REGION Network 2: HOPPER 1 UNIT 01
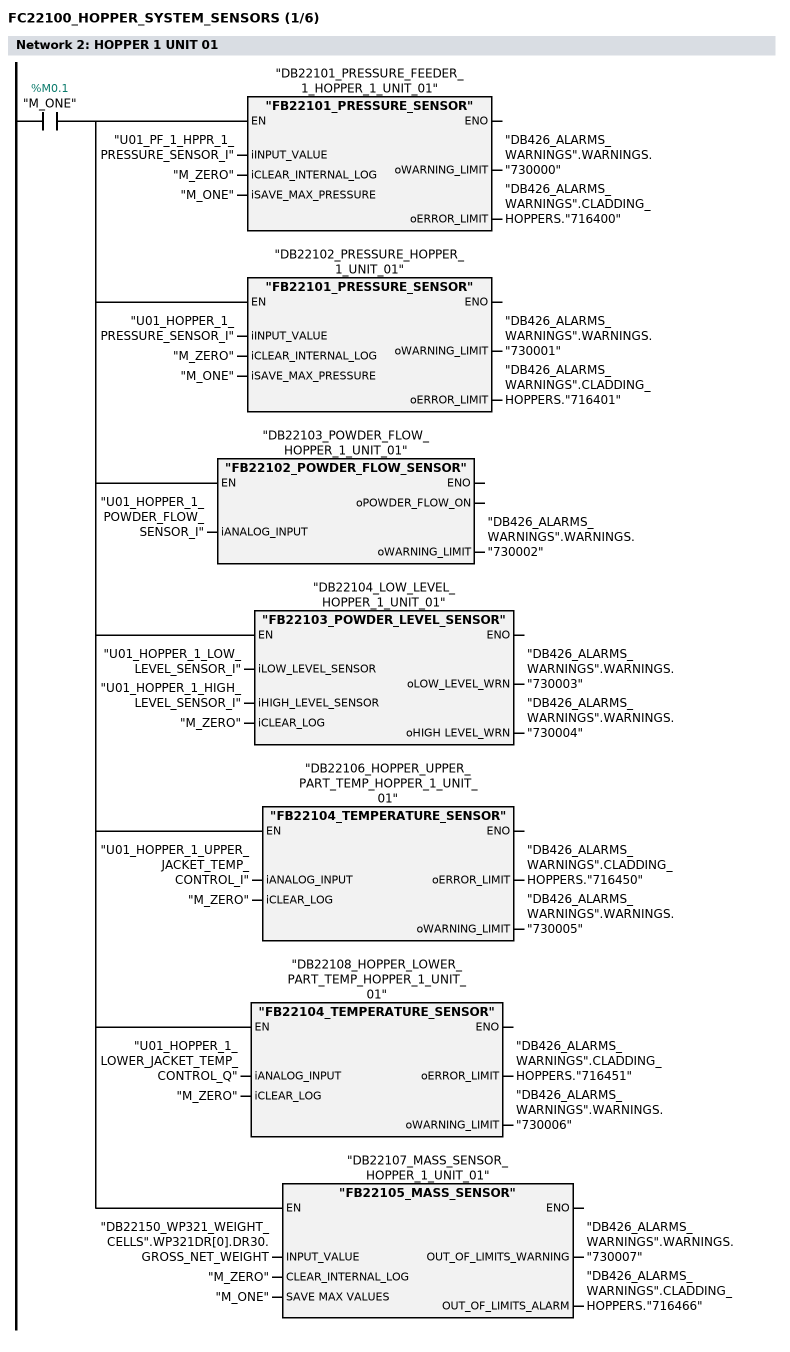
   RUNG wire#powerrail
      Contact( "M_ONE" )
      wire#w1
      "DB22101_PRESSURE_FEEDER_1_HOPPER_1_UNIT_01"(iINPUT_VALUE := "U01_PF_1_HPPR_1_PRESSURE_SENSOR_I", iCLEAR_INTERNAL_LOG := "M_ZERO", iSAVE_MAX_PRESSURE := "M_ONE", oWARNING_LIMIT => "DB426_ALARMS_WARNINGS".WARNINGS."730000", oERROR_LIMIT => "DB426_ALARMS_WARNINGS".CLADDING_HOPPERS."716400")
   END_RUNG
   RUNG wire#w1
      "DB22102_PRESSURE_HOPPER_1_UNIT_01"(iINPUT_VALUE := "U01_HOPPER_1_PRESSURE_SENSOR_I", iCLEAR_INTERNAL_LOG := "M_ZERO", iSAVE_MAX_PRESSURE := "M_ONE", oWARNING_LIMIT => "DB426_ALARMS_WARNINGS".WARNINGS."730001", oERROR_LIMIT => "DB426_ALARMS_WARNINGS".CLADDING_HOPPERS."716401")
   END_RUNG
   RUNG wire#w1
      "DB22103_POWDER_FLOW_HOPPER_1_UNIT_01"(iANALOG_INPUT := "U01_HOPPER_1_POWDER_FLOW_SENSOR_I", oPOWDER_FLOW_ON =>, oWARNING_LIMIT => "DB426_ALARMS_WARNINGS".WARNINGS."730002")
   END_RUNG
   RUNG wire#w1
      "DB22104_LOW_LEVEL_HOPPER_1_UNIT_01"(iLOW_LEVEL_SENSOR := "U01_HOPPER_1_LOW_LEVEL_SENSOR_I", iHIGH_LEVEL_SENSOR := "U01_HOPPER_1_HIGH_LEVEL_SENSOR_I", iCLEAR_LOG := "M_ZERO", oLOW_LEVEL_WRN => "DB426_ALARMS_WARNINGS".WARNINGS."730003", "oHIGH LEVEL_WRN" => "DB426_ALARMS_WARNINGS".WARNINGS."730004")
   END_RUNG
   RUNG wire#w1
      "DB22106_HOPPER_UPPER_PART_TEMP_HOPPER_1_UNIT_01"(iANALOG_INPUT := "U01_HOPPER_1_UPPER_JACKET_TEMP_CONTROL_I", iCLEAR_LOG := "M_ZERO", oERROR_LIMIT => "DB426_ALARMS_WARNINGS".CLADDING_HOPPERS."716450", oWARNING_LIMIT => "DB426_ALARMS_WARNINGS".WARNINGS."730005")
   END_RUNG
   RUNG wire#w1
      "DB22108_HOPPER_LOWER_PART_TEMP_HOPPER_1_UNIT_01"(iANALOG_INPUT := "U01_HOPPER_1_LOWER_JACKET_TEMP_CONTROL_Q", iCLEAR_LOG := "M_ZERO", oERROR_LIMIT => "DB426_ALARMS_WARNINGS".CLADDING_HOPPERS."716451", oWARNING_LIMIT => "DB426_ALARMS_WARNINGS".WARNINGS."730006")
   END_RUNG
   RUNG wire#w1
      "DB22107_MASS_SENSOR_HOPPER_1_UNIT_01"(INPUT_VALUE := "DB22150_WP321_WEIGHT_CELLS".WP321DR[0].DR30.GROSS_NET_WEIGHT, CLEAR_INTERNAL_LOG := "M_ZERO", "SAVE MAX VALUES" := "M_ONE", OUT_OF_LIMITS_WARNING => "DB426_ALARMS_WARNINGS".WARNINGS."730007", OUT_OF_LIMITS_ALARM => "DB426_ALARMS_WARNINGS".CLADDING_HOPPERS."716466")
   END_RUNG
   // the same network as SCL:
   #_w1 := "M_ONE";
   IF #_w1 THEN
       "DB22101_PRESSURE_FEEDER_1_HOPPER_1_UNIT_01"(iINPUT_VALUE := "U01_PF_1_HPPR_1_PRESSURE_SENSOR_I",   // "FB22101_PRESSURE_SENSOR"
                               iCLEAR_INTERNAL_LOG := "M_ZERO",
                               iSAVE_MAX_PRESSURE := "M_ONE",
                               oWARNING_LIMIT => "DB426_ALARMS_WARNINGS".WARNINGS."730000",
                               oERROR_LIMIT => "DB426_ALARMS_WARNINGS".CLADDING_HOPPERS."716400");
       "DB22102_PRESSURE_HOPPER_1_UNIT_01"(iINPUT_VALUE := "U01_HOPPER_1_PRESSURE_SENSOR_I",   // "FB22101_PRESSURE_SENSOR"
                               iCLEAR_INTERNAL_LOG := "M_ZERO",
                               iSAVE_MAX_PRESSURE := "M_ONE",
                               oWARNING_LIMIT => "DB426_ALARMS_WARNINGS".WARNINGS."730001",
                               oERROR_LIMIT => "DB426_ALARMS_WARNINGS".CLADDING_HOPPERS."716401");
       "DB22103_POWDER_FLOW_HOPPER_1_UNIT_01"(iANALOG_INPUT := "U01_HOPPER_1_POWDER_FLOW_SENSOR_I",   // "FB22102_POWDER_FLOW_SENSOR"
                               oWARNING_LIMIT => "DB426_ALARMS_WARNINGS".WARNINGS."730002");
       "DB22104_LOW_LEVEL_HOPPER_1_UNIT_01"(iLOW_LEVEL_SENSOR := "U01_HOPPER_1_LOW_LEVEL_SENSOR_I",   // "FB22103_POWDER_LEVEL_SENSOR"
                               iHIGH_LEVEL_SENSOR := "U01_HOPPER_1_HIGH_LEVEL_SENSOR_I",
                               iCLEAR_LOG := "M_ZERO",
                               oLOW_LEVEL_WRN => "DB426_ALARMS_WARNINGS".WARNINGS."730003",
                               "oHIGH LEVEL_WRN" => "DB426_ALARMS_WARNINGS".WARNINGS."730004");
       "DB22106_HOPPER_UPPER_PART_TEMP_HOPPER_1_UNIT_01"(iANALOG_INPUT := "U01_HOPPER_1_UPPER_JACKET_TEMP_CONTROL_I",   // "FB22104_TEMPERATURE_SENSOR"
                               iCLEAR_LOG := "M_ZERO",
                               oERROR_LIMIT => "DB426_ALARMS_WARNINGS".CLADDING_HOPPERS."716450",
                               oWARNING_LIMIT => "DB426_ALARMS_WARNINGS".WARNINGS."730005");
       "DB22108_HOPPER_LOWER_PART_TEMP_HOPPER_1_UNIT_01"(iANALOG_INPUT := "U01_HOPPER_1_LOWER_JACKET_TEMP_CONTROL_Q",   // "FB22104_TEMPERATURE_SENSOR"
                               iCLEAR_LOG := "M_ZERO",
                               oERROR_LIMIT => "DB426_ALARMS_WARNINGS".CLADDING_HOPPERS."716451",
                               oWARNING_LIMIT => "DB426_ALARMS_WARNINGS".WARNINGS."730006");
       "DB22107_MASS_SENSOR_HOPPER_1_UNIT_01"(INPUT_VALUE := "DB22150_WP321_WEIGHT_CELLS".WP321DR[0].DR30.GROSS_NET_WEIGHT,   // "FB22105_MASS_SENSOR"
                               CLEAR_INTERNAL_LOG := "M_ZERO",
                               "SAVE MAX VALUES" := "M_ONE",
                               OUT_OF_LIMITS_WARNING => "DB426_ALARMS_WARNINGS".WARNINGS."730007",
                               OUT_OF_LIMITS_ALARM => "DB426_ALARMS_WARNINGS".CLADDING_HOPPERS."716466");
   END_IF;
END_REGION

REGION Network 3: HOPPER 2 UNIT 01
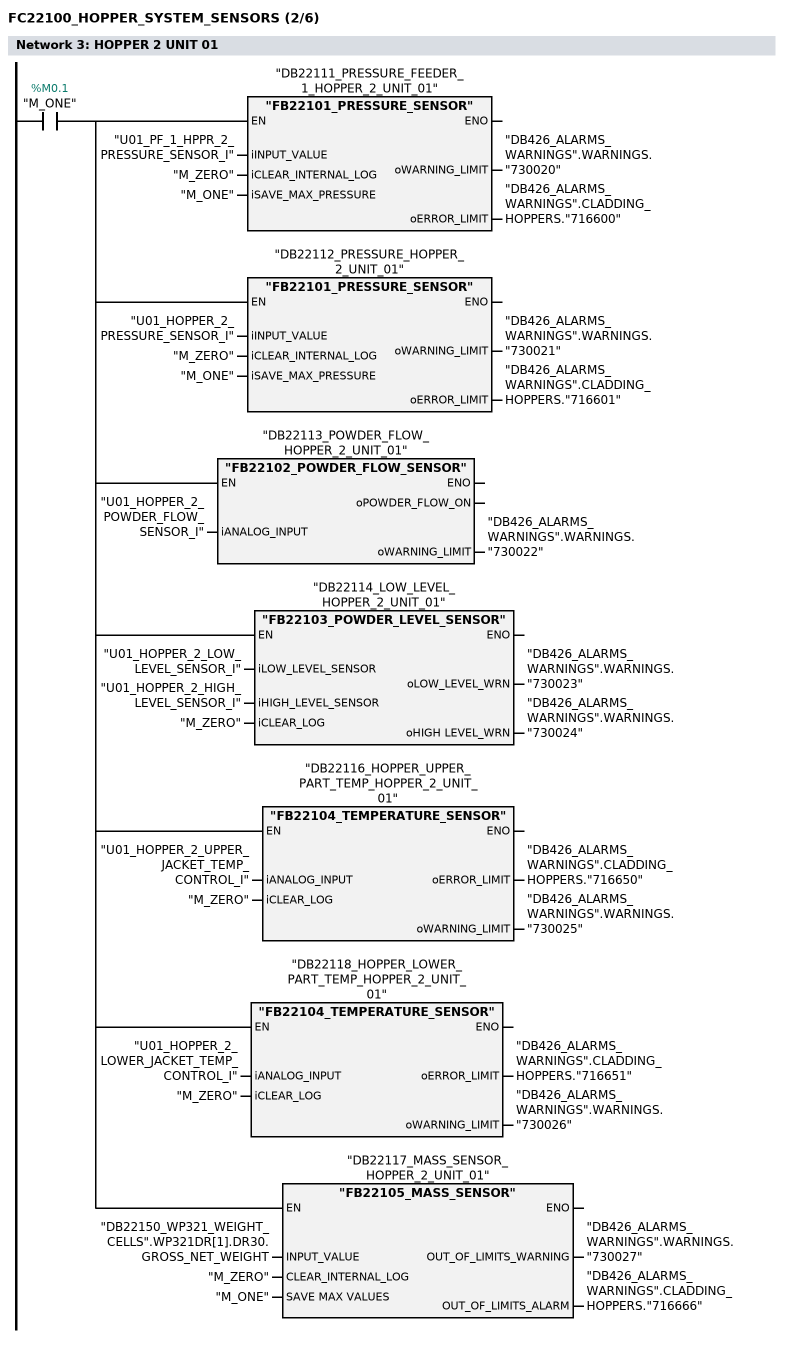
   RUNG wire#powerrail
      Contact( "M_ONE" )
      wire#w1
      "DB22111_PRESSURE_FEEDER_1_HOPPER_2_UNIT_01"(iINPUT_VALUE := "U01_PF_1_HPPR_2_PRESSURE_SENSOR_I", iCLEAR_INTERNAL_LOG := "M_ZERO", iSAVE_MAX_PRESSURE := "M_ONE", oWARNING_LIMIT => "DB426_ALARMS_WARNINGS".WARNINGS."730020", oERROR_LIMIT => "DB426_ALARMS_WARNINGS".CLADDING_HOPPERS."716600")
   END_RUNG
   RUNG wire#w1
      "DB22112_PRESSURE_HOPPER_2_UNIT_01"(iINPUT_VALUE := "U01_HOPPER_2_PRESSURE_SENSOR_I", iCLEAR_INTERNAL_LOG := "M_ZERO", iSAVE_MAX_PRESSURE := "M_ONE", oWARNING_LIMIT => "DB426_ALARMS_WARNINGS".WARNINGS."730021", oERROR_LIMIT => "DB426_ALARMS_WARNINGS".CLADDING_HOPPERS."716601")
   END_RUNG
   RUNG wire#w1
      "DB22113_POWDER_FLOW_HOPPER_2_UNIT_01"(iANALOG_INPUT := "U01_HOPPER_2_POWDER_FLOW_SENSOR_I", oPOWDER_FLOW_ON =>, oWARNING_LIMIT => "DB426_ALARMS_WARNINGS".WARNINGS."730022")
   END_RUNG
   RUNG wire#w1
      "DB22114_LOW_LEVEL_HOPPER_2_UNIT_01"(iLOW_LEVEL_SENSOR := "U01_HOPPER_2_LOW_LEVEL_SENSOR_I", iHIGH_LEVEL_SENSOR := "U01_HOPPER_2_HIGH_LEVEL_SENSOR_I", iCLEAR_LOG := "M_ZERO", oLOW_LEVEL_WRN => "DB426_ALARMS_WARNINGS".WARNINGS."730023", "oHIGH LEVEL_WRN" => "DB426_ALARMS_WARNINGS".WARNINGS."730024")
   END_RUNG
   RUNG wire#w1
      "DB22116_HOPPER_UPPER_PART_TEMP_HOPPER_2_UNIT_01"(iANALOG_INPUT := "U01_HOPPER_2_UPPER_JACKET_TEMP_CONTROL_I", iCLEAR_LOG := "M_ZERO", oERROR_LIMIT => "DB426_ALARMS_WARNINGS".CLADDING_HOPPERS."716650", oWARNING_LIMIT => "DB426_ALARMS_WARNINGS".WARNINGS."730025")
   END_RUNG
   RUNG wire#w1
      "DB22118_HOPPER_LOWER_PART_TEMP_HOPPER_2_UNIT_01"(iANALOG_INPUT := "U01_HOPPER_2_LOWER_JACKET_TEMP_CONTROL_I", iCLEAR_LOG := "M_ZERO", oERROR_LIMIT => "DB426_ALARMS_WARNINGS".CLADDING_HOPPERS."716651", oWARNING_LIMIT => "DB426_ALARMS_WARNINGS".WARNINGS."730026")
   END_RUNG
   RUNG wire#w1
      "DB22117_MASS_SENSOR_HOPPER_2_UNIT_01"(INPUT_VALUE := "DB22150_WP321_WEIGHT_CELLS".WP321DR[1].DR30.GROSS_NET_WEIGHT, CLEAR_INTERNAL_LOG := "M_ZERO", "SAVE MAX VALUES" := "M_ONE", OUT_OF_LIMITS_WARNING => "DB426_ALARMS_WARNINGS".WARNINGS."730027", OUT_OF_LIMITS_ALARM => "DB426_ALARMS_WARNINGS".CLADDING_HOPPERS."716666")
   END_RUNG
   // the same network as SCL:
   #_w1 := "M_ONE";
   IF #_w1 THEN
       "DB22111_PRESSURE_FEEDER_1_HOPPER_2_UNIT_01"(iINPUT_VALUE := "U01_PF_1_HPPR_2_PRESSURE_SENSOR_I",   // "FB22101_PRESSURE_SENSOR"
                               iCLEAR_INTERNAL_LOG := "M_ZERO",
                               iSAVE_MAX_PRESSURE := "M_ONE",
                               oWARNING_LIMIT => "DB426_ALARMS_WARNINGS".WARNINGS."730020",
                               oERROR_LIMIT => "DB426_ALARMS_WARNINGS".CLADDING_HOPPERS."716600");
       "DB22112_PRESSURE_HOPPER_2_UNIT_01"(iINPUT_VALUE := "U01_HOPPER_2_PRESSURE_SENSOR_I",   // "FB22101_PRESSURE_SENSOR"
                               iCLEAR_INTERNAL_LOG := "M_ZERO",
                               iSAVE_MAX_PRESSURE := "M_ONE",
                               oWARNING_LIMIT => "DB426_ALARMS_WARNINGS".WARNINGS."730021",
                               oERROR_LIMIT => "DB426_ALARMS_WARNINGS".CLADDING_HOPPERS."716601");
       "DB22113_POWDER_FLOW_HOPPER_2_UNIT_01"(iANALOG_INPUT := "U01_HOPPER_2_POWDER_FLOW_SENSOR_I",   // "FB22102_POWDER_FLOW_SENSOR"
                               oWARNING_LIMIT => "DB426_ALARMS_WARNINGS".WARNINGS."730022");
       "DB22114_LOW_LEVEL_HOPPER_2_UNIT_01"(iLOW_LEVEL_SENSOR := "U01_HOPPER_2_LOW_LEVEL_SENSOR_I",   // "FB22103_POWDER_LEVEL_SENSOR"
                               iHIGH_LEVEL_SENSOR := "U01_HOPPER_2_HIGH_LEVEL_SENSOR_I",
                               iCLEAR_LOG := "M_ZERO",
                               oLOW_LEVEL_WRN => "DB426_ALARMS_WARNINGS".WARNINGS."730023",
                               "oHIGH LEVEL_WRN" => "DB426_ALARMS_WARNINGS".WARNINGS."730024");
       "DB22116_HOPPER_UPPER_PART_TEMP_HOPPER_2_UNIT_01"(iANALOG_INPUT := "U01_HOPPER_2_UPPER_JACKET_TEMP_CONTROL_I",   // "FB22104_TEMPERATURE_SENSOR"
                               iCLEAR_LOG := "M_ZERO",
                               oERROR_LIMIT => "DB426_ALARMS_WARNINGS".CLADDING_HOPPERS."716650",
                               oWARNING_LIMIT => "DB426_ALARMS_WARNINGS".WARNINGS."730025");
       "DB22118_HOPPER_LOWER_PART_TEMP_HOPPER_2_UNIT_01"(iANALOG_INPUT := "U01_HOPPER_2_LOWER_JACKET_TEMP_CONTROL_I",   // "FB22104_TEMPERATURE_SENSOR"
                               iCLEAR_LOG := "M_ZERO",
                               oERROR_LIMIT => "DB426_ALARMS_WARNINGS".CLADDING_HOPPERS."716651",
                               oWARNING_LIMIT => "DB426_ALARMS_WARNINGS".WARNINGS."730026");
       "DB22117_MASS_SENSOR_HOPPER_2_UNIT_01"(INPUT_VALUE := "DB22150_WP321_WEIGHT_CELLS".WP321DR[1].DR30.GROSS_NET_WEIGHT,   // "FB22105_MASS_SENSOR"
                               CLEAR_INTERNAL_LOG := "M_ZERO",
                               "SAVE MAX VALUES" := "M_ONE",
                               OUT_OF_LIMITS_WARNING => "DB426_ALARMS_WARNINGS".WARNINGS."730027",
                               OUT_OF_LIMITS_ALARM => "DB426_ALARMS_WARNINGS".CLADDING_HOPPERS."716666");
   END_IF;
END_REGION

REGION Network 4: /////_UNIT_02_SENSORS_/////
END_REGION

REGION Network 5: HOPPER 1 UNIT 02
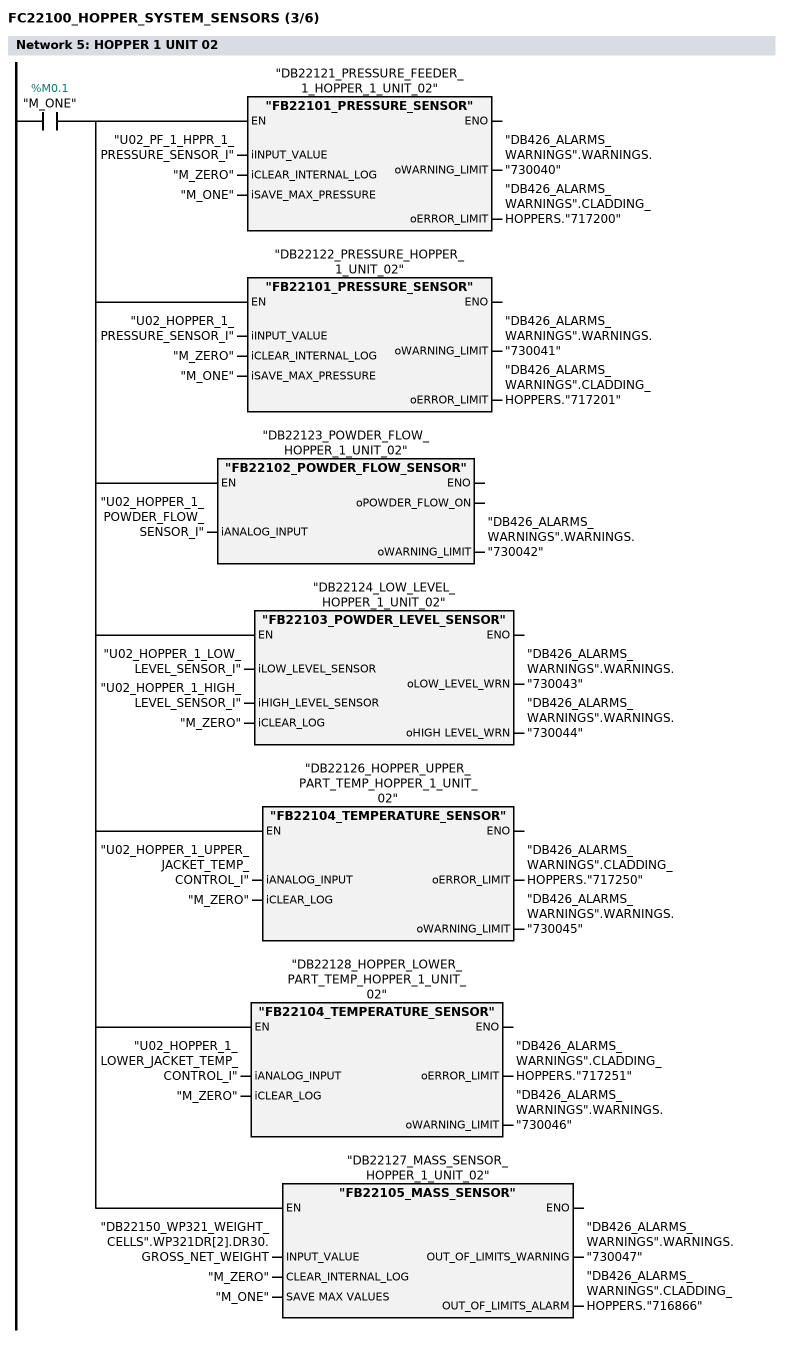
   RUNG wire#powerrail
      Contact( "M_ONE" )
      wire#w1
      "DB22121_PRESSURE_FEEDER_1_HOPPER_1_UNIT_02"(iINPUT_VALUE := "U02_PF_1_HPPR_1_PRESSURE_SENSOR_I", iCLEAR_INTERNAL_LOG := "M_ZERO", iSAVE_MAX_PRESSURE := "M_ONE", oWARNING_LIMIT => "DB426_ALARMS_WARNINGS".WARNINGS."730040", oERROR_LIMIT => "DB426_ALARMS_WARNINGS".CLADDING_HOPPERS."717200")
   END_RUNG
   RUNG wire#w1
      "DB22122_PRESSURE_HOPPER_1_UNIT_02"(iINPUT_VALUE := "U02_HOPPER_1_PRESSURE_SENSOR_I", iCLEAR_INTERNAL_LOG := "M_ZERO", iSAVE_MAX_PRESSURE := "M_ONE", oWARNING_LIMIT => "DB426_ALARMS_WARNINGS".WARNINGS."730041", oERROR_LIMIT => "DB426_ALARMS_WARNINGS".CLADDING_HOPPERS."717201")
   END_RUNG
   RUNG wire#w1
      "DB22123_POWDER_FLOW_HOPPER_1_UNIT_02"(iANALOG_INPUT := "U02_HOPPER_1_POWDER_FLOW_SENSOR_I", oPOWDER_FLOW_ON =>, oWARNING_LIMIT => "DB426_ALARMS_WARNINGS".WARNINGS."730042")
   END_RUNG
   RUNG wire#w1
      "DB22124_LOW_LEVEL_HOPPER_1_UNIT_02"(iLOW_LEVEL_SENSOR := "U02_HOPPER_1_LOW_LEVEL_SENSOR_I", iHIGH_LEVEL_SENSOR := "U02_HOPPER_1_HIGH_LEVEL_SENSOR_I", iCLEAR_LOG := "M_ZERO", oLOW_LEVEL_WRN => "DB426_ALARMS_WARNINGS".WARNINGS."730043", "oHIGH LEVEL_WRN" => "DB426_ALARMS_WARNINGS".WARNINGS."730044")
   END_RUNG
   RUNG wire#w1
      "DB22126_HOPPER_UPPER_PART_TEMP_HOPPER_1_UNIT_02"(iANALOG_INPUT := "U02_HOPPER_1_UPPER_JACKET_TEMP_CONTROL_I", iCLEAR_LOG := "M_ZERO", oERROR_LIMIT => "DB426_ALARMS_WARNINGS".CLADDING_HOPPERS."717250", oWARNING_LIMIT => "DB426_ALARMS_WARNINGS".WARNINGS."730045")
   END_RUNG
   RUNG wire#w1
      "DB22128_HOPPER_LOWER_PART_TEMP_HOPPER_1_UNIT_02"(iANALOG_INPUT := "U02_HOPPER_1_LOWER_JACKET_TEMP_CONTROL_I", iCLEAR_LOG := "M_ZERO", oERROR_LIMIT => "DB426_ALARMS_WARNINGS".CLADDING_HOPPERS."717251", oWARNING_LIMIT => "DB426_ALARMS_WARNINGS".WARNINGS."730046")
   END_RUNG
   RUNG wire#w1
      "DB22127_MASS_SENSOR_HOPPER_1_UNIT_02"(INPUT_VALUE := "DB22150_WP321_WEIGHT_CELLS".WP321DR[2].DR30.GROSS_NET_WEIGHT, CLEAR_INTERNAL_LOG := "M_ZERO", "SAVE MAX VALUES" := "M_ONE", OUT_OF_LIMITS_WARNING => "DB426_ALARMS_WARNINGS".WARNINGS."730047", OUT_OF_LIMITS_ALARM => "DB426_ALARMS_WARNINGS".CLADDING_HOPPERS."716866")
   END_RUNG
   // the same network as SCL:
   #_w1 := "M_ONE";
   IF #_w1 THEN
       "DB22121_PRESSURE_FEEDER_1_HOPPER_1_UNIT_02"(iINPUT_VALUE := "U02_PF_1_HPPR_1_PRESSURE_SENSOR_I",   // "FB22101_PRESSURE_SENSOR"
                               iCLEAR_INTERNAL_LOG := "M_ZERO",
                               iSAVE_MAX_PRESSURE := "M_ONE",
                               oWARNING_LIMIT => "DB426_ALARMS_WARNINGS".WARNINGS."730040",
                               oERROR_LIMIT => "DB426_ALARMS_WARNINGS".CLADDING_HOPPERS."717200");
       "DB22122_PRESSURE_HOPPER_1_UNIT_02"(iINPUT_VALUE := "U02_HOPPER_1_PRESSURE_SENSOR_I",   // "FB22101_PRESSURE_SENSOR"
                               iCLEAR_INTERNAL_LOG := "M_ZERO",
                               iSAVE_MAX_PRESSURE := "M_ONE",
                               oWARNING_LIMIT => "DB426_ALARMS_WARNINGS".WARNINGS."730041",
                               oERROR_LIMIT => "DB426_ALARMS_WARNINGS".CLADDING_HOPPERS."717201");
       "DB22123_POWDER_FLOW_HOPPER_1_UNIT_02"(iANALOG_INPUT := "U02_HOPPER_1_POWDER_FLOW_SENSOR_I",   // "FB22102_POWDER_FLOW_SENSOR"
                               oWARNING_LIMIT => "DB426_ALARMS_WARNINGS".WARNINGS."730042");
       "DB22124_LOW_LEVEL_HOPPER_1_UNIT_02"(iLOW_LEVEL_SENSOR := "U02_HOPPER_1_LOW_LEVEL_SENSOR_I",   // "FB22103_POWDER_LEVEL_SENSOR"
                               iHIGH_LEVEL_SENSOR := "U02_HOPPER_1_HIGH_LEVEL_SENSOR_I",
                               iCLEAR_LOG := "M_ZERO",
                               oLOW_LEVEL_WRN => "DB426_ALARMS_WARNINGS".WARNINGS."730043",
                               "oHIGH LEVEL_WRN" => "DB426_ALARMS_WARNINGS".WARNINGS."730044");
       "DB22126_HOPPER_UPPER_PART_TEMP_HOPPER_1_UNIT_02"(iANALOG_INPUT := "U02_HOPPER_1_UPPER_JACKET_TEMP_CONTROL_I",   // "FB22104_TEMPERATURE_SENSOR"
                               iCLEAR_LOG := "M_ZERO",
                               oERROR_LIMIT => "DB426_ALARMS_WARNINGS".CLADDING_HOPPERS."717250",
                               oWARNING_LIMIT => "DB426_ALARMS_WARNINGS".WARNINGS."730045");
       "DB22128_HOPPER_LOWER_PART_TEMP_HOPPER_1_UNIT_02"(iANALOG_INPUT := "U02_HOPPER_1_LOWER_JACKET_TEMP_CONTROL_I",   // "FB22104_TEMPERATURE_SENSOR"
                               iCLEAR_LOG := "M_ZERO",
                               oERROR_LIMIT => "DB426_ALARMS_WARNINGS".CLADDING_HOPPERS."717251",
                               oWARNING_LIMIT => "DB426_ALARMS_WARNINGS".WARNINGS."730046");
       "DB22127_MASS_SENSOR_HOPPER_1_UNIT_02"(INPUT_VALUE := "DB22150_WP321_WEIGHT_CELLS".WP321DR[2].DR30.GROSS_NET_WEIGHT,   // "FB22105_MASS_SENSOR"
                               CLEAR_INTERNAL_LOG := "M_ZERO",
                               "SAVE MAX VALUES" := "M_ONE",
                               OUT_OF_LIMITS_WARNING => "DB426_ALARMS_WARNINGS".WARNINGS."730047",
                               OUT_OF_LIMITS_ALARM => "DB426_ALARMS_WARNINGS".CLADDING_HOPPERS."716866");
   END_IF;
END_REGION

REGION Network 6: HOPPER 2 UNIT 02
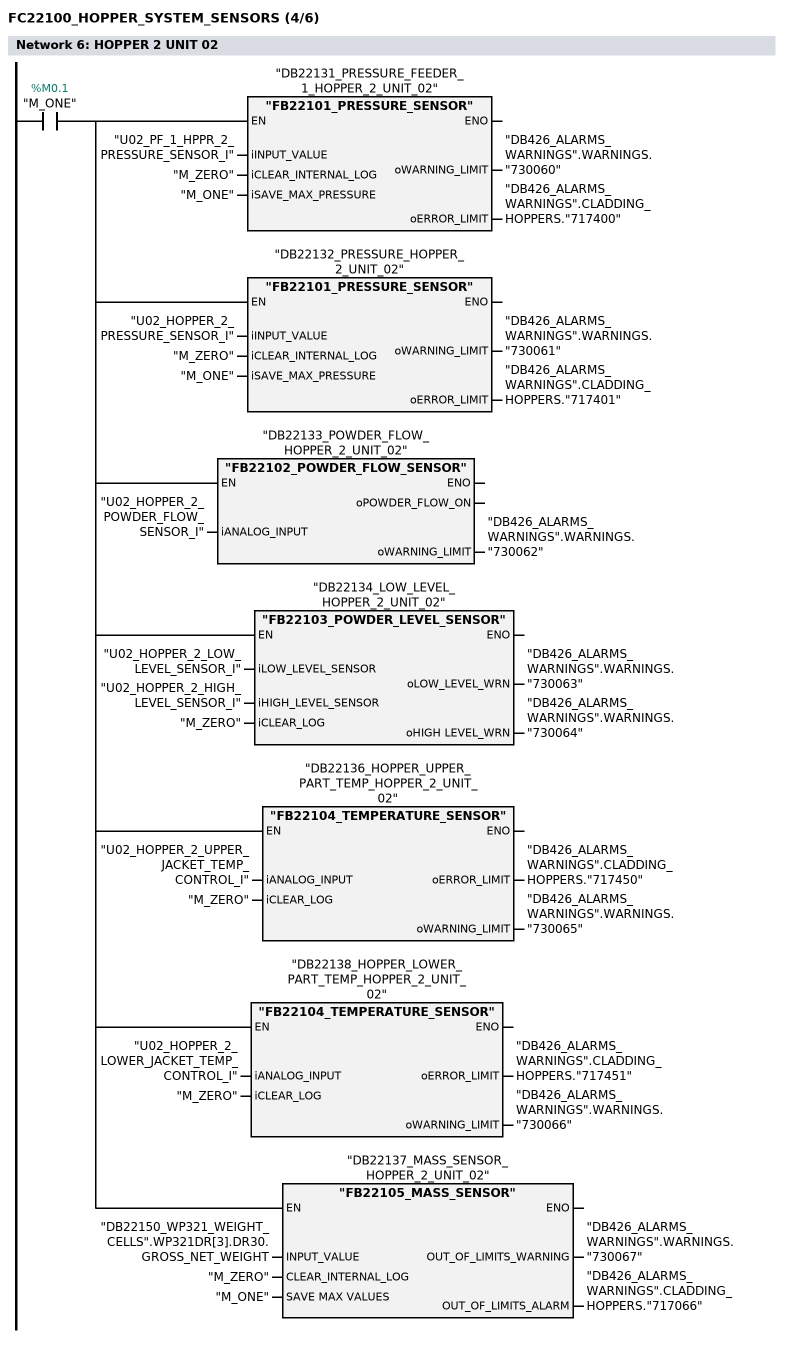
   RUNG wire#powerrail
      Contact( "M_ONE" )
      wire#w1
      "DB22131_PRESSURE_FEEDER_1_HOPPER_2_UNIT_02"(iINPUT_VALUE := "U02_PF_1_HPPR_2_PRESSURE_SENSOR_I", iCLEAR_INTERNAL_LOG := "M_ZERO", iSAVE_MAX_PRESSURE := "M_ONE", oWARNING_LIMIT => "DB426_ALARMS_WARNINGS".WARNINGS."730060", oERROR_LIMIT => "DB426_ALARMS_WARNINGS".CLADDING_HOPPERS."717400")
   END_RUNG
   RUNG wire#w1
      "DB22132_PRESSURE_HOPPER_2_UNIT_02"(iINPUT_VALUE := "U02_HOPPER_2_PRESSURE_SENSOR_I", iCLEAR_INTERNAL_LOG := "M_ZERO", iSAVE_MAX_PRESSURE := "M_ONE", oWARNING_LIMIT => "DB426_ALARMS_WARNINGS".WARNINGS."730061", oERROR_LIMIT => "DB426_ALARMS_WARNINGS".CLADDING_HOPPERS."717401")
   END_RUNG
   RUNG wire#w1
      "DB22133_POWDER_FLOW_HOPPER_2_UNIT_02"(iANALOG_INPUT := "U02_HOPPER_2_POWDER_FLOW_SENSOR_I", oPOWDER_FLOW_ON =>, oWARNING_LIMIT => "DB426_ALARMS_WARNINGS".WARNINGS."730062")
   END_RUNG
   RUNG wire#w1
      "DB22134_LOW_LEVEL_HOPPER_2_UNIT_02"(iLOW_LEVEL_SENSOR := "U02_HOPPER_2_LOW_LEVEL_SENSOR_I", iHIGH_LEVEL_SENSOR := "U02_HOPPER_2_HIGH_LEVEL_SENSOR_I", iCLEAR_LOG := "M_ZERO", oLOW_LEVEL_WRN => "DB426_ALARMS_WARNINGS".WARNINGS."730063", "oHIGH LEVEL_WRN" => "DB426_ALARMS_WARNINGS".WARNINGS."730064")
   END_RUNG
   RUNG wire#w1
      "DB22136_HOPPER_UPPER_PART_TEMP_HOPPER_2_UNIT_02"(iANALOG_INPUT := "U02_HOPPER_2_UPPER_JACKET_TEMP_CONTROL_I", iCLEAR_LOG := "M_ZERO", oERROR_LIMIT => "DB426_ALARMS_WARNINGS".CLADDING_HOPPERS."717450", oWARNING_LIMIT => "DB426_ALARMS_WARNINGS".WARNINGS."730065")
   END_RUNG
   RUNG wire#w1
      "DB22138_HOPPER_LOWER_PART_TEMP_HOPPER_2_UNIT_02"(iANALOG_INPUT := "U02_HOPPER_2_LOWER_JACKET_TEMP_CONTROL_I", iCLEAR_LOG := "M_ZERO", oERROR_LIMIT => "DB426_ALARMS_WARNINGS".CLADDING_HOPPERS."717451", oWARNING_LIMIT => "DB426_ALARMS_WARNINGS".WARNINGS."730066")
   END_RUNG
   RUNG wire#w1
      "DB22137_MASS_SENSOR_HOPPER_2_UNIT_02"(INPUT_VALUE := "DB22150_WP321_WEIGHT_CELLS".WP321DR[3].DR30.GROSS_NET_WEIGHT, CLEAR_INTERNAL_LOG := "M_ZERO", "SAVE MAX VALUES" := "M_ONE", OUT_OF_LIMITS_WARNING => "DB426_ALARMS_WARNINGS".WARNINGS."730067", OUT_OF_LIMITS_ALARM => "DB426_ALARMS_WARNINGS".CLADDING_HOPPERS."717066")
   END_RUNG
   // the same network as SCL:
   #_w1 := "M_ONE";
   IF #_w1 THEN
       "DB22131_PRESSURE_FEEDER_1_HOPPER_2_UNIT_02"(iINPUT_VALUE := "U02_PF_1_HPPR_2_PRESSURE_SENSOR_I",   // "FB22101_PRESSURE_SENSOR"
                               iCLEAR_INTERNAL_LOG := "M_ZERO",
                               iSAVE_MAX_PRESSURE := "M_ONE",
                               oWARNING_LIMIT => "DB426_ALARMS_WARNINGS".WARNINGS."730060",
                               oERROR_LIMIT => "DB426_ALARMS_WARNINGS".CLADDING_HOPPERS."717400");
       "DB22132_PRESSURE_HOPPER_2_UNIT_02"(iINPUT_VALUE := "U02_HOPPER_2_PRESSURE_SENSOR_I",   // "FB22101_PRESSURE_SENSOR"
                               iCLEAR_INTERNAL_LOG := "M_ZERO",
                               iSAVE_MAX_PRESSURE := "M_ONE",
                               oWARNING_LIMIT => "DB426_ALARMS_WARNINGS".WARNINGS."730061",
                               oERROR_LIMIT => "DB426_ALARMS_WARNINGS".CLADDING_HOPPERS."717401");
       "DB22133_POWDER_FLOW_HOPPER_2_UNIT_02"(iANALOG_INPUT := "U02_HOPPER_2_POWDER_FLOW_SENSOR_I",   // "FB22102_POWDER_FLOW_SENSOR"
                               oWARNING_LIMIT => "DB426_ALARMS_WARNINGS".WARNINGS."730062");
       "DB22134_LOW_LEVEL_HOPPER_2_UNIT_02"(iLOW_LEVEL_SENSOR := "U02_HOPPER_2_LOW_LEVEL_SENSOR_I",   // "FB22103_POWDER_LEVEL_SENSOR"
                               iHIGH_LEVEL_SENSOR := "U02_HOPPER_2_HIGH_LEVEL_SENSOR_I",
                               iCLEAR_LOG := "M_ZERO",
                               oLOW_LEVEL_WRN => "DB426_ALARMS_WARNINGS".WARNINGS."730063",
                               "oHIGH LEVEL_WRN" => "DB426_ALARMS_WARNINGS".WARNINGS."730064");
       "DB22136_HOPPER_UPPER_PART_TEMP_HOPPER_2_UNIT_02"(iANALOG_INPUT := "U02_HOPPER_2_UPPER_JACKET_TEMP_CONTROL_I",   // "FB22104_TEMPERATURE_SENSOR"
                               iCLEAR_LOG := "M_ZERO",
                               oERROR_LIMIT => "DB426_ALARMS_WARNINGS".CLADDING_HOPPERS."717450",
                               oWARNING_LIMIT => "DB426_ALARMS_WARNINGS".WARNINGS."730065");
       "DB22138_HOPPER_LOWER_PART_TEMP_HOPPER_2_UNIT_02"(iANALOG_INPUT := "U02_HOPPER_2_LOWER_JACKET_TEMP_CONTROL_I",   // "FB22104_TEMPERATURE_SENSOR"
                               iCLEAR_LOG := "M_ZERO",
                               oERROR_LIMIT => "DB426_ALARMS_WARNINGS".CLADDING_HOPPERS."717451",
                               oWARNING_LIMIT => "DB426_ALARMS_WARNINGS".WARNINGS."730066");
       "DB22137_MASS_SENSOR_HOPPER_2_UNIT_02"(INPUT_VALUE := "DB22150_WP321_WEIGHT_CELLS".WP321DR[3].DR30.GROSS_NET_WEIGHT,   // "FB22105_MASS_SENSOR"
                               CLEAR_INTERNAL_LOG := "M_ZERO",
                               "SAVE MAX VALUES" := "M_ONE",
                               OUT_OF_LIMITS_WARNING => "DB426_ALARMS_WARNINGS".WARNINGS."730067",
                               OUT_OF_LIMITS_ALARM => "DB426_ALARMS_WARNINGS".CLADDING_HOPPERS."717066");
   END_IF;
END_REGION

REGION Network 7: HOPPER 3 UNIT 02
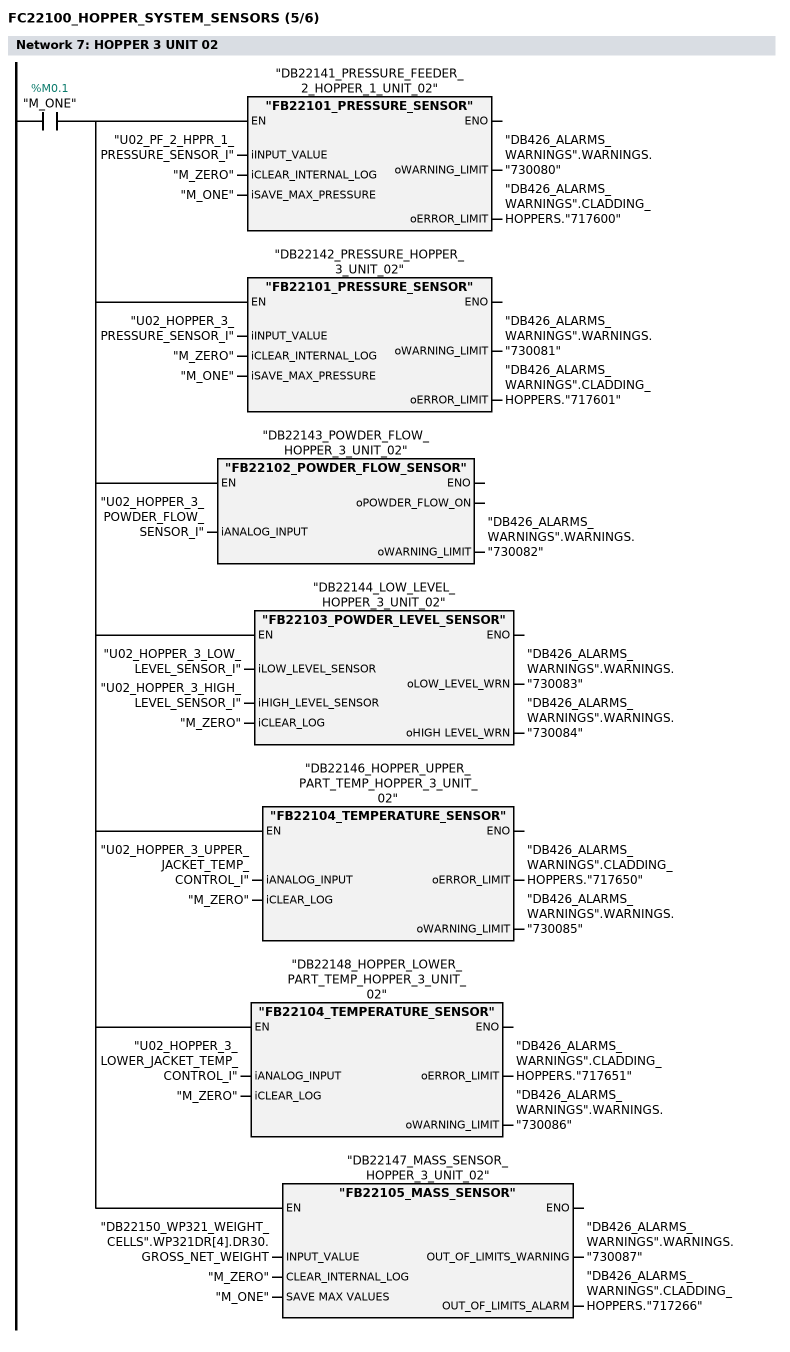
   RUNG wire#powerrail
      Contact( "M_ONE" )
      wire#w1
      "DB22141_PRESSURE_FEEDER_2_HOPPER_1_UNIT_02"(iINPUT_VALUE := "U02_PF_2_HPPR_1_PRESSURE_SENSOR_I", iCLEAR_INTERNAL_LOG := "M_ZERO", iSAVE_MAX_PRESSURE := "M_ONE", oWARNING_LIMIT => "DB426_ALARMS_WARNINGS".WARNINGS."730080", oERROR_LIMIT => "DB426_ALARMS_WARNINGS".CLADDING_HOPPERS."717600")
   END_RUNG
   RUNG wire#w1
      "DB22142_PRESSURE_HOPPER_3_UNIT_02"(iINPUT_VALUE := "U02_HOPPER_3_PRESSURE_SENSOR_I", iCLEAR_INTERNAL_LOG := "M_ZERO", iSAVE_MAX_PRESSURE := "M_ONE", oWARNING_LIMIT => "DB426_ALARMS_WARNINGS".WARNINGS."730081", oERROR_LIMIT => "DB426_ALARMS_WARNINGS".CLADDING_HOPPERS."717601")
   END_RUNG
   RUNG wire#w1
      "DB22143_POWDER_FLOW_HOPPER_3_UNIT_02"(iANALOG_INPUT := "U02_HOPPER_3_POWDER_FLOW_SENSOR_I", oPOWDER_FLOW_ON =>, oWARNING_LIMIT => "DB426_ALARMS_WARNINGS".WARNINGS."730082")
   END_RUNG
   RUNG wire#w1
      "DB22144_LOW_LEVEL_HOPPER_3_UNIT_02"(iLOW_LEVEL_SENSOR := "U02_HOPPER_3_LOW_LEVEL_SENSOR_I", iHIGH_LEVEL_SENSOR := "U02_HOPPER_3_HIGH_LEVEL_SENSOR_I", iCLEAR_LOG := "M_ZERO", oLOW_LEVEL_WRN => "DB426_ALARMS_WARNINGS".WARNINGS."730083", "oHIGH LEVEL_WRN" => "DB426_ALARMS_WARNINGS".WARNINGS."730084")
   END_RUNG
   RUNG wire#w1
      "DB22146_HOPPER_UPPER_PART_TEMP_HOPPER_3_UNIT_02"(iANALOG_INPUT := "U02_HOPPER_3_UPPER_JACKET_TEMP_CONTROL_I", iCLEAR_LOG := "M_ZERO", oERROR_LIMIT => "DB426_ALARMS_WARNINGS".CLADDING_HOPPERS."717650", oWARNING_LIMIT => "DB426_ALARMS_WARNINGS".WARNINGS."730085")
   END_RUNG
   RUNG wire#w1
      "DB22148_HOPPER_LOWER_PART_TEMP_HOPPER_3_UNIT_02"(iANALOG_INPUT := "U02_HOPPER_3_LOWER_JACKET_TEMP_CONTROL_I", iCLEAR_LOG := "M_ZERO", oERROR_LIMIT => "DB426_ALARMS_WARNINGS".CLADDING_HOPPERS."717651", oWARNING_LIMIT => "DB426_ALARMS_WARNINGS".WARNINGS."730086")
   END_RUNG
   RUNG wire#w1
      "DB22147_MASS_SENSOR_HOPPER_3_UNIT_02"(INPUT_VALUE := "DB22150_WP321_WEIGHT_CELLS".WP321DR[4].DR30.GROSS_NET_WEIGHT, CLEAR_INTERNAL_LOG := "M_ZERO", "SAVE MAX VALUES" := "M_ONE", OUT_OF_LIMITS_WARNING => "DB426_ALARMS_WARNINGS".WARNINGS."730087", OUT_OF_LIMITS_ALARM => "DB426_ALARMS_WARNINGS".CLADDING_HOPPERS."717266")
   END_RUNG
   // the same network as SCL:
   #_w1 := "M_ONE";
   IF #_w1 THEN
       "DB22141_PRESSURE_FEEDER_2_HOPPER_1_UNIT_02"(iINPUT_VALUE := "U02_PF_2_HPPR_1_PRESSURE_SENSOR_I",   // "FB22101_PRESSURE_SENSOR"
                               iCLEAR_INTERNAL_LOG := "M_ZERO",
                               iSAVE_MAX_PRESSURE := "M_ONE",
                               oWARNING_LIMIT => "DB426_ALARMS_WARNINGS".WARNINGS."730080",
                               oERROR_LIMIT => "DB426_ALARMS_WARNINGS".CLADDING_HOPPERS."717600");
       "DB22142_PRESSURE_HOPPER_3_UNIT_02"(iINPUT_VALUE := "U02_HOPPER_3_PRESSURE_SENSOR_I",   // "FB22101_PRESSURE_SENSOR"
                               iCLEAR_INTERNAL_LOG := "M_ZERO",
                               iSAVE_MAX_PRESSURE := "M_ONE",
                               oWARNING_LIMIT => "DB426_ALARMS_WARNINGS".WARNINGS."730081",
                               oERROR_LIMIT => "DB426_ALARMS_WARNINGS".CLADDING_HOPPERS."717601");
       "DB22143_POWDER_FLOW_HOPPER_3_UNIT_02"(iANALOG_INPUT := "U02_HOPPER_3_POWDER_FLOW_SENSOR_I",   // "FB22102_POWDER_FLOW_SENSOR"
                               oWARNING_LIMIT => "DB426_ALARMS_WARNINGS".WARNINGS."730082");
       "DB22144_LOW_LEVEL_HOPPER_3_UNIT_02"(iLOW_LEVEL_SENSOR := "U02_HOPPER_3_LOW_LEVEL_SENSOR_I",   // "FB22103_POWDER_LEVEL_SENSOR"
                               iHIGH_LEVEL_SENSOR := "U02_HOPPER_3_HIGH_LEVEL_SENSOR_I",
                               iCLEAR_LOG := "M_ZERO",
                               oLOW_LEVEL_WRN => "DB426_ALARMS_WARNINGS".WARNINGS."730083",
                               "oHIGH LEVEL_WRN" => "DB426_ALARMS_WARNINGS".WARNINGS."730084");
       "DB22146_HOPPER_UPPER_PART_TEMP_HOPPER_3_UNIT_02"(iANALOG_INPUT := "U02_HOPPER_3_UPPER_JACKET_TEMP_CONTROL_I",   // "FB22104_TEMPERATURE_SENSOR"
                               iCLEAR_LOG := "M_ZERO",
                               oERROR_LIMIT => "DB426_ALARMS_WARNINGS".CLADDING_HOPPERS."717650",
                               oWARNING_LIMIT => "DB426_ALARMS_WARNINGS".WARNINGS."730085");
       "DB22148_HOPPER_LOWER_PART_TEMP_HOPPER_3_UNIT_02"(iANALOG_INPUT := "U02_HOPPER_3_LOWER_JACKET_TEMP_CONTROL_I",   // "FB22104_TEMPERATURE_SENSOR"
                               iCLEAR_LOG := "M_ZERO",
                               oERROR_LIMIT => "DB426_ALARMS_WARNINGS".CLADDING_HOPPERS."717651",
                               oWARNING_LIMIT => "DB426_ALARMS_WARNINGS".WARNINGS."730086");
       "DB22147_MASS_SENSOR_HOPPER_3_UNIT_02"(INPUT_VALUE := "DB22150_WP321_WEIGHT_CELLS".WP321DR[4].DR30.GROSS_NET_WEIGHT,   // "FB22105_MASS_SENSOR"
                               CLEAR_INTERNAL_LOG := "M_ZERO",
                               "SAVE MAX VALUES" := "M_ONE",
                               OUT_OF_LIMITS_WARNING => "DB426_ALARMS_WARNINGS".WARNINGS."730087",
                               OUT_OF_LIMITS_ALARM => "DB426_ALARMS_WARNINGS".CLADDING_HOPPERS."717266");
   END_IF;
END_REGION

REGION Network 8: CALL FB22108 WP321_MUL_CALL
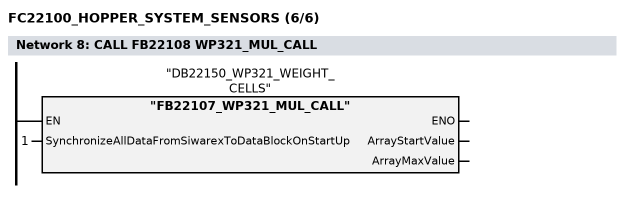
   RUNG wire#powerrail
      "DB22150_WP321_WEIGHT_CELLS"(SynchronizeAllDataFromSiwarexToDataBlockOnStartUp := 1, ArrayStartValue =>, ArrayMaxValue =>)
   END_RUNG
   // the same network as SCL:
   "DB22150_WP321_WEIGHT_CELLS"(SynchronizeAllDataFromSiwarexToDataBlockOnStartUp := 1);   // "FB22107_WP321_MUL_CALL"
END_REGION
END_FUNCTION

FUNCTION "FC22300_HOPPER_SYSTEM_ACTUATORS" : Void   // FC22300, LAD
TITLE = FC22300 HOPPER SYSTEM ACTUATORS
{ S7_Optimized_Access := 'TRUE' }
VERSION : 0.1
// stored: AutoNumber false, IsIECCheckEnabled false, SetENOAutomatically false, UDAEnableTagReadback false
BEGIN

REGION Network 1: //////////ACTUATORS HOPPERS UNIT 01//////////
END_REGION

REGION Network 2: CALL FB22301 TRANSFER POWDER VALVE HOPPER 1 UNIT 01
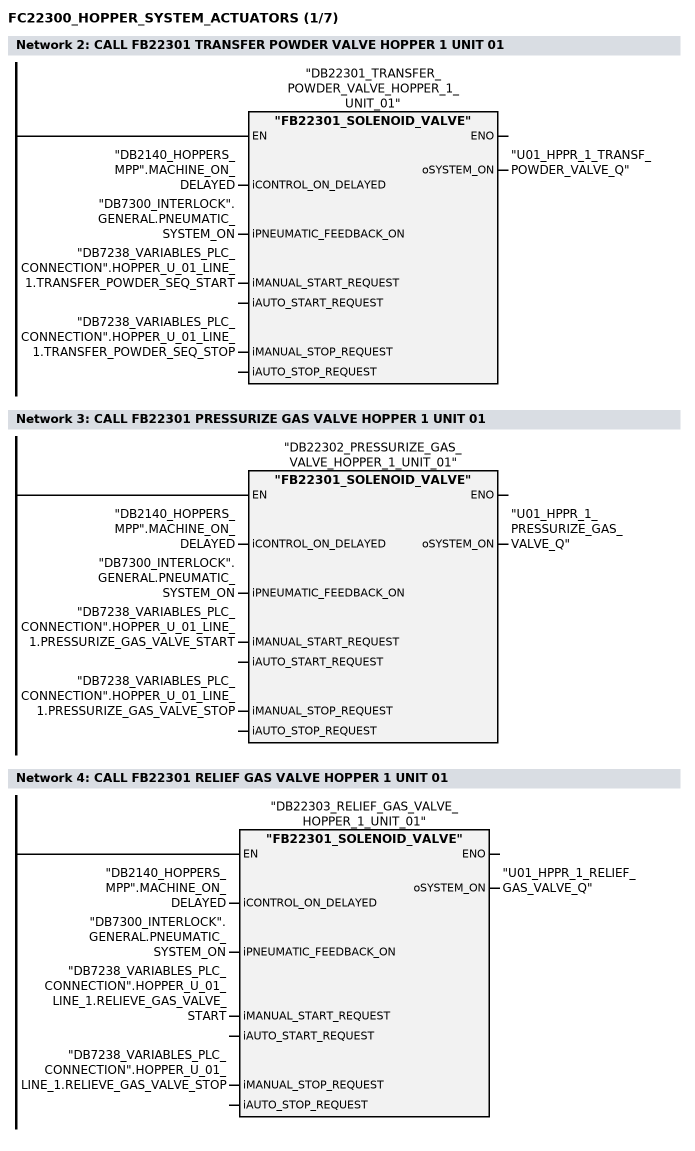
   RUNG wire#powerrail
      "DB22301_TRANSFER_POWDER_VALVE_HOPPER_1_UNIT_01"(iCONTROL_ON_DELAYED := "DB2140_HOPPERS_MPP".MACHINE_ON_DELAYED, iPNEUMATIC_FEEDBACK_ON := "DB7300_INTERLOCK".GENERAL.PNEUMATIC_SYSTEM_ON, iMANUAL_START_REQUEST := "DB7238_VARIABLES_PLC_CONNECTION".HOPPER_U_01_LINE_1.TRANSFER_POWDER_SEQ_START, iAUTO_START_REQUEST :=, iMANUAL_STOP_REQUEST := "DB7238_VARIABLES_PLC_CONNECTION".HOPPER_U_01_LINE_1.TRANSFER_POWDER_SEQ_STOP, iAUTO_STOP_REQUEST :=, oSYSTEM_ON => "U01_HPPR_1_TRANSF_POWDER_VALVE_Q")
   END_RUNG
   // the same network as SCL:
   "DB22301_TRANSFER_POWDER_VALVE_HOPPER_1_UNIT_01"(iCONTROL_ON_DELAYED := "DB2140_HOPPERS_MPP".MACHINE_ON_DELAYED,   // "FB22301_SOLENOID_VALVE"
                           iPNEUMATIC_FEEDBACK_ON := "DB7300_INTERLOCK".GENERAL.PNEUMATIC_SYSTEM_ON,
                           iMANUAL_START_REQUEST := "DB7238_VARIABLES_PLC_CONNECTION".HOPPER_U_01_LINE_1.TRANSFER_POWDER_SEQ_START,
                           iMANUAL_STOP_REQUEST := "DB7238_VARIABLES_PLC_CONNECTION".HOPPER_U_01_LINE_1.TRANSFER_POWDER_SEQ_STOP,
                           oSYSTEM_ON => "U01_HPPR_1_TRANSF_POWDER_VALVE_Q");
END_REGION

REGION Network 3: CALL FB22301 PRESSURIZE GAS VALVE HOPPER 1 UNIT 01
   RUNG wire#powerrail
      "DB22302_PRESSURIZE_GAS_VALVE_HOPPER_1_UNIT_01"(iCONTROL_ON_DELAYED := "DB2140_HOPPERS_MPP".MACHINE_ON_DELAYED, iPNEUMATIC_FEEDBACK_ON := "DB7300_INTERLOCK".GENERAL.PNEUMATIC_SYSTEM_ON, iMANUAL_START_REQUEST := "DB7238_VARIABLES_PLC_CONNECTION".HOPPER_U_01_LINE_1.PRESSURIZE_GAS_VALVE_START, iAUTO_START_REQUEST :=, iMANUAL_STOP_REQUEST := "DB7238_VARIABLES_PLC_CONNECTION".HOPPER_U_01_LINE_1.PRESSURIZE_GAS_VALVE_STOP, iAUTO_STOP_REQUEST :=, oSYSTEM_ON => "U01_HPPR_1_PRESSURIZE_GAS_VALVE_Q")
   END_RUNG
   // the same network as SCL:
   "DB22302_PRESSURIZE_GAS_VALVE_HOPPER_1_UNIT_01"(iCONTROL_ON_DELAYED := "DB2140_HOPPERS_MPP".MACHINE_ON_DELAYED,   // "FB22301_SOLENOID_VALVE"
                           iPNEUMATIC_FEEDBACK_ON := "DB7300_INTERLOCK".GENERAL.PNEUMATIC_SYSTEM_ON,
                           iMANUAL_START_REQUEST := "DB7238_VARIABLES_PLC_CONNECTION".HOPPER_U_01_LINE_1.PRESSURIZE_GAS_VALVE_START,
                           iMANUAL_STOP_REQUEST := "DB7238_VARIABLES_PLC_CONNECTION".HOPPER_U_01_LINE_1.PRESSURIZE_GAS_VALVE_STOP,
                           oSYSTEM_ON => "U01_HPPR_1_PRESSURIZE_GAS_VALVE_Q");
END_REGION

REGION Network 4: CALL FB22301 RELIEF GAS VALVE HOPPER 1 UNIT 01
   RUNG wire#powerrail
      "DB22303_RELIEF_GAS_VALVE_HOPPER_1_UNIT_01"(iCONTROL_ON_DELAYED := "DB2140_HOPPERS_MPP".MACHINE_ON_DELAYED, iPNEUMATIC_FEEDBACK_ON := "DB7300_INTERLOCK".GENERAL.PNEUMATIC_SYSTEM_ON, iMANUAL_START_REQUEST := "DB7238_VARIABLES_PLC_CONNECTION".HOPPER_U_01_LINE_1.RELIEVE_GAS_VALVE_START, iAUTO_START_REQUEST :=, iMANUAL_STOP_REQUEST := "DB7238_VARIABLES_PLC_CONNECTION".HOPPER_U_01_LINE_1.RELIEVE_GAS_VALVE_STOP, iAUTO_STOP_REQUEST :=, oSYSTEM_ON => "U01_HPPR_1_RELIEF_GAS_VALVE_Q")
   END_RUNG
   // the same network as SCL:
   "DB22303_RELIEF_GAS_VALVE_HOPPER_1_UNIT_01"(iCONTROL_ON_DELAYED := "DB2140_HOPPERS_MPP".MACHINE_ON_DELAYED,   // "FB22301_SOLENOID_VALVE"
                           iPNEUMATIC_FEEDBACK_ON := "DB7300_INTERLOCK".GENERAL.PNEUMATIC_SYSTEM_ON,
                           iMANUAL_START_REQUEST := "DB7238_VARIABLES_PLC_CONNECTION".HOPPER_U_01_LINE_1.RELIEVE_GAS_VALVE_START,
                           iMANUAL_STOP_REQUEST := "DB7238_VARIABLES_PLC_CONNECTION".HOPPER_U_01_LINE_1.RELIEVE_GAS_VALVE_STOP,
                           oSYSTEM_ON => "U01_HPPR_1_RELIEF_GAS_VALVE_Q");
END_REGION

REGION Network 5: CALL FB22301 CLEANING AIR VALVE HOPPER 1 UNIT 01
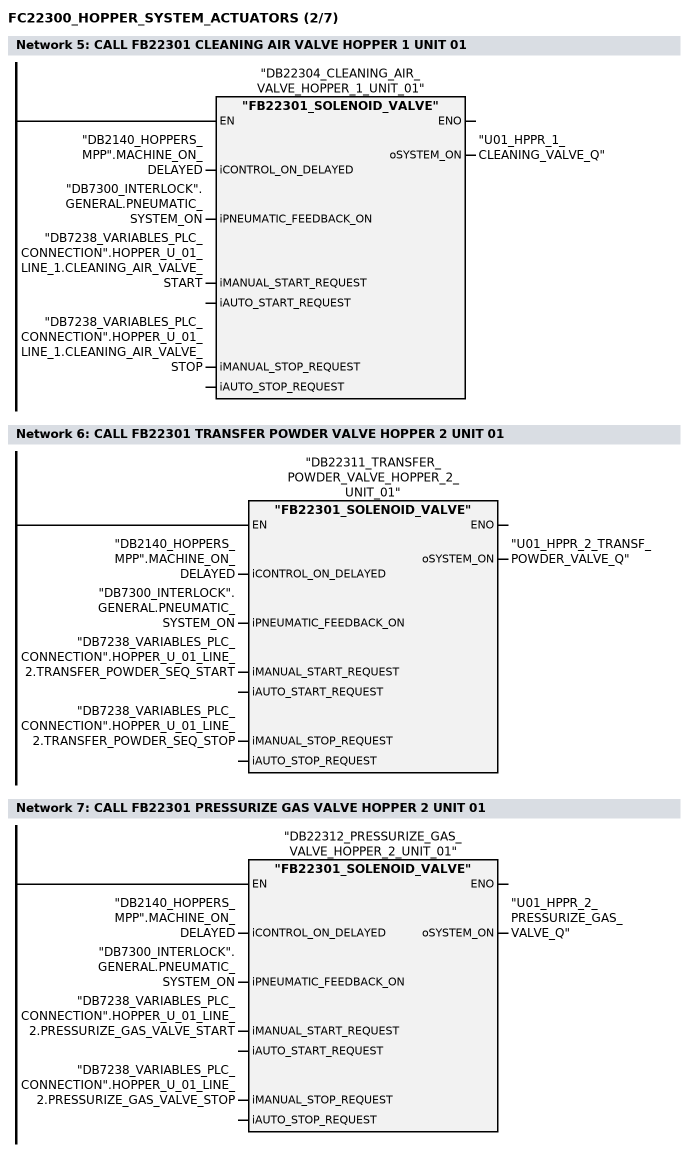
   RUNG wire#powerrail
      "DB22304_CLEANING_AIR_VALVE_HOPPER_1_UNIT_01"(iCONTROL_ON_DELAYED := "DB2140_HOPPERS_MPP".MACHINE_ON_DELAYED, iPNEUMATIC_FEEDBACK_ON := "DB7300_INTERLOCK".GENERAL.PNEUMATIC_SYSTEM_ON, iMANUAL_START_REQUEST := "DB7238_VARIABLES_PLC_CONNECTION".HOPPER_U_01_LINE_1.CLEANING_AIR_VALVE_START, iAUTO_START_REQUEST :=, iMANUAL_STOP_REQUEST := "DB7238_VARIABLES_PLC_CONNECTION".HOPPER_U_01_LINE_1.CLEANING_AIR_VALVE_STOP, iAUTO_STOP_REQUEST :=, oSYSTEM_ON => "U01_HPPR_1_CLEANING_VALVE_Q")
   END_RUNG
   // the same network as SCL:
   "DB22304_CLEANING_AIR_VALVE_HOPPER_1_UNIT_01"(iCONTROL_ON_DELAYED := "DB2140_HOPPERS_MPP".MACHINE_ON_DELAYED,   // "FB22301_SOLENOID_VALVE"
                           iPNEUMATIC_FEEDBACK_ON := "DB7300_INTERLOCK".GENERAL.PNEUMATIC_SYSTEM_ON,
                           iMANUAL_START_REQUEST := "DB7238_VARIABLES_PLC_CONNECTION".HOPPER_U_01_LINE_1.CLEANING_AIR_VALVE_START,
                           iMANUAL_STOP_REQUEST := "DB7238_VARIABLES_PLC_CONNECTION".HOPPER_U_01_LINE_1.CLEANING_AIR_VALVE_STOP,
                           oSYSTEM_ON => "U01_HPPR_1_CLEANING_VALVE_Q");
END_REGION

REGION Network 6: CALL FB22301 TRANSFER POWDER VALVE HOPPER 2 UNIT 01
   RUNG wire#powerrail
      "DB22311_TRANSFER_POWDER_VALVE_HOPPER_2_UNIT_01"(iCONTROL_ON_DELAYED := "DB2140_HOPPERS_MPP".MACHINE_ON_DELAYED, iPNEUMATIC_FEEDBACK_ON := "DB7300_INTERLOCK".GENERAL.PNEUMATIC_SYSTEM_ON, iMANUAL_START_REQUEST := "DB7238_VARIABLES_PLC_CONNECTION".HOPPER_U_01_LINE_2.TRANSFER_POWDER_SEQ_START, iAUTO_START_REQUEST :=, iMANUAL_STOP_REQUEST := "DB7238_VARIABLES_PLC_CONNECTION".HOPPER_U_01_LINE_2.TRANSFER_POWDER_SEQ_STOP, iAUTO_STOP_REQUEST :=, oSYSTEM_ON => "U01_HPPR_2_TRANSF_POWDER_VALVE_Q")
   END_RUNG
   // the same network as SCL:
   "DB22311_TRANSFER_POWDER_VALVE_HOPPER_2_UNIT_01"(iCONTROL_ON_DELAYED := "DB2140_HOPPERS_MPP".MACHINE_ON_DELAYED,   // "FB22301_SOLENOID_VALVE"
                           iPNEUMATIC_FEEDBACK_ON := "DB7300_INTERLOCK".GENERAL.PNEUMATIC_SYSTEM_ON,
                           iMANUAL_START_REQUEST := "DB7238_VARIABLES_PLC_CONNECTION".HOPPER_U_01_LINE_2.TRANSFER_POWDER_SEQ_START,
                           iMANUAL_STOP_REQUEST := "DB7238_VARIABLES_PLC_CONNECTION".HOPPER_U_01_LINE_2.TRANSFER_POWDER_SEQ_STOP,
                           oSYSTEM_ON => "U01_HPPR_2_TRANSF_POWDER_VALVE_Q");
END_REGION

REGION Network 7: CALL FB22301 PRESSURIZE GAS VALVE HOPPER 2 UNIT 01
   RUNG wire#powerrail
      "DB22312_PRESSURIZE_GAS_VALVE_HOPPER_2_UNIT_01"(iCONTROL_ON_DELAYED := "DB2140_HOPPERS_MPP".MACHINE_ON_DELAYED, iPNEUMATIC_FEEDBACK_ON := "DB7300_INTERLOCK".GENERAL.PNEUMATIC_SYSTEM_ON, iMANUAL_START_REQUEST := "DB7238_VARIABLES_PLC_CONNECTION".HOPPER_U_01_LINE_2.PRESSURIZE_GAS_VALVE_START, iAUTO_START_REQUEST :=, iMANUAL_STOP_REQUEST := "DB7238_VARIABLES_PLC_CONNECTION".HOPPER_U_01_LINE_2.PRESSURIZE_GAS_VALVE_STOP, iAUTO_STOP_REQUEST :=, oSYSTEM_ON => "U01_HPPR_2_PRESSURIZE_GAS_VALVE_Q")
   END_RUNG
   // the same network as SCL:
   "DB22312_PRESSURIZE_GAS_VALVE_HOPPER_2_UNIT_01"(iCONTROL_ON_DELAYED := "DB2140_HOPPERS_MPP".MACHINE_ON_DELAYED,   // "FB22301_SOLENOID_VALVE"
                           iPNEUMATIC_FEEDBACK_ON := "DB7300_INTERLOCK".GENERAL.PNEUMATIC_SYSTEM_ON,
                           iMANUAL_START_REQUEST := "DB7238_VARIABLES_PLC_CONNECTION".HOPPER_U_01_LINE_2.PRESSURIZE_GAS_VALVE_START,
                           iMANUAL_STOP_REQUEST := "DB7238_VARIABLES_PLC_CONNECTION".HOPPER_U_01_LINE_2.PRESSURIZE_GAS_VALVE_STOP,
                           oSYSTEM_ON => "U01_HPPR_2_PRESSURIZE_GAS_VALVE_Q");
END_REGION

REGION Network 8: CALL FB22301 RELIEF GAS VALVE HOPPER 2 UNIT 01
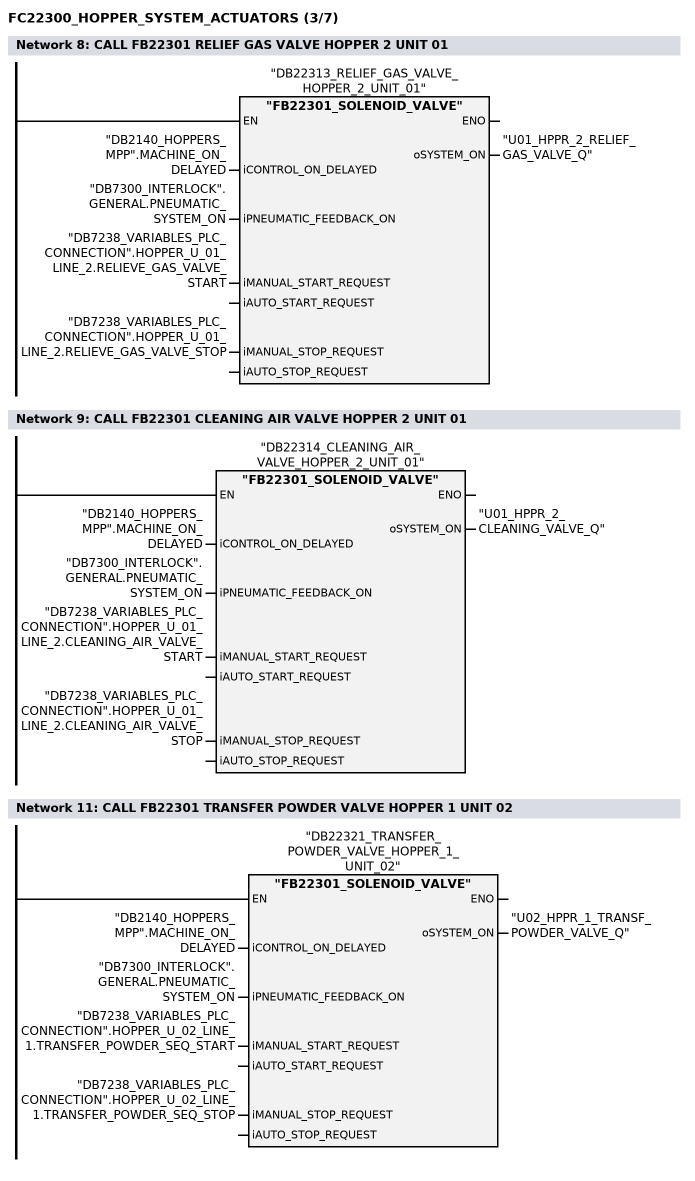
   RUNG wire#powerrail
      "DB22313_RELIEF_GAS_VALVE_HOPPER_2_UNIT_01"(iCONTROL_ON_DELAYED := "DB2140_HOPPERS_MPP".MACHINE_ON_DELAYED, iPNEUMATIC_FEEDBACK_ON := "DB7300_INTERLOCK".GENERAL.PNEUMATIC_SYSTEM_ON, iMANUAL_START_REQUEST := "DB7238_VARIABLES_PLC_CONNECTION".HOPPER_U_01_LINE_2.RELIEVE_GAS_VALVE_START, iAUTO_START_REQUEST :=, iMANUAL_STOP_REQUEST := "DB7238_VARIABLES_PLC_CONNECTION".HOPPER_U_01_LINE_2.RELIEVE_GAS_VALVE_STOP, iAUTO_STOP_REQUEST :=, oSYSTEM_ON => "U01_HPPR_2_RELIEF_GAS_VALVE_Q")
   END_RUNG
   // the same network as SCL:
   "DB22313_RELIEF_GAS_VALVE_HOPPER_2_UNIT_01"(iCONTROL_ON_DELAYED := "DB2140_HOPPERS_MPP".MACHINE_ON_DELAYED,   // "FB22301_SOLENOID_VALVE"
                           iPNEUMATIC_FEEDBACK_ON := "DB7300_INTERLOCK".GENERAL.PNEUMATIC_SYSTEM_ON,
                           iMANUAL_START_REQUEST := "DB7238_VARIABLES_PLC_CONNECTION".HOPPER_U_01_LINE_2.RELIEVE_GAS_VALVE_START,
                           iMANUAL_STOP_REQUEST := "DB7238_VARIABLES_PLC_CONNECTION".HOPPER_U_01_LINE_2.RELIEVE_GAS_VALVE_STOP,
                           oSYSTEM_ON => "U01_HPPR_2_RELIEF_GAS_VALVE_Q");
END_REGION

REGION Network 9: CALL FB22301 CLEANING AIR VALVE HOPPER 2 UNIT 01
   RUNG wire#powerrail
      "DB22314_CLEANING_AIR_VALVE_HOPPER_2_UNIT_01"(iCONTROL_ON_DELAYED := "DB2140_HOPPERS_MPP".MACHINE_ON_DELAYED, iPNEUMATIC_FEEDBACK_ON := "DB7300_INTERLOCK".GENERAL.PNEUMATIC_SYSTEM_ON, iMANUAL_START_REQUEST := "DB7238_VARIABLES_PLC_CONNECTION".HOPPER_U_01_LINE_2.CLEANING_AIR_VALVE_START, iAUTO_START_REQUEST :=, iMANUAL_STOP_REQUEST := "DB7238_VARIABLES_PLC_CONNECTION".HOPPER_U_01_LINE_2.CLEANING_AIR_VALVE_STOP, iAUTO_STOP_REQUEST :=, oSYSTEM_ON => "U01_HPPR_2_CLEANING_VALVE_Q")
   END_RUNG
   // the same network as SCL:
   "DB22314_CLEANING_AIR_VALVE_HOPPER_2_UNIT_01"(iCONTROL_ON_DELAYED := "DB2140_HOPPERS_MPP".MACHINE_ON_DELAYED,   // "FB22301_SOLENOID_VALVE"
                           iPNEUMATIC_FEEDBACK_ON := "DB7300_INTERLOCK".GENERAL.PNEUMATIC_SYSTEM_ON,
                           iMANUAL_START_REQUEST := "DB7238_VARIABLES_PLC_CONNECTION".HOPPER_U_01_LINE_2.CLEANING_AIR_VALVE_START,
                           iMANUAL_STOP_REQUEST := "DB7238_VARIABLES_PLC_CONNECTION".HOPPER_U_01_LINE_2.CLEANING_AIR_VALVE_STOP,
                           oSYSTEM_ON => "U01_HPPR_2_CLEANING_VALVE_Q");
END_REGION

REGION Network 10: //////////ACTUATORS HOPPERS UNIT 02//////////
END_REGION

REGION Network 11: CALL FB22301 TRANSFER POWDER VALVE HOPPER 1 UNIT 02
   RUNG wire#powerrail
      "DB22321_TRANSFER_POWDER_VALVE_HOPPER_1_UNIT_02"(iCONTROL_ON_DELAYED := "DB2140_HOPPERS_MPP".MACHINE_ON_DELAYED, iPNEUMATIC_FEEDBACK_ON := "DB7300_INTERLOCK".GENERAL.PNEUMATIC_SYSTEM_ON, iMANUAL_START_REQUEST := "DB7238_VARIABLES_PLC_CONNECTION".HOPPER_U_02_LINE_1.TRANSFER_POWDER_SEQ_START, iAUTO_START_REQUEST :=, iMANUAL_STOP_REQUEST := "DB7238_VARIABLES_PLC_CONNECTION".HOPPER_U_02_LINE_1.TRANSFER_POWDER_SEQ_STOP, iAUTO_STOP_REQUEST :=, oSYSTEM_ON => "U02_HPPR_1_TRANSF_POWDER_VALVE_Q")
   END_RUNG
   // the same network as SCL:
   "DB22321_TRANSFER_POWDER_VALVE_HOPPER_1_UNIT_02"(iCONTROL_ON_DELAYED := "DB2140_HOPPERS_MPP".MACHINE_ON_DELAYED,   // "FB22301_SOLENOID_VALVE"
                           iPNEUMATIC_FEEDBACK_ON := "DB7300_INTERLOCK".GENERAL.PNEUMATIC_SYSTEM_ON,
                           iMANUAL_START_REQUEST := "DB7238_VARIABLES_PLC_CONNECTION".HOPPER_U_02_LINE_1.TRANSFER_POWDER_SEQ_START,
                           iMANUAL_STOP_REQUEST := "DB7238_VARIABLES_PLC_CONNECTION".HOPPER_U_02_LINE_1.TRANSFER_POWDER_SEQ_STOP,
                           oSYSTEM_ON => "U02_HPPR_1_TRANSF_POWDER_VALVE_Q");
END_REGION

REGION Network 12: CALL FB22301 PRESSURIZE GAS VALVE HOPPER 1 UNIT 02
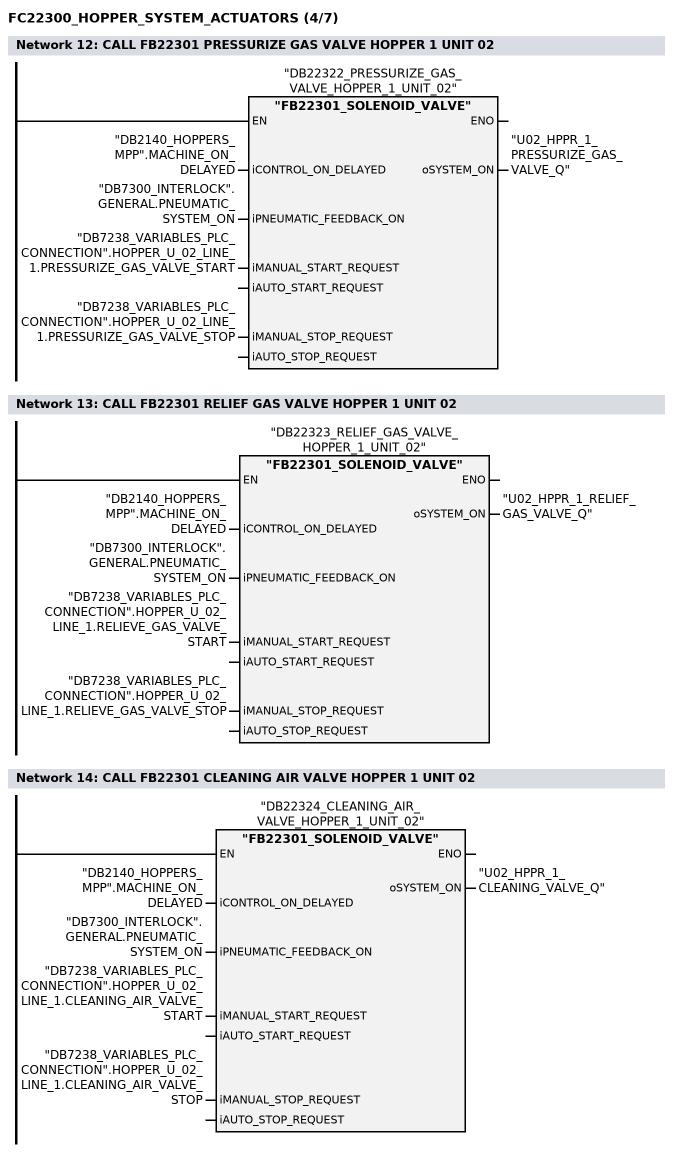
   RUNG wire#powerrail
      "DB22322_PRESSURIZE_GAS_VALVE_HOPPER_1_UNIT_02"(iCONTROL_ON_DELAYED := "DB2140_HOPPERS_MPP".MACHINE_ON_DELAYED, iPNEUMATIC_FEEDBACK_ON := "DB7300_INTERLOCK".GENERAL.PNEUMATIC_SYSTEM_ON, iMANUAL_START_REQUEST := "DB7238_VARIABLES_PLC_CONNECTION".HOPPER_U_02_LINE_1.PRESSURIZE_GAS_VALVE_START, iAUTO_START_REQUEST :=, iMANUAL_STOP_REQUEST := "DB7238_VARIABLES_PLC_CONNECTION".HOPPER_U_02_LINE_1.PRESSURIZE_GAS_VALVE_STOP, iAUTO_STOP_REQUEST :=, oSYSTEM_ON => "U02_HPPR_1_PRESSURIZE_GAS_VALVE_Q")
   END_RUNG
   // the same network as SCL:
   "DB22322_PRESSURIZE_GAS_VALVE_HOPPER_1_UNIT_02"(iCONTROL_ON_DELAYED := "DB2140_HOPPERS_MPP".MACHINE_ON_DELAYED,   // "FB22301_SOLENOID_VALVE"
                           iPNEUMATIC_FEEDBACK_ON := "DB7300_INTERLOCK".GENERAL.PNEUMATIC_SYSTEM_ON,
                           iMANUAL_START_REQUEST := "DB7238_VARIABLES_PLC_CONNECTION".HOPPER_U_02_LINE_1.PRESSURIZE_GAS_VALVE_START,
                           iMANUAL_STOP_REQUEST := "DB7238_VARIABLES_PLC_CONNECTION".HOPPER_U_02_LINE_1.PRESSURIZE_GAS_VALVE_STOP,
                           oSYSTEM_ON => "U02_HPPR_1_PRESSURIZE_GAS_VALVE_Q");
END_REGION

REGION Network 13: CALL FB22301 RELIEF GAS VALVE HOPPER 1 UNIT 02
   RUNG wire#powerrail
      "DB22323_RELIEF_GAS_VALVE_HOPPER_1_UNIT_02"(iCONTROL_ON_DELAYED := "DB2140_HOPPERS_MPP".MACHINE_ON_DELAYED, iPNEUMATIC_FEEDBACK_ON := "DB7300_INTERLOCK".GENERAL.PNEUMATIC_SYSTEM_ON, iMANUAL_START_REQUEST := "DB7238_VARIABLES_PLC_CONNECTION".HOPPER_U_02_LINE_1.RELIEVE_GAS_VALVE_START, iAUTO_START_REQUEST :=, iMANUAL_STOP_REQUEST := "DB7238_VARIABLES_PLC_CONNECTION".HOPPER_U_02_LINE_1.RELIEVE_GAS_VALVE_STOP, iAUTO_STOP_REQUEST :=, oSYSTEM_ON => "U02_HPPR_1_RELIEF_GAS_VALVE_Q")
   END_RUNG
   // the same network as SCL:
   "DB22323_RELIEF_GAS_VALVE_HOPPER_1_UNIT_02"(iCONTROL_ON_DELAYED := "DB2140_HOPPERS_MPP".MACHINE_ON_DELAYED,   // "FB22301_SOLENOID_VALVE"
                           iPNEUMATIC_FEEDBACK_ON := "DB7300_INTERLOCK".GENERAL.PNEUMATIC_SYSTEM_ON,
                           iMANUAL_START_REQUEST := "DB7238_VARIABLES_PLC_CONNECTION".HOPPER_U_02_LINE_1.RELIEVE_GAS_VALVE_START,
                           iMANUAL_STOP_REQUEST := "DB7238_VARIABLES_PLC_CONNECTION".HOPPER_U_02_LINE_1.RELIEVE_GAS_VALVE_STOP,
                           oSYSTEM_ON => "U02_HPPR_1_RELIEF_GAS_VALVE_Q");
END_REGION

REGION Network 14: CALL FB22301 CLEANING AIR VALVE HOPPER 1 UNIT 02
   RUNG wire#powerrail
      "DB22324_CLEANING_AIR_VALVE_HOPPER_1_UNIT_02"(iCONTROL_ON_DELAYED := "DB2140_HOPPERS_MPP".MACHINE_ON_DELAYED, iPNEUMATIC_FEEDBACK_ON := "DB7300_INTERLOCK".GENERAL.PNEUMATIC_SYSTEM_ON, iMANUAL_START_REQUEST := "DB7238_VARIABLES_PLC_CONNECTION".HOPPER_U_02_LINE_1.CLEANING_AIR_VALVE_START, iAUTO_START_REQUEST :=, iMANUAL_STOP_REQUEST := "DB7238_VARIABLES_PLC_CONNECTION".HOPPER_U_02_LINE_1.CLEANING_AIR_VALVE_STOP, iAUTO_STOP_REQUEST :=, oSYSTEM_ON => "U02_HPPR_1_CLEANING_VALVE_Q")
   END_RUNG
   // the same network as SCL:
   "DB22324_CLEANING_AIR_VALVE_HOPPER_1_UNIT_02"(iCONTROL_ON_DELAYED := "DB2140_HOPPERS_MPP".MACHINE_ON_DELAYED,   // "FB22301_SOLENOID_VALVE"
                           iPNEUMATIC_FEEDBACK_ON := "DB7300_INTERLOCK".GENERAL.PNEUMATIC_SYSTEM_ON,
                           iMANUAL_START_REQUEST := "DB7238_VARIABLES_PLC_CONNECTION".HOPPER_U_02_LINE_1.CLEANING_AIR_VALVE_START,
                           iMANUAL_STOP_REQUEST := "DB7238_VARIABLES_PLC_CONNECTION".HOPPER_U_02_LINE_1.CLEANING_AIR_VALVE_STOP,
                           oSYSTEM_ON => "U02_HPPR_1_CLEANING_VALVE_Q");
END_REGION

REGION Network 15: CALL FB22301 TRANSFER POWDER VALVE HOPPER 2 UNIT 02
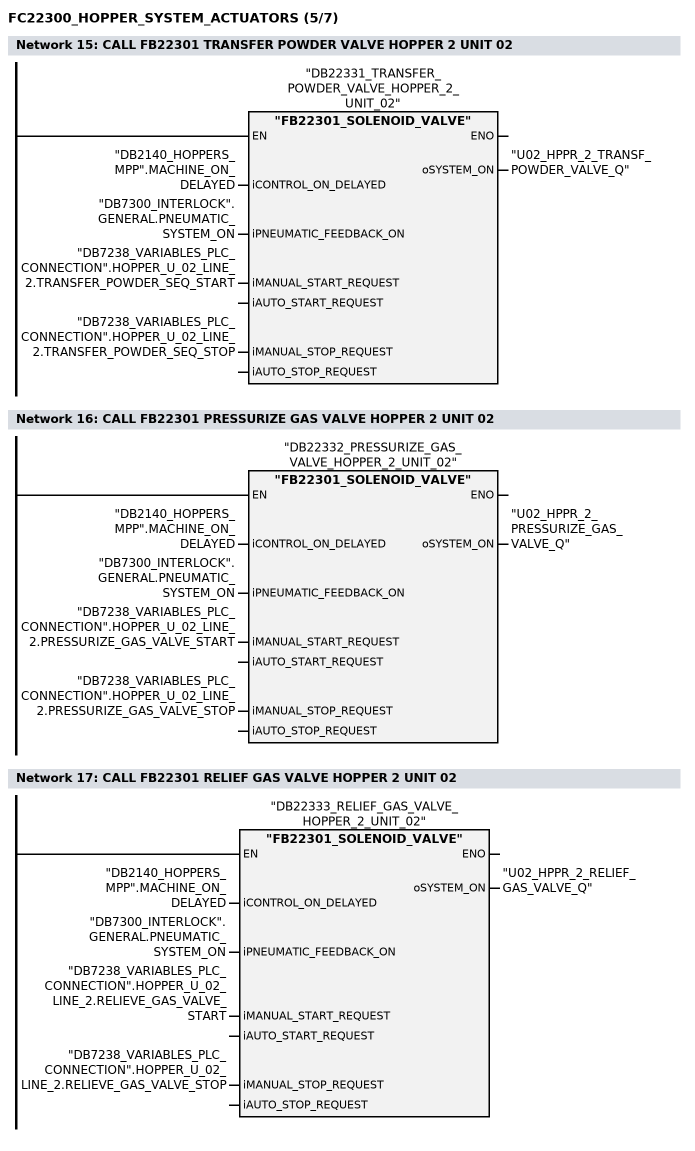
   RUNG wire#powerrail
      "DB22331_TRANSFER_POWDER_VALVE_HOPPER_2_UNIT_02"(iCONTROL_ON_DELAYED := "DB2140_HOPPERS_MPP".MACHINE_ON_DELAYED, iPNEUMATIC_FEEDBACK_ON := "DB7300_INTERLOCK".GENERAL.PNEUMATIC_SYSTEM_ON, iMANUAL_START_REQUEST := "DB7238_VARIABLES_PLC_CONNECTION".HOPPER_U_02_LINE_2.TRANSFER_POWDER_SEQ_START, iAUTO_START_REQUEST :=, iMANUAL_STOP_REQUEST := "DB7238_VARIABLES_PLC_CONNECTION".HOPPER_U_02_LINE_2.TRANSFER_POWDER_SEQ_STOP, iAUTO_STOP_REQUEST :=, oSYSTEM_ON => "U02_HPPR_2_TRANSF_POWDER_VALVE_Q")
   END_RUNG
   // the same network as SCL:
   "DB22331_TRANSFER_POWDER_VALVE_HOPPER_2_UNIT_02"(iCONTROL_ON_DELAYED := "DB2140_HOPPERS_MPP".MACHINE_ON_DELAYED,   // "FB22301_SOLENOID_VALVE"
                           iPNEUMATIC_FEEDBACK_ON := "DB7300_INTERLOCK".GENERAL.PNEUMATIC_SYSTEM_ON,
                           iMANUAL_START_REQUEST := "DB7238_VARIABLES_PLC_CONNECTION".HOPPER_U_02_LINE_2.TRANSFER_POWDER_SEQ_START,
                           iMANUAL_STOP_REQUEST := "DB7238_VARIABLES_PLC_CONNECTION".HOPPER_U_02_LINE_2.TRANSFER_POWDER_SEQ_STOP,
                           oSYSTEM_ON => "U02_HPPR_2_TRANSF_POWDER_VALVE_Q");
END_REGION

REGION Network 16: CALL FB22301 PRESSURIZE GAS VALVE HOPPER 2 UNIT 02
   RUNG wire#powerrail
      "DB22332_PRESSURIZE_GAS_VALVE_HOPPER_2_UNIT_02"(iCONTROL_ON_DELAYED := "DB2140_HOPPERS_MPP".MACHINE_ON_DELAYED, iPNEUMATIC_FEEDBACK_ON := "DB7300_INTERLOCK".GENERAL.PNEUMATIC_SYSTEM_ON, iMANUAL_START_REQUEST := "DB7238_VARIABLES_PLC_CONNECTION".HOPPER_U_02_LINE_2.PRESSURIZE_GAS_VALVE_START, iAUTO_START_REQUEST :=, iMANUAL_STOP_REQUEST := "DB7238_VARIABLES_PLC_CONNECTION".HOPPER_U_02_LINE_2.PRESSURIZE_GAS_VALVE_STOP, iAUTO_STOP_REQUEST :=, oSYSTEM_ON => "U02_HPPR_2_PRESSURIZE_GAS_VALVE_Q")
   END_RUNG
   // the same network as SCL:
   "DB22332_PRESSURIZE_GAS_VALVE_HOPPER_2_UNIT_02"(iCONTROL_ON_DELAYED := "DB2140_HOPPERS_MPP".MACHINE_ON_DELAYED,   // "FB22301_SOLENOID_VALVE"
                           iPNEUMATIC_FEEDBACK_ON := "DB7300_INTERLOCK".GENERAL.PNEUMATIC_SYSTEM_ON,
                           iMANUAL_START_REQUEST := "DB7238_VARIABLES_PLC_CONNECTION".HOPPER_U_02_LINE_2.PRESSURIZE_GAS_VALVE_START,
                           iMANUAL_STOP_REQUEST := "DB7238_VARIABLES_PLC_CONNECTION".HOPPER_U_02_LINE_2.PRESSURIZE_GAS_VALVE_STOP,
                           oSYSTEM_ON => "U02_HPPR_2_PRESSURIZE_GAS_VALVE_Q");
END_REGION

REGION Network 17: CALL FB22301 RELIEF GAS VALVE HOPPER 2 UNIT 02
   RUNG wire#powerrail
      "DB22333_RELIEF_GAS_VALVE_HOPPER_2_UNIT_02"(iCONTROL_ON_DELAYED := "DB2140_HOPPERS_MPP".MACHINE_ON_DELAYED, iPNEUMATIC_FEEDBACK_ON := "DB7300_INTERLOCK".GENERAL.PNEUMATIC_SYSTEM_ON, iMANUAL_START_REQUEST := "DB7238_VARIABLES_PLC_CONNECTION".HOPPER_U_02_LINE_2.RELIEVE_GAS_VALVE_START, iAUTO_START_REQUEST :=, iMANUAL_STOP_REQUEST := "DB7238_VARIABLES_PLC_CONNECTION".HOPPER_U_02_LINE_2.RELIEVE_GAS_VALVE_STOP, iAUTO_STOP_REQUEST :=, oSYSTEM_ON => "U02_HPPR_2_RELIEF_GAS_VALVE_Q")
   END_RUNG
   // the same network as SCL:
   "DB22333_RELIEF_GAS_VALVE_HOPPER_2_UNIT_02"(iCONTROL_ON_DELAYED := "DB2140_HOPPERS_MPP".MACHINE_ON_DELAYED,   // "FB22301_SOLENOID_VALVE"
                           iPNEUMATIC_FEEDBACK_ON := "DB7300_INTERLOCK".GENERAL.PNEUMATIC_SYSTEM_ON,
                           iMANUAL_START_REQUEST := "DB7238_VARIABLES_PLC_CONNECTION".HOPPER_U_02_LINE_2.RELIEVE_GAS_VALVE_START,
                           iMANUAL_STOP_REQUEST := "DB7238_VARIABLES_PLC_CONNECTION".HOPPER_U_02_LINE_2.RELIEVE_GAS_VALVE_STOP,
                           oSYSTEM_ON => "U02_HPPR_2_RELIEF_GAS_VALVE_Q");
END_REGION

REGION Network 18: CALL FB22301 CLEANING AIR VALVE HOPPER 2 UNIT 02
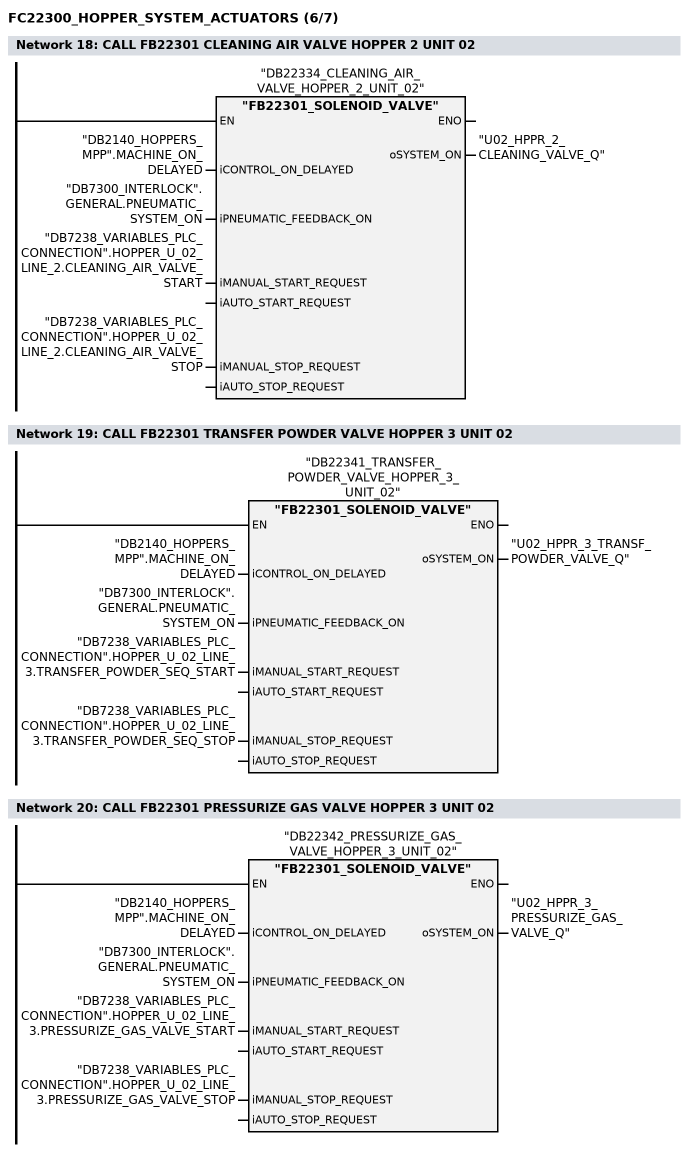
   RUNG wire#powerrail
      "DB22334_CLEANING_AIR_VALVE_HOPPER_2_UNIT_02"(iCONTROL_ON_DELAYED := "DB2140_HOPPERS_MPP".MACHINE_ON_DELAYED, iPNEUMATIC_FEEDBACK_ON := "DB7300_INTERLOCK".GENERAL.PNEUMATIC_SYSTEM_ON, iMANUAL_START_REQUEST := "DB7238_VARIABLES_PLC_CONNECTION".HOPPER_U_02_LINE_2.CLEANING_AIR_VALVE_START, iAUTO_START_REQUEST :=, iMANUAL_STOP_REQUEST := "DB7238_VARIABLES_PLC_CONNECTION".HOPPER_U_02_LINE_2.CLEANING_AIR_VALVE_STOP, iAUTO_STOP_REQUEST :=, oSYSTEM_ON => "U02_HPPR_2_CLEANING_VALVE_Q")
   END_RUNG
   // the same network as SCL:
   "DB22334_CLEANING_AIR_VALVE_HOPPER_2_UNIT_02"(iCONTROL_ON_DELAYED := "DB2140_HOPPERS_MPP".MACHINE_ON_DELAYED,   // "FB22301_SOLENOID_VALVE"
                           iPNEUMATIC_FEEDBACK_ON := "DB7300_INTERLOCK".GENERAL.PNEUMATIC_SYSTEM_ON,
                           iMANUAL_START_REQUEST := "DB7238_VARIABLES_PLC_CONNECTION".HOPPER_U_02_LINE_2.CLEANING_AIR_VALVE_START,
                           iMANUAL_STOP_REQUEST := "DB7238_VARIABLES_PLC_CONNECTION".HOPPER_U_02_LINE_2.CLEANING_AIR_VALVE_STOP,
                           oSYSTEM_ON => "U02_HPPR_2_CLEANING_VALVE_Q");
END_REGION

REGION Network 19: CALL FB22301 TRANSFER POWDER VALVE HOPPER 3 UNIT 02
   RUNG wire#powerrail
      "DB22341_TRANSFER_POWDER_VALVE_HOPPER_3_UNIT_02"(iCONTROL_ON_DELAYED := "DB2140_HOPPERS_MPP".MACHINE_ON_DELAYED, iPNEUMATIC_FEEDBACK_ON := "DB7300_INTERLOCK".GENERAL.PNEUMATIC_SYSTEM_ON, iMANUAL_START_REQUEST := "DB7238_VARIABLES_PLC_CONNECTION".HOPPER_U_02_LINE_3.TRANSFER_POWDER_SEQ_START, iAUTO_START_REQUEST :=, iMANUAL_STOP_REQUEST := "DB7238_VARIABLES_PLC_CONNECTION".HOPPER_U_02_LINE_3.TRANSFER_POWDER_SEQ_STOP, iAUTO_STOP_REQUEST :=, oSYSTEM_ON => "U02_HPPR_3_TRANSF_POWDER_VALVE_Q")
   END_RUNG
   // the same network as SCL:
   "DB22341_TRANSFER_POWDER_VALVE_HOPPER_3_UNIT_02"(iCONTROL_ON_DELAYED := "DB2140_HOPPERS_MPP".MACHINE_ON_DELAYED,   // "FB22301_SOLENOID_VALVE"
                           iPNEUMATIC_FEEDBACK_ON := "DB7300_INTERLOCK".GENERAL.PNEUMATIC_SYSTEM_ON,
                           iMANUAL_START_REQUEST := "DB7238_VARIABLES_PLC_CONNECTION".HOPPER_U_02_LINE_3.TRANSFER_POWDER_SEQ_START,
                           iMANUAL_STOP_REQUEST := "DB7238_VARIABLES_PLC_CONNECTION".HOPPER_U_02_LINE_3.TRANSFER_POWDER_SEQ_STOP,
                           oSYSTEM_ON => "U02_HPPR_3_TRANSF_POWDER_VALVE_Q");
END_REGION

REGION Network 20: CALL FB22301 PRESSURIZE GAS VALVE HOPPER 3 UNIT 02
   RUNG wire#powerrail
      "DB22342_PRESSURIZE_GAS_VALVE_HOPPER_3_UNIT_02"(iCONTROL_ON_DELAYED := "DB2140_HOPPERS_MPP".MACHINE_ON_DELAYED, iPNEUMATIC_FEEDBACK_ON := "DB7300_INTERLOCK".GENERAL.PNEUMATIC_SYSTEM_ON, iMANUAL_START_REQUEST := "DB7238_VARIABLES_PLC_CONNECTION".HOPPER_U_02_LINE_3.PRESSURIZE_GAS_VALVE_START, iAUTO_START_REQUEST :=, iMANUAL_STOP_REQUEST := "DB7238_VARIABLES_PLC_CONNECTION".HOPPER_U_02_LINE_3.PRESSURIZE_GAS_VALVE_STOP, iAUTO_STOP_REQUEST :=, oSYSTEM_ON => "U02_HPPR_3_PRESSURIZE_GAS_VALVE_Q")
   END_RUNG
   // the same network as SCL:
   "DB22342_PRESSURIZE_GAS_VALVE_HOPPER_3_UNIT_02"(iCONTROL_ON_DELAYED := "DB2140_HOPPERS_MPP".MACHINE_ON_DELAYED,   // "FB22301_SOLENOID_VALVE"
                           iPNEUMATIC_FEEDBACK_ON := "DB7300_INTERLOCK".GENERAL.PNEUMATIC_SYSTEM_ON,
                           iMANUAL_START_REQUEST := "DB7238_VARIABLES_PLC_CONNECTION".HOPPER_U_02_LINE_3.PRESSURIZE_GAS_VALVE_START,
                           iMANUAL_STOP_REQUEST := "DB7238_VARIABLES_PLC_CONNECTION".HOPPER_U_02_LINE_3.PRESSURIZE_GAS_VALVE_STOP,
                           oSYSTEM_ON => "U02_HPPR_3_PRESSURIZE_GAS_VALVE_Q");
END_REGION

REGION Network 21: CALL FB22301 RELIEF GAS VALVE HOPPER 3 UNIT 02
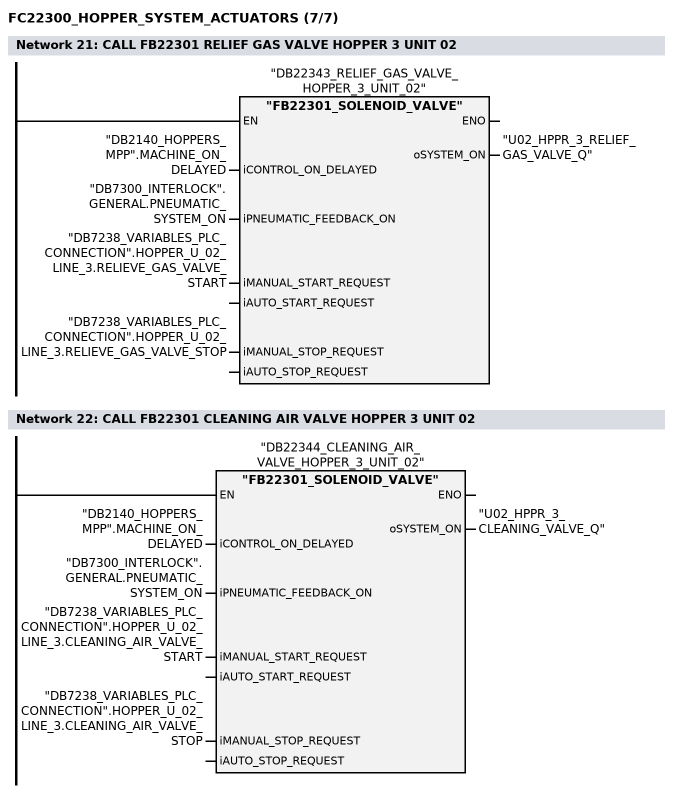
   RUNG wire#powerrail
      "DB22343_RELIEF_GAS_VALVE_HOPPER_3_UNIT_02"(iCONTROL_ON_DELAYED := "DB2140_HOPPERS_MPP".MACHINE_ON_DELAYED, iPNEUMATIC_FEEDBACK_ON := "DB7300_INTERLOCK".GENERAL.PNEUMATIC_SYSTEM_ON, iMANUAL_START_REQUEST := "DB7238_VARIABLES_PLC_CONNECTION".HOPPER_U_02_LINE_3.RELIEVE_GAS_VALVE_START, iAUTO_START_REQUEST :=, iMANUAL_STOP_REQUEST := "DB7238_VARIABLES_PLC_CONNECTION".HOPPER_U_02_LINE_3.RELIEVE_GAS_VALVE_STOP, iAUTO_STOP_REQUEST :=, oSYSTEM_ON => "U02_HPPR_3_RELIEF_GAS_VALVE_Q")
   END_RUNG
   // the same network as SCL:
   "DB22343_RELIEF_GAS_VALVE_HOPPER_3_UNIT_02"(iCONTROL_ON_DELAYED := "DB2140_HOPPERS_MPP".MACHINE_ON_DELAYED,   // "FB22301_SOLENOID_VALVE"
                           iPNEUMATIC_FEEDBACK_ON := "DB7300_INTERLOCK".GENERAL.PNEUMATIC_SYSTEM_ON,
                           iMANUAL_START_REQUEST := "DB7238_VARIABLES_PLC_CONNECTION".HOPPER_U_02_LINE_3.RELIEVE_GAS_VALVE_START,
                           iMANUAL_STOP_REQUEST := "DB7238_VARIABLES_PLC_CONNECTION".HOPPER_U_02_LINE_3.RELIEVE_GAS_VALVE_STOP,
                           oSYSTEM_ON => "U02_HPPR_3_RELIEF_GAS_VALVE_Q");
END_REGION

REGION Network 22: CALL FB22301 CLEANING AIR VALVE HOPPER 3 UNIT 02
   RUNG wire#powerrail
      "DB22344_CLEANING_AIR_VALVE_HOPPER_3_UNIT_02"(iCONTROL_ON_DELAYED := "DB2140_HOPPERS_MPP".MACHINE_ON_DELAYED, iPNEUMATIC_FEEDBACK_ON := "DB7300_INTERLOCK".GENERAL.PNEUMATIC_SYSTEM_ON, iMANUAL_START_REQUEST := "DB7238_VARIABLES_PLC_CONNECTION".HOPPER_U_02_LINE_3.CLEANING_AIR_VALVE_START, iAUTO_START_REQUEST :=, iMANUAL_STOP_REQUEST := "DB7238_VARIABLES_PLC_CONNECTION".HOPPER_U_02_LINE_3.CLEANING_AIR_VALVE_STOP, iAUTO_STOP_REQUEST :=, oSYSTEM_ON => "U02_HPPR_3_CLEANING_VALVE_Q")
   END_RUNG
   // the same network as SCL:
   "DB22344_CLEANING_AIR_VALVE_HOPPER_3_UNIT_02"(iCONTROL_ON_DELAYED := "DB2140_HOPPERS_MPP".MACHINE_ON_DELAYED,   // "FB22301_SOLENOID_VALVE"
                           iPNEUMATIC_FEEDBACK_ON := "DB7300_INTERLOCK".GENERAL.PNEUMATIC_SYSTEM_ON,
                           iMANUAL_START_REQUEST := "DB7238_VARIABLES_PLC_CONNECTION".HOPPER_U_02_LINE_3.CLEANING_AIR_VALVE_START,
                           iMANUAL_STOP_REQUEST := "DB7238_VARIABLES_PLC_CONNECTION".HOPPER_U_02_LINE_3.CLEANING_AIR_VALVE_STOP,
                           oSYSTEM_ON => "U02_HPPR_3_CLEANING_VALVE_Q");
END_REGION
END_FUNCTION

FUNCTION "FC22500_HOPPER_SYSTEM_CONTROLS" : Void   // FC22500, LAD
TITLE = FC22500 HOPPER SYSTEM CONTROLS
{ S7_Optimized_Access := 'TRUE' }
VERSION : 0.1
// stored: AutoNumber false, IsIECCheckEnabled false, SetENOAutomatically false, UDAEnableTagReadback false
   VAR_TEMP
      RPM_INT_AUX : Word;
      RPM_REAL_AUX : Real;
   END_VAR
BEGIN

REGION Network 1: //////////UNIT 01 HOPERS CONTROLS//////////
END_REGION

REGION Network 2: CALL FB22501 TEMPERATURE JKT CONTROL UPPER HOPPER 1 UNIT 01
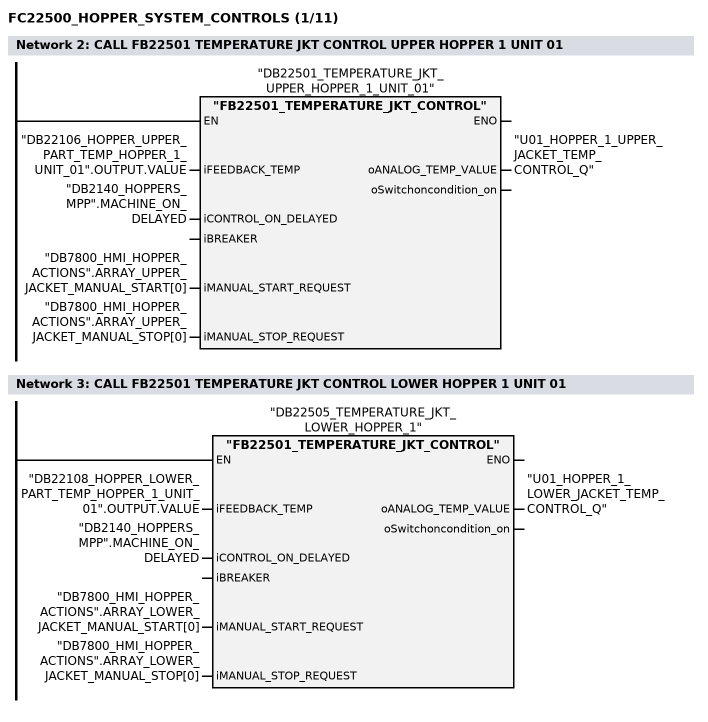
   RUNG wire#powerrail
      "DB22501_TEMPERATURE_JKT_UPPER_HOPPER_1_UNIT_01"(iFEEDBACK_TEMP := "DB22106_HOPPER_UPPER_PART_TEMP_HOPPER_1_UNIT_01".OUTPUT.VALUE, iCONTROL_ON_DELAYED := "DB2140_HOPPERS_MPP".MACHINE_ON_DELAYED, iBREAKER :=, iMANUAL_START_REQUEST := "DB7800_HMI_HOPPER_ACTIONS".ARRAY_UPPER_JACKET_MANUAL_START[0], iMANUAL_STOP_REQUEST := "DB7800_HMI_HOPPER_ACTIONS".ARRAY_UPPER_JACKET_MANUAL_STOP[0], oANALOG_TEMP_VALUE => "U01_HOPPER_1_UPPER_JACKET_TEMP_CONTROL_Q", oSwitchoncondition_on =>)
   END_RUNG
   // the same network as SCL:
   "DB22501_TEMPERATURE_JKT_UPPER_HOPPER_1_UNIT_01"(iFEEDBACK_TEMP := "DB22106_HOPPER_UPPER_PART_TEMP_HOPPER_1_UNIT_01".OUTPUT.VALUE,   // "FB22501_TEMPERATURE_JKT_CONTROL"
                           iCONTROL_ON_DELAYED := "DB2140_HOPPERS_MPP".MACHINE_ON_DELAYED,
                           iMANUAL_START_REQUEST := "DB7800_HMI_HOPPER_ACTIONS".ARRAY_UPPER_JACKET_MANUAL_START[0],
                           iMANUAL_STOP_REQUEST := "DB7800_HMI_HOPPER_ACTIONS".ARRAY_UPPER_JACKET_MANUAL_STOP[0],
                           oANALOG_TEMP_VALUE => "U01_HOPPER_1_UPPER_JACKET_TEMP_CONTROL_Q");
END_REGION

REGION Network 3: CALL FB22501 TEMPERATURE JKT CONTROL LOWER HOPPER 1 UNIT 01
   RUNG wire#powerrail
      "DB22505_TEMPERATURE_JKT_LOWER_HOPPER_1"(iFEEDBACK_TEMP := "DB22108_HOPPER_LOWER_PART_TEMP_HOPPER_1_UNIT_01".OUTPUT.VALUE, iCONTROL_ON_DELAYED := "DB2140_HOPPERS_MPP".MACHINE_ON_DELAYED, iBREAKER :=, iMANUAL_START_REQUEST := "DB7800_HMI_HOPPER_ACTIONS".ARRAY_LOWER_JACKET_MANUAL_START[0], iMANUAL_STOP_REQUEST := "DB7800_HMI_HOPPER_ACTIONS".ARRAY_LOWER_JACKET_MANUAL_STOP[0], oANALOG_TEMP_VALUE => "U01_HOPPER_1_LOWER_JACKET_TEMP_CONTROL_Q", oSwitchoncondition_on =>)
   END_RUNG
   // the same network as SCL:
   "DB22505_TEMPERATURE_JKT_LOWER_HOPPER_1"(iFEEDBACK_TEMP := "DB22108_HOPPER_LOWER_PART_TEMP_HOPPER_1_UNIT_01".OUTPUT.VALUE,   // "FB22501_TEMPERATURE_JKT_CONTROL"
                           iCONTROL_ON_DELAYED := "DB2140_HOPPERS_MPP".MACHINE_ON_DELAYED,
                           iMANUAL_START_REQUEST := "DB7800_HMI_HOPPER_ACTIONS".ARRAY_LOWER_JACKET_MANUAL_START[0],
                           iMANUAL_STOP_REQUEST := "DB7800_HMI_HOPPER_ACTIONS".ARRAY_LOWER_JACKET_MANUAL_STOP[0],
                           oANALOG_TEMP_VALUE => "U01_HOPPER_1_LOWER_JACKET_TEMP_CONTROL_Q");
END_REGION

REGION Network 4: CALL FB22502 MOTOR STIRRER CONTROL HOPPER 1 UNIT 01
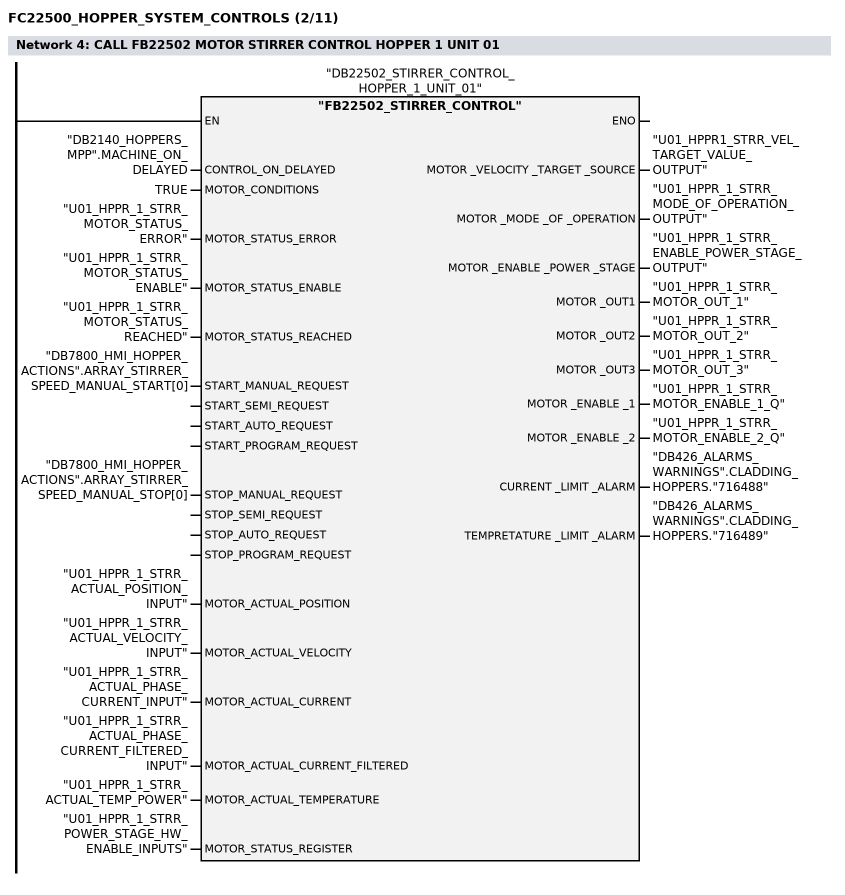
   RUNG wire#powerrail
      "DB22502_STIRRER_CONTROL_HOPPER_1_UNIT_01"(CONTROL_ON_DELAYED := "DB2140_HOPPERS_MPP".MACHINE_ON_DELAYED, MOTOR_CONDITIONS := TRUE, MOTOR_STATUS_ERROR := "U01_HPPR_1_STRR_MOTOR_STATUS_ERROR", MOTOR_STATUS_ENABLE := "U01_HPPR_1_STRR_MOTOR_STATUS_ENABLE", MOTOR_STATUS_REACHED := "U01_HPPR_1_STRR_MOTOR_STATUS_REACHED", START_MANUAL_REQUEST := "DB7800_HMI_HOPPER_ACTIONS".ARRAY_STIRRER_SPEED_MANUAL_START[0], START_SEMI_REQUEST :=, START_AUTO_REQUEST :=, START_PROGRAM_REQUEST :=, STOP_MANUAL_REQUEST := "DB7800_HMI_HOPPER_ACTIONS".ARRAY_STIRRER_SPEED_MANUAL_STOP[0], STOP_SEMI_REQUEST :=, STOP_AUTO_REQUEST :=, STOP_PROGRAM_REQUEST :=, MOTOR_ACTUAL_POSITION := "U01_HPPR_1_STRR_ACTUAL_POSITION_INPUT", MOTOR_ACTUAL_VELOCITY := "U01_HPPR_1_STRR_ACTUAL_VELOCITY_INPUT", MOTOR_ACTUAL_CURRENT := "U01_HPPR_1_STRR_ACTUAL_PHASE_CURRENT_INPUT", MOTOR_ACTUAL_CURRENT_FILTERED := "U01_HPPR_1_STRR_ACTUAL_PHASE_CURRENT_FILTERED_INPUT", MOTOR_ACTUAL_TEMPERATURE := "U01_HPPR_1_STRR_ACTUAL_TEMP_POWER", MOTOR_STATUS_REGISTER := "U01_HPPR_1_STRR_POWER_STAGE_HW_ENABLE_INPUTS", "MOTOR _VELOCITY _TARGET _SOURCE" => "U01_HPPR1_STRR_VEL_TARGET_VALUE_OUTPUT", "MOTOR _MODE _OF _OPERATION" => "U01_HPPR_1_STRR_MODE_OF_OPERATION_OUTPUT", "MOTOR _ENABLE _POWER _STAGE" => "U01_HPPR_1_STRR_ENABLE_POWER_STAGE_OUTPUT", "MOTOR _OUT1" => "U01_HPPR_1_STRR_MOTOR_OUT_1", "MOTOR _OUT2" => "U01_HPPR_1_STRR_MOTOR_OUT_2", "MOTOR _OUT3" => "U01_HPPR_1_STRR_MOTOR_OUT_3", "MOTOR _ENABLE _1" => "U01_HPPR_1_STRR_MOTOR_ENABLE_1_Q", "MOTOR _ENABLE _2" => "U01_HPPR_1_STRR_MOTOR_ENABLE_2_Q", "CURRENT _LIMIT _ALARM" => "DB426_ALARMS_WARNINGS".CLADDING_HOPPERS."716488", "TEMPRETATURE _LIMIT _ALARM" => "DB426_ALARMS_WARNINGS".CLADDING_HOPPERS."716489")
   END_RUNG
   // the same network as SCL:
   "DB22502_STIRRER_CONTROL_HOPPER_1_UNIT_01"(CONTROL_ON_DELAYED := "DB2140_HOPPERS_MPP".MACHINE_ON_DELAYED,   // "FB22502_STIRRER_CONTROL"
                           MOTOR_CONDITIONS := TRUE,
                           MOTOR_STATUS_ERROR := "U01_HPPR_1_STRR_MOTOR_STATUS_ERROR",
                           MOTOR_STATUS_ENABLE := "U01_HPPR_1_STRR_MOTOR_STATUS_ENABLE",
                           MOTOR_STATUS_REACHED := "U01_HPPR_1_STRR_MOTOR_STATUS_REACHED",
                           START_MANUAL_REQUEST := "DB7800_HMI_HOPPER_ACTIONS".ARRAY_STIRRER_SPEED_MANUAL_START[0],
                           STOP_MANUAL_REQUEST := "DB7800_HMI_HOPPER_ACTIONS".ARRAY_STIRRER_SPEED_MANUAL_STOP[0],
                           MOTOR_ACTUAL_POSITION := "U01_HPPR_1_STRR_ACTUAL_POSITION_INPUT",
                           MOTOR_ACTUAL_VELOCITY := "U01_HPPR_1_STRR_ACTUAL_VELOCITY_INPUT",
                           MOTOR_ACTUAL_CURRENT := "U01_HPPR_1_STRR_ACTUAL_PHASE_CURRENT_INPUT",
                           MOTOR_ACTUAL_CURRENT_FILTERED := "U01_HPPR_1_STRR_ACTUAL_PHASE_CURRENT_FILTERED_INPUT",
                           MOTOR_ACTUAL_TEMPERATURE := "U01_HPPR_1_STRR_ACTUAL_TEMP_POWER",
                           MOTOR_STATUS_REGISTER := "U01_HPPR_1_STRR_POWER_STAGE_HW_ENABLE_INPUTS",
                           "MOTOR _VELOCITY _TARGET _SOURCE" => "U01_HPPR1_STRR_VEL_TARGET_VALUE_OUTPUT",
                           "MOTOR _MODE _OF _OPERATION" => "U01_HPPR_1_STRR_MODE_OF_OPERATION_OUTPUT",
                           "MOTOR _ENABLE _POWER _STAGE" => "U01_HPPR_1_STRR_ENABLE_POWER_STAGE_OUTPUT",
                           "MOTOR _OUT1" => "U01_HPPR_1_STRR_MOTOR_OUT_1",
                           "MOTOR _OUT2" => "U01_HPPR_1_STRR_MOTOR_OUT_2",
                           "MOTOR _OUT3" => "U01_HPPR_1_STRR_MOTOR_OUT_3",
                           "MOTOR _ENABLE _1" => "U01_HPPR_1_STRR_MOTOR_ENABLE_1_Q",
                           "MOTOR _ENABLE _2" => "U01_HPPR_1_STRR_MOTOR_ENABLE_2_Q",
                           "CURRENT _LIMIT _ALARM" => "DB426_ALARMS_WARNINGS".CLADDING_HOPPERS."716488",
                           "TEMPRETATURE _LIMIT _ALARM" => "DB426_ALARMS_WARNINGS".CLADDING_HOPPERS."716489");
END_REGION

REGION Network 5: CALL FB22503 HOPPER COVER PRESSURE CONTROL HOPPER 1 UNIT 01
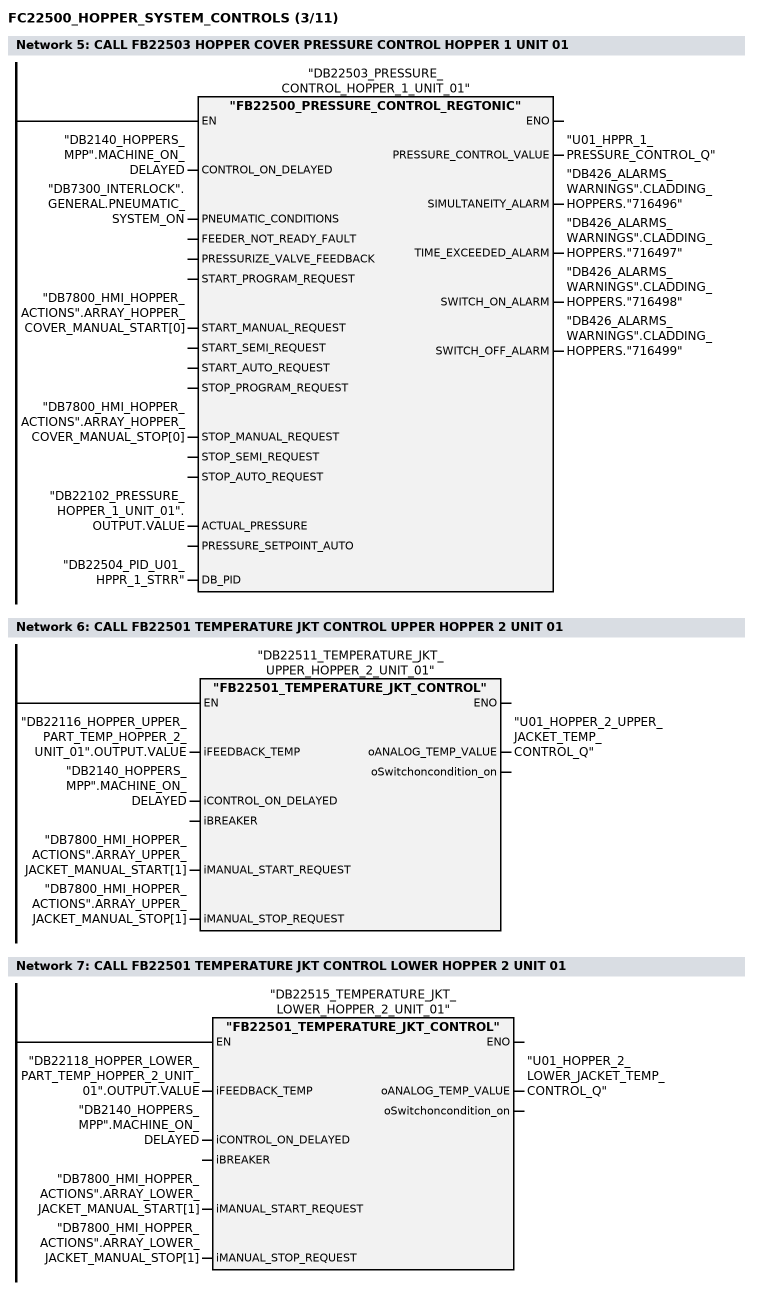
   RUNG wire#powerrail
      "DB22503_PRESSURE_CONTROL_HOPPER_1_UNIT_01"(CONTROL_ON_DELAYED := "DB2140_HOPPERS_MPP".MACHINE_ON_DELAYED, PNEUMATIC_CONDITIONS := "DB7300_INTERLOCK".GENERAL.PNEUMATIC_SYSTEM_ON, FEEDER_NOT_READY_FAULT :=, PRESSURIZE_VALVE_FEEDBACK :=, START_PROGRAM_REQUEST :=, START_MANUAL_REQUEST := "DB7800_HMI_HOPPER_ACTIONS".ARRAY_HOPPER_COVER_MANUAL_START[0], START_SEMI_REQUEST :=, START_AUTO_REQUEST :=, STOP_PROGRAM_REQUEST :=, STOP_MANUAL_REQUEST := "DB7800_HMI_HOPPER_ACTIONS".ARRAY_HOPPER_COVER_MANUAL_STOP[0], STOP_SEMI_REQUEST :=, STOP_AUTO_REQUEST :=, ACTUAL_PRESSURE := "DB22102_PRESSURE_HOPPER_1_UNIT_01".OUTPUT.VALUE, PRESSURE_SETPOINT_AUTO :=, DB_PID := "DB22504_PID_U01_HPPR_1_STRR", PRESSURE_CONTROL_VALUE => "U01_HPPR_1_PRESSURE_CONTROL_Q", SIMULTANEITY_ALARM => "DB426_ALARMS_WARNINGS".CLADDING_HOPPERS."716496", TIME_EXCEEDED_ALARM => "DB426_ALARMS_WARNINGS".CLADDING_HOPPERS."716497", SWITCH_ON_ALARM => "DB426_ALARMS_WARNINGS".CLADDING_HOPPERS."716498", SWITCH_OFF_ALARM => "DB426_ALARMS_WARNINGS".CLADDING_HOPPERS."716499")
   END_RUNG
   // the same network as SCL:
   "DB22503_PRESSURE_CONTROL_HOPPER_1_UNIT_01"(CONTROL_ON_DELAYED := "DB2140_HOPPERS_MPP".MACHINE_ON_DELAYED,   // "FB22500_PRESSURE_CONTROL_REGTONIC"
                           PNEUMATIC_CONDITIONS := "DB7300_INTERLOCK".GENERAL.PNEUMATIC_SYSTEM_ON,
                           START_MANUAL_REQUEST := "DB7800_HMI_HOPPER_ACTIONS".ARRAY_HOPPER_COVER_MANUAL_START[0],
                           STOP_MANUAL_REQUEST := "DB7800_HMI_HOPPER_ACTIONS".ARRAY_HOPPER_COVER_MANUAL_STOP[0],
                           ACTUAL_PRESSURE := "DB22102_PRESSURE_HOPPER_1_UNIT_01".OUTPUT.VALUE,
                           DB_PID := "DB22504_PID_U01_HPPR_1_STRR",
                           PRESSURE_CONTROL_VALUE => "U01_HPPR_1_PRESSURE_CONTROL_Q",
                           SIMULTANEITY_ALARM => "DB426_ALARMS_WARNINGS".CLADDING_HOPPERS."716496",
                           TIME_EXCEEDED_ALARM => "DB426_ALARMS_WARNINGS".CLADDING_HOPPERS."716497",
                           SWITCH_ON_ALARM => "DB426_ALARMS_WARNINGS".CLADDING_HOPPERS."716498",
                           SWITCH_OFF_ALARM => "DB426_ALARMS_WARNINGS".CLADDING_HOPPERS."716499");
END_REGION

REGION Network 6: CALL FB22501 TEMPERATURE JKT CONTROL UPPER HOPPER 2 UNIT 01
   RUNG wire#powerrail
      "DB22511_TEMPERATURE_JKT_UPPER_HOPPER_2_UNIT_01"(iFEEDBACK_TEMP := "DB22116_HOPPER_UPPER_PART_TEMP_HOPPER_2_UNIT_01".OUTPUT.VALUE, iCONTROL_ON_DELAYED := "DB2140_HOPPERS_MPP".MACHINE_ON_DELAYED, iBREAKER :=, iMANUAL_START_REQUEST := "DB7800_HMI_HOPPER_ACTIONS".ARRAY_UPPER_JACKET_MANUAL_START[1], iMANUAL_STOP_REQUEST := "DB7800_HMI_HOPPER_ACTIONS".ARRAY_UPPER_JACKET_MANUAL_STOP[1], oANALOG_TEMP_VALUE => "U01_HOPPER_2_UPPER_JACKET_TEMP_CONTROL_Q", oSwitchoncondition_on =>)
   END_RUNG
   // the same network as SCL:
   "DB22511_TEMPERATURE_JKT_UPPER_HOPPER_2_UNIT_01"(iFEEDBACK_TEMP := "DB22116_HOPPER_UPPER_PART_TEMP_HOPPER_2_UNIT_01".OUTPUT.VALUE,   // "FB22501_TEMPERATURE_JKT_CONTROL"
                           iCONTROL_ON_DELAYED := "DB2140_HOPPERS_MPP".MACHINE_ON_DELAYED,
                           iMANUAL_START_REQUEST := "DB7800_HMI_HOPPER_ACTIONS".ARRAY_UPPER_JACKET_MANUAL_START[1],
                           iMANUAL_STOP_REQUEST := "DB7800_HMI_HOPPER_ACTIONS".ARRAY_UPPER_JACKET_MANUAL_STOP[1],
                           oANALOG_TEMP_VALUE => "U01_HOPPER_2_UPPER_JACKET_TEMP_CONTROL_Q");
END_REGION

REGION Network 7: CALL FB22501 TEMPERATURE JKT CONTROL LOWER HOPPER 2 UNIT 01
   RUNG wire#powerrail
      "DB22515_TEMPERATURE_JKT_LOWER_HOPPER_2_UNIT_01"(iFEEDBACK_TEMP := "DB22118_HOPPER_LOWER_PART_TEMP_HOPPER_2_UNIT_01".OUTPUT.VALUE, iCONTROL_ON_DELAYED := "DB2140_HOPPERS_MPP".MACHINE_ON_DELAYED, iBREAKER :=, iMANUAL_START_REQUEST := "DB7800_HMI_HOPPER_ACTIONS".ARRAY_LOWER_JACKET_MANUAL_START[1], iMANUAL_STOP_REQUEST := "DB7800_HMI_HOPPER_ACTIONS".ARRAY_LOWER_JACKET_MANUAL_STOP[1], oANALOG_TEMP_VALUE => "U01_HOPPER_2_LOWER_JACKET_TEMP_CONTROL_Q", oSwitchoncondition_on =>)
   END_RUNG
   // the same network as SCL:
   "DB22515_TEMPERATURE_JKT_LOWER_HOPPER_2_UNIT_01"(iFEEDBACK_TEMP := "DB22118_HOPPER_LOWER_PART_TEMP_HOPPER_2_UNIT_01".OUTPUT.VALUE,   // "FB22501_TEMPERATURE_JKT_CONTROL"
                           iCONTROL_ON_DELAYED := "DB2140_HOPPERS_MPP".MACHINE_ON_DELAYED,
                           iMANUAL_START_REQUEST := "DB7800_HMI_HOPPER_ACTIONS".ARRAY_LOWER_JACKET_MANUAL_START[1],
                           iMANUAL_STOP_REQUEST := "DB7800_HMI_HOPPER_ACTIONS".ARRAY_LOWER_JACKET_MANUAL_STOP[1],
                           oANALOG_TEMP_VALUE => "U01_HOPPER_2_LOWER_JACKET_TEMP_CONTROL_Q");
END_REGION

REGION Network 8: CALL FB22502 MOTOR STIRRER CONTROL HOPPER 2 UNIT 01
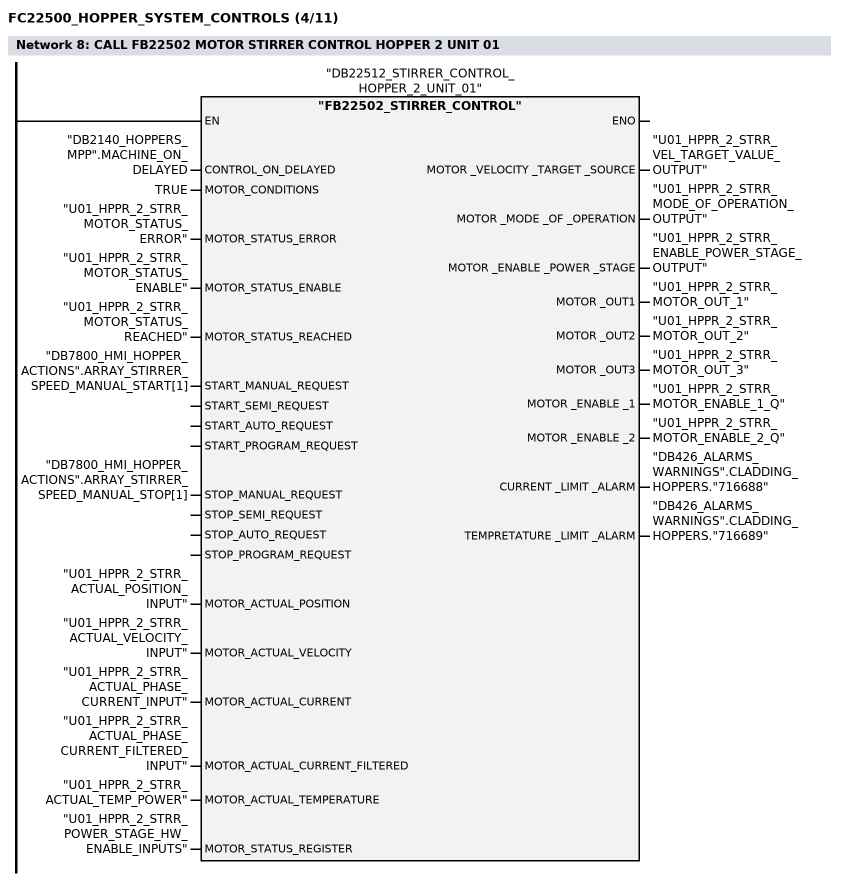
   RUNG wire#powerrail
      "DB22512_STIRRER_CONTROL_HOPPER_2_UNIT_01"(CONTROL_ON_DELAYED := "DB2140_HOPPERS_MPP".MACHINE_ON_DELAYED, MOTOR_CONDITIONS := TRUE, MOTOR_STATUS_ERROR := "U01_HPPR_2_STRR_MOTOR_STATUS_ERROR", MOTOR_STATUS_ENABLE := "U01_HPPR_2_STRR_MOTOR_STATUS_ENABLE", MOTOR_STATUS_REACHED := "U01_HPPR_2_STRR_MOTOR_STATUS_REACHED", START_MANUAL_REQUEST := "DB7800_HMI_HOPPER_ACTIONS".ARRAY_STIRRER_SPEED_MANUAL_START[1], START_SEMI_REQUEST :=, START_AUTO_REQUEST :=, START_PROGRAM_REQUEST :=, STOP_MANUAL_REQUEST := "DB7800_HMI_HOPPER_ACTIONS".ARRAY_STIRRER_SPEED_MANUAL_STOP[1], STOP_SEMI_REQUEST :=, STOP_AUTO_REQUEST :=, STOP_PROGRAM_REQUEST :=, MOTOR_ACTUAL_POSITION := "U01_HPPR_2_STRR_ACTUAL_POSITION_INPUT", MOTOR_ACTUAL_VELOCITY := "U01_HPPR_2_STRR_ACTUAL_VELOCITY_INPUT", MOTOR_ACTUAL_CURRENT := "U01_HPPR_2_STRR_ACTUAL_PHASE_CURRENT_INPUT", MOTOR_ACTUAL_CURRENT_FILTERED := "U01_HPPR_2_STRR_ACTUAL_PHASE_CURRENT_FILTERED_INPUT", MOTOR_ACTUAL_TEMPERATURE := "U01_HPPR_2_STRR_ACTUAL_TEMP_POWER", MOTOR_STATUS_REGISTER := "U01_HPPR_2_STRR_POWER_STAGE_HW_ENABLE_INPUTS", "MOTOR _VELOCITY _TARGET _SOURCE" => "U01_HPPR_2_STRR_VEL_TARGET_VALUE_OUTPUT", "MOTOR _MODE _OF _OPERATION" => "U01_HPPR_2_STRR_MODE_OF_OPERATION_OUTPUT", "MOTOR _ENABLE _POWER _STAGE" => "U01_HPPR_2_STRR_ENABLE_POWER_STAGE_OUTPUT", "MOTOR _OUT1" => "U01_HPPR_2_STRR_MOTOR_OUT_1", "MOTOR _OUT2" => "U01_HPPR_2_STRR_MOTOR_OUT_2", "MOTOR _OUT3" => "U01_HPPR_2_STRR_MOTOR_OUT_3", "MOTOR _ENABLE _1" => "U01_HPPR_2_STRR_MOTOR_ENABLE_1_Q", "MOTOR _ENABLE _2" => "U01_HPPR_2_STRR_MOTOR_ENABLE_2_Q", "CURRENT _LIMIT _ALARM" => "DB426_ALARMS_WARNINGS".CLADDING_HOPPERS."716688", "TEMPRETATURE _LIMIT _ALARM" => "DB426_ALARMS_WARNINGS".CLADDING_HOPPERS."716689")
   END_RUNG
   // the same network as SCL:
   "DB22512_STIRRER_CONTROL_HOPPER_2_UNIT_01"(CONTROL_ON_DELAYED := "DB2140_HOPPERS_MPP".MACHINE_ON_DELAYED,   // "FB22502_STIRRER_CONTROL"
                           MOTOR_CONDITIONS := TRUE,
                           MOTOR_STATUS_ERROR := "U01_HPPR_2_STRR_MOTOR_STATUS_ERROR",
                           MOTOR_STATUS_ENABLE := "U01_HPPR_2_STRR_MOTOR_STATUS_ENABLE",
                           MOTOR_STATUS_REACHED := "U01_HPPR_2_STRR_MOTOR_STATUS_REACHED",
                           START_MANUAL_REQUEST := "DB7800_HMI_HOPPER_ACTIONS".ARRAY_STIRRER_SPEED_MANUAL_START[1],
                           STOP_MANUAL_REQUEST := "DB7800_HMI_HOPPER_ACTIONS".ARRAY_STIRRER_SPEED_MANUAL_STOP[1],
                           MOTOR_ACTUAL_POSITION := "U01_HPPR_2_STRR_ACTUAL_POSITION_INPUT",
                           MOTOR_ACTUAL_VELOCITY := "U01_HPPR_2_STRR_ACTUAL_VELOCITY_INPUT",
                           MOTOR_ACTUAL_CURRENT := "U01_HPPR_2_STRR_ACTUAL_PHASE_CURRENT_INPUT",
                           MOTOR_ACTUAL_CURRENT_FILTERED := "U01_HPPR_2_STRR_ACTUAL_PHASE_CURRENT_FILTERED_INPUT",
                           MOTOR_ACTUAL_TEMPERATURE := "U01_HPPR_2_STRR_ACTUAL_TEMP_POWER",
                           MOTOR_STATUS_REGISTER := "U01_HPPR_2_STRR_POWER_STAGE_HW_ENABLE_INPUTS",
                           "MOTOR _VELOCITY _TARGET _SOURCE" => "U01_HPPR_2_STRR_VEL_TARGET_VALUE_OUTPUT",
                           "MOTOR _MODE _OF _OPERATION" => "U01_HPPR_2_STRR_MODE_OF_OPERATION_OUTPUT",
                           "MOTOR _ENABLE _POWER _STAGE" => "U01_HPPR_2_STRR_ENABLE_POWER_STAGE_OUTPUT",
                           "MOTOR _OUT1" => "U01_HPPR_2_STRR_MOTOR_OUT_1",
                           "MOTOR _OUT2" => "U01_HPPR_2_STRR_MOTOR_OUT_2",
                           "MOTOR _OUT3" => "U01_HPPR_2_STRR_MOTOR_OUT_3",
                           "MOTOR _ENABLE _1" => "U01_HPPR_2_STRR_MOTOR_ENABLE_1_Q",
                           "MOTOR _ENABLE _2" => "U01_HPPR_2_STRR_MOTOR_ENABLE_2_Q",
                           "CURRENT _LIMIT _ALARM" => "DB426_ALARMS_WARNINGS".CLADDING_HOPPERS."716688",
                           "TEMPRETATURE _LIMIT _ALARM" => "DB426_ALARMS_WARNINGS".CLADDING_HOPPERS."716689");
END_REGION

REGION Network 9: CALL FB22503 HOPPER PRESSURE CONTROL HOPPER 2 UNIT 01
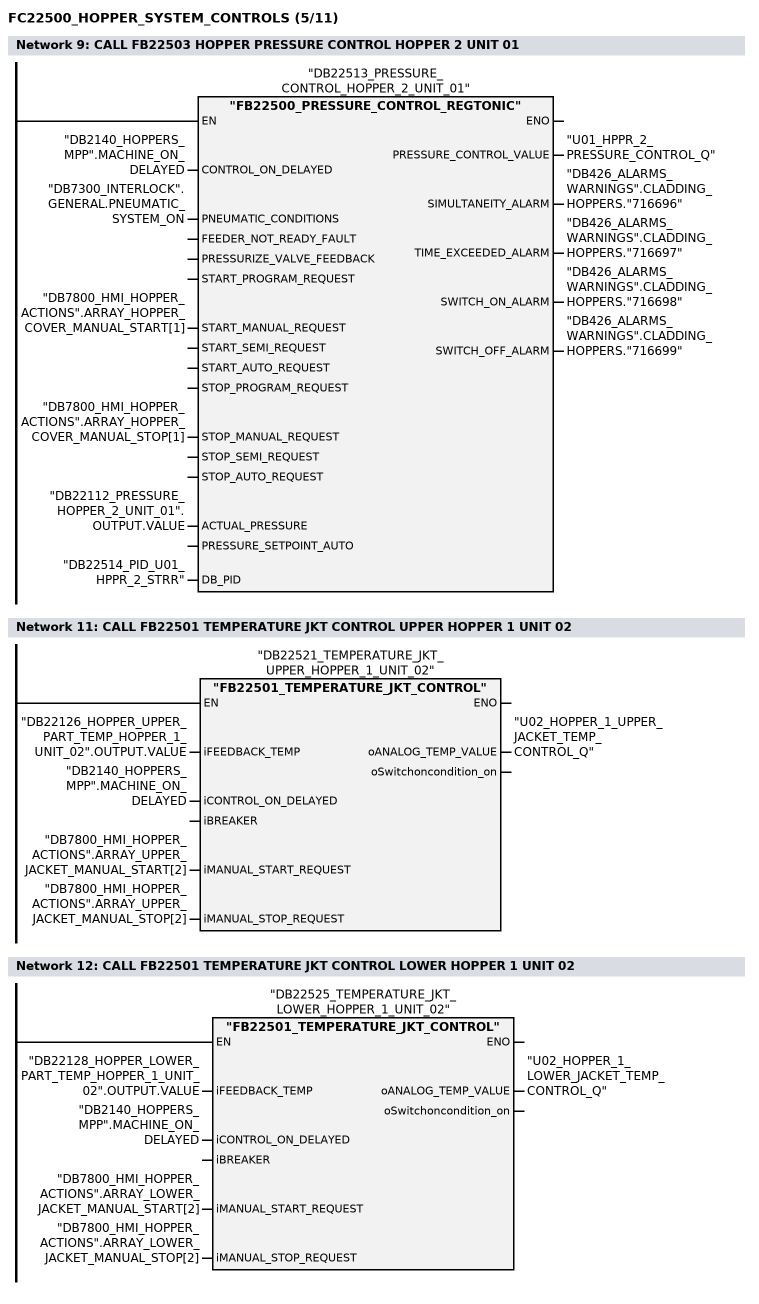
   RUNG wire#powerrail
      "DB22513_PRESSURE_CONTROL_HOPPER_2_UNIT_01"(CONTROL_ON_DELAYED := "DB2140_HOPPERS_MPP".MACHINE_ON_DELAYED, PNEUMATIC_CONDITIONS := "DB7300_INTERLOCK".GENERAL.PNEUMATIC_SYSTEM_ON, FEEDER_NOT_READY_FAULT :=, PRESSURIZE_VALVE_FEEDBACK :=, START_PROGRAM_REQUEST :=, START_MANUAL_REQUEST := "DB7800_HMI_HOPPER_ACTIONS".ARRAY_HOPPER_COVER_MANUAL_START[1], START_SEMI_REQUEST :=, START_AUTO_REQUEST :=, STOP_PROGRAM_REQUEST :=, STOP_MANUAL_REQUEST := "DB7800_HMI_HOPPER_ACTIONS".ARRAY_HOPPER_COVER_MANUAL_STOP[1], STOP_SEMI_REQUEST :=, STOP_AUTO_REQUEST :=, ACTUAL_PRESSURE := "DB22112_PRESSURE_HOPPER_2_UNIT_01".OUTPUT.VALUE, PRESSURE_SETPOINT_AUTO :=, DB_PID := "DB22514_PID_U01_HPPR_2_STRR", PRESSURE_CONTROL_VALUE => "U01_HPPR_2_PRESSURE_CONTROL_Q", SIMULTANEITY_ALARM => "DB426_ALARMS_WARNINGS".CLADDING_HOPPERS."716696", TIME_EXCEEDED_ALARM => "DB426_ALARMS_WARNINGS".CLADDING_HOPPERS."716697", SWITCH_ON_ALARM => "DB426_ALARMS_WARNINGS".CLADDING_HOPPERS."716698", SWITCH_OFF_ALARM => "DB426_ALARMS_WARNINGS".CLADDING_HOPPERS."716699")
   END_RUNG
   // the same network as SCL:
   "DB22513_PRESSURE_CONTROL_HOPPER_2_UNIT_01"(CONTROL_ON_DELAYED := "DB2140_HOPPERS_MPP".MACHINE_ON_DELAYED,   // "FB22500_PRESSURE_CONTROL_REGTONIC"
                           PNEUMATIC_CONDITIONS := "DB7300_INTERLOCK".GENERAL.PNEUMATIC_SYSTEM_ON,
                           START_MANUAL_REQUEST := "DB7800_HMI_HOPPER_ACTIONS".ARRAY_HOPPER_COVER_MANUAL_START[1],
                           STOP_MANUAL_REQUEST := "DB7800_HMI_HOPPER_ACTIONS".ARRAY_HOPPER_COVER_MANUAL_STOP[1],
                           ACTUAL_PRESSURE := "DB22112_PRESSURE_HOPPER_2_UNIT_01".OUTPUT.VALUE,
                           DB_PID := "DB22514_PID_U01_HPPR_2_STRR",
                           PRESSURE_CONTROL_VALUE => "U01_HPPR_2_PRESSURE_CONTROL_Q",
                           SIMULTANEITY_ALARM => "DB426_ALARMS_WARNINGS".CLADDING_HOPPERS."716696",
                           TIME_EXCEEDED_ALARM => "DB426_ALARMS_WARNINGS".CLADDING_HOPPERS."716697",
                           SWITCH_ON_ALARM => "DB426_ALARMS_WARNINGS".CLADDING_HOPPERS."716698",
                           SWITCH_OFF_ALARM => "DB426_ALARMS_WARNINGS".CLADDING_HOPPERS."716699");
END_REGION

REGION Network 10: //////////UNIT 02 HOPERS CONTROLS//////////
END_REGION

REGION Network 11: CALL FB22501 TEMPERATURE JKT CONTROL UPPER HOPPER 1 UNIT 02
   RUNG wire#powerrail
      "DB22521_TEMPERATURE_JKT_UPPER_HOPPER_1_UNIT_02"(iFEEDBACK_TEMP := "DB22126_HOPPER_UPPER_PART_TEMP_HOPPER_1_UNIT_02".OUTPUT.VALUE, iCONTROL_ON_DELAYED := "DB2140_HOPPERS_MPP".MACHINE_ON_DELAYED, iBREAKER :=, iMANUAL_START_REQUEST := "DB7800_HMI_HOPPER_ACTIONS".ARRAY_UPPER_JACKET_MANUAL_START[2], iMANUAL_STOP_REQUEST := "DB7800_HMI_HOPPER_ACTIONS".ARRAY_UPPER_JACKET_MANUAL_STOP[2], oANALOG_TEMP_VALUE => "U02_HOPPER_1_UPPER_JACKET_TEMP_CONTROL_Q", oSwitchoncondition_on =>)
   END_RUNG
   // the same network as SCL:
   "DB22521_TEMPERATURE_JKT_UPPER_HOPPER_1_UNIT_02"(iFEEDBACK_TEMP := "DB22126_HOPPER_UPPER_PART_TEMP_HOPPER_1_UNIT_02".OUTPUT.VALUE,   // "FB22501_TEMPERATURE_JKT_CONTROL"
                           iCONTROL_ON_DELAYED := "DB2140_HOPPERS_MPP".MACHINE_ON_DELAYED,
                           iMANUAL_START_REQUEST := "DB7800_HMI_HOPPER_ACTIONS".ARRAY_UPPER_JACKET_MANUAL_START[2],
                           iMANUAL_STOP_REQUEST := "DB7800_HMI_HOPPER_ACTIONS".ARRAY_UPPER_JACKET_MANUAL_STOP[2],
                           oANALOG_TEMP_VALUE => "U02_HOPPER_1_UPPER_JACKET_TEMP_CONTROL_Q");
END_REGION

REGION Network 12: CALL FB22501 TEMPERATURE JKT CONTROL LOWER HOPPER 1 UNIT 02
   RUNG wire#powerrail
      "DB22525_TEMPERATURE_JKT_LOWER_HOPPER_1_UNIT_02"(iFEEDBACK_TEMP := "DB22128_HOPPER_LOWER_PART_TEMP_HOPPER_1_UNIT_02".OUTPUT.VALUE, iCONTROL_ON_DELAYED := "DB2140_HOPPERS_MPP".MACHINE_ON_DELAYED, iBREAKER :=, iMANUAL_START_REQUEST := "DB7800_HMI_HOPPER_ACTIONS".ARRAY_LOWER_JACKET_MANUAL_START[2], iMANUAL_STOP_REQUEST := "DB7800_HMI_HOPPER_ACTIONS".ARRAY_LOWER_JACKET_MANUAL_STOP[2], oANALOG_TEMP_VALUE => "U02_HOPPER_1_LOWER_JACKET_TEMP_CONTROL_Q", oSwitchoncondition_on =>)
   END_RUNG
   // the same network as SCL:
   "DB22525_TEMPERATURE_JKT_LOWER_HOPPER_1_UNIT_02"(iFEEDBACK_TEMP := "DB22128_HOPPER_LOWER_PART_TEMP_HOPPER_1_UNIT_02".OUTPUT.VALUE,   // "FB22501_TEMPERATURE_JKT_CONTROL"
                           iCONTROL_ON_DELAYED := "DB2140_HOPPERS_MPP".MACHINE_ON_DELAYED,
                           iMANUAL_START_REQUEST := "DB7800_HMI_HOPPER_ACTIONS".ARRAY_LOWER_JACKET_MANUAL_START[2],
                           iMANUAL_STOP_REQUEST := "DB7800_HMI_HOPPER_ACTIONS".ARRAY_LOWER_JACKET_MANUAL_STOP[2],
                           oANALOG_TEMP_VALUE => "U02_HOPPER_1_LOWER_JACKET_TEMP_CONTROL_Q");
END_REGION

REGION Network 13: CALL FB22502 MOTOR STIRRER CONTROL HOPPER 1 UNIT 02
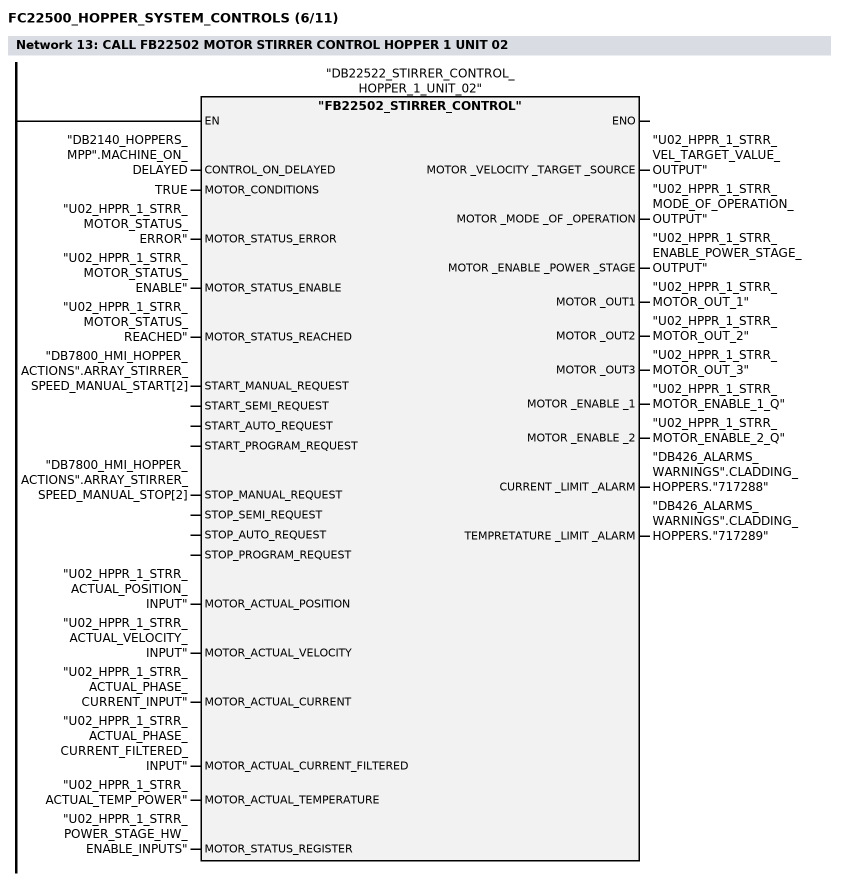
   RUNG wire#powerrail
      "DB22522_STIRRER_CONTROL_HOPPER_1_UNIT_02"(CONTROL_ON_DELAYED := "DB2140_HOPPERS_MPP".MACHINE_ON_DELAYED, MOTOR_CONDITIONS := TRUE, MOTOR_STATUS_ERROR := "U02_HPPR_1_STRR_MOTOR_STATUS_ERROR", MOTOR_STATUS_ENABLE := "U02_HPPR_1_STRR_MOTOR_STATUS_ENABLE", MOTOR_STATUS_REACHED := "U02_HPPR_1_STRR_MOTOR_STATUS_REACHED", START_MANUAL_REQUEST := "DB7800_HMI_HOPPER_ACTIONS".ARRAY_STIRRER_SPEED_MANUAL_START[2], START_SEMI_REQUEST :=, START_AUTO_REQUEST :=, START_PROGRAM_REQUEST :=, STOP_MANUAL_REQUEST := "DB7800_HMI_HOPPER_ACTIONS".ARRAY_STIRRER_SPEED_MANUAL_STOP[2], STOP_SEMI_REQUEST :=, STOP_AUTO_REQUEST :=, STOP_PROGRAM_REQUEST :=, MOTOR_ACTUAL_POSITION := "U02_HPPR_1_STRR_ACTUAL_POSITION_INPUT", MOTOR_ACTUAL_VELOCITY := "U02_HPPR_1_STRR_ACTUAL_VELOCITY_INPUT", MOTOR_ACTUAL_CURRENT := "U02_HPPR_1_STRR_ACTUAL_PHASE_CURRENT_INPUT", MOTOR_ACTUAL_CURRENT_FILTERED := "U02_HPPR_1_STRR_ACTUAL_PHASE_CURRENT_FILTERED_INPUT", MOTOR_ACTUAL_TEMPERATURE := "U02_HPPR_1_STRR_ACTUAL_TEMP_POWER", MOTOR_STATUS_REGISTER := "U02_HPPR_1_STRR_POWER_STAGE_HW_ENABLE_INPUTS", "MOTOR _VELOCITY _TARGET _SOURCE" => "U02_HPPR_1_STRR_VEL_TARGET_VALUE_OUTPUT", "MOTOR _MODE _OF _OPERATION" => "U02_HPPR_1_STRR_MODE_OF_OPERATION_OUTPUT", "MOTOR _ENABLE _POWER _STAGE" => "U02_HPPR_1_STRR_ENABLE_POWER_STAGE_OUTPUT", "MOTOR _OUT1" => "U02_HPPR_1_STRR_MOTOR_OUT_1", "MOTOR _OUT2" => "U02_HPPR_1_STRR_MOTOR_OUT_2", "MOTOR _OUT3" => "U02_HPPR_1_STRR_MOTOR_OUT_3", "MOTOR _ENABLE _1" => "U02_HPPR_1_STRR_MOTOR_ENABLE_1_Q", "MOTOR _ENABLE _2" => "U02_HPPR_1_STRR_MOTOR_ENABLE_2_Q", "CURRENT _LIMIT _ALARM" => "DB426_ALARMS_WARNINGS".CLADDING_HOPPERS."717288", "TEMPRETATURE _LIMIT _ALARM" => "DB426_ALARMS_WARNINGS".CLADDING_HOPPERS."717289")
   END_RUNG
   // the same network as SCL:
   "DB22522_STIRRER_CONTROL_HOPPER_1_UNIT_02"(CONTROL_ON_DELAYED := "DB2140_HOPPERS_MPP".MACHINE_ON_DELAYED,   // "FB22502_STIRRER_CONTROL"
                           MOTOR_CONDITIONS := TRUE,
                           MOTOR_STATUS_ERROR := "U02_HPPR_1_STRR_MOTOR_STATUS_ERROR",
                           MOTOR_STATUS_ENABLE := "U02_HPPR_1_STRR_MOTOR_STATUS_ENABLE",
                           MOTOR_STATUS_REACHED := "U02_HPPR_1_STRR_MOTOR_STATUS_REACHED",
                           START_MANUAL_REQUEST := "DB7800_HMI_HOPPER_ACTIONS".ARRAY_STIRRER_SPEED_MANUAL_START[2],
                           STOP_MANUAL_REQUEST := "DB7800_HMI_HOPPER_ACTIONS".ARRAY_STIRRER_SPEED_MANUAL_STOP[2],
                           MOTOR_ACTUAL_POSITION := "U02_HPPR_1_STRR_ACTUAL_POSITION_INPUT",
                           MOTOR_ACTUAL_VELOCITY := "U02_HPPR_1_STRR_ACTUAL_VELOCITY_INPUT",
                           MOTOR_ACTUAL_CURRENT := "U02_HPPR_1_STRR_ACTUAL_PHASE_CURRENT_INPUT",
                           MOTOR_ACTUAL_CURRENT_FILTERED := "U02_HPPR_1_STRR_ACTUAL_PHASE_CURRENT_FILTERED_INPUT",
                           MOTOR_ACTUAL_TEMPERATURE := "U02_HPPR_1_STRR_ACTUAL_TEMP_POWER",
                           MOTOR_STATUS_REGISTER := "U02_HPPR_1_STRR_POWER_STAGE_HW_ENABLE_INPUTS",
                           "MOTOR _VELOCITY _TARGET _SOURCE" => "U02_HPPR_1_STRR_VEL_TARGET_VALUE_OUTPUT",
                           "MOTOR _MODE _OF _OPERATION" => "U02_HPPR_1_STRR_MODE_OF_OPERATION_OUTPUT",
                           "MOTOR _ENABLE _POWER _STAGE" => "U02_HPPR_1_STRR_ENABLE_POWER_STAGE_OUTPUT",
                           "MOTOR _OUT1" => "U02_HPPR_1_STRR_MOTOR_OUT_1",
                           "MOTOR _OUT2" => "U02_HPPR_1_STRR_MOTOR_OUT_2",
                           "MOTOR _OUT3" => "U02_HPPR_1_STRR_MOTOR_OUT_3",
                           "MOTOR _ENABLE _1" => "U02_HPPR_1_STRR_MOTOR_ENABLE_1_Q",
                           "MOTOR _ENABLE _2" => "U02_HPPR_1_STRR_MOTOR_ENABLE_2_Q",
                           "CURRENT _LIMIT _ALARM" => "DB426_ALARMS_WARNINGS".CLADDING_HOPPERS."717288",
                           "TEMPRETATURE _LIMIT _ALARM" => "DB426_ALARMS_WARNINGS".CLADDING_HOPPERS."717289");
END_REGION

REGION Network 14: CALL FB22503 HOPPER PRESSURE CONTROL HOPPER 1 UNIT 02
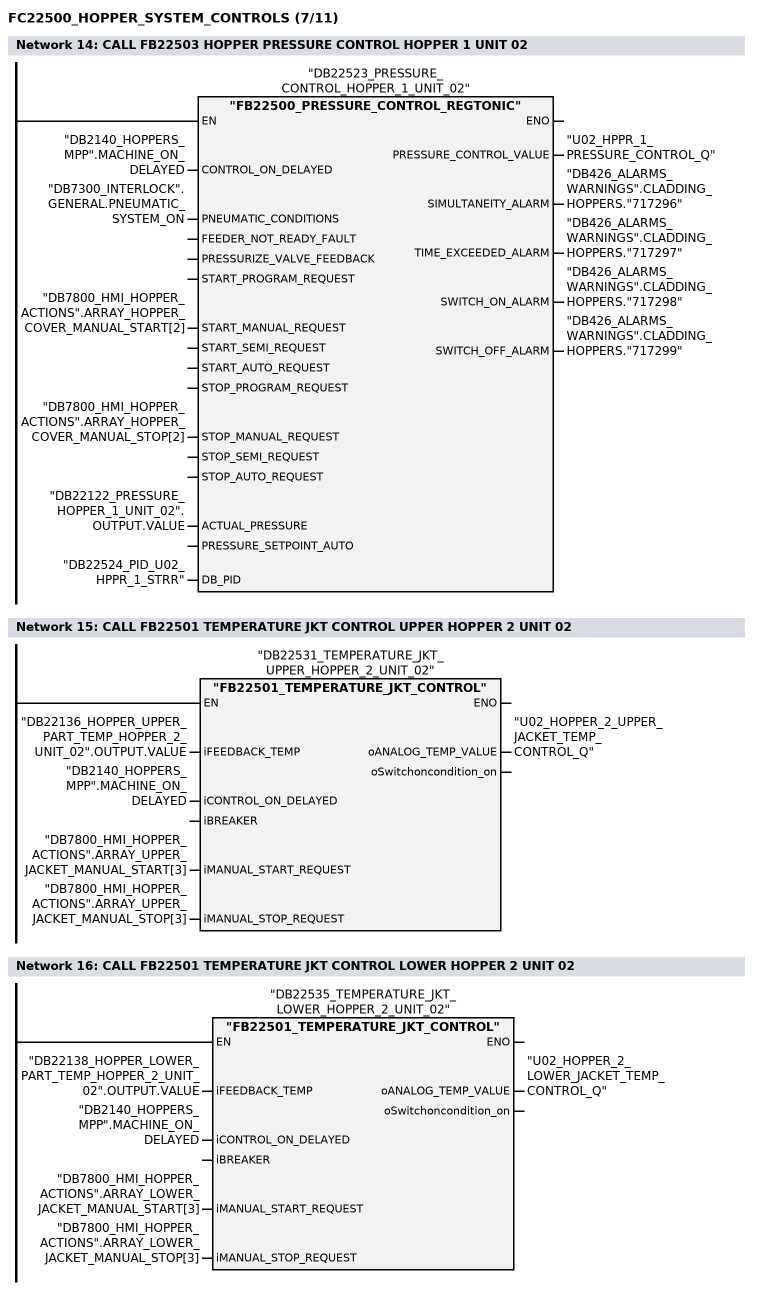
   RUNG wire#powerrail
      "DB22523_PRESSURE_CONTROL_HOPPER_1_UNIT_02"(CONTROL_ON_DELAYED := "DB2140_HOPPERS_MPP".MACHINE_ON_DELAYED, PNEUMATIC_CONDITIONS := "DB7300_INTERLOCK".GENERAL.PNEUMATIC_SYSTEM_ON, FEEDER_NOT_READY_FAULT :=, PRESSURIZE_VALVE_FEEDBACK :=, START_PROGRAM_REQUEST :=, START_MANUAL_REQUEST := "DB7800_HMI_HOPPER_ACTIONS".ARRAY_HOPPER_COVER_MANUAL_START[2], START_SEMI_REQUEST :=, START_AUTO_REQUEST :=, STOP_PROGRAM_REQUEST :=, STOP_MANUAL_REQUEST := "DB7800_HMI_HOPPER_ACTIONS".ARRAY_HOPPER_COVER_MANUAL_STOP[2], STOP_SEMI_REQUEST :=, STOP_AUTO_REQUEST :=, ACTUAL_PRESSURE := "DB22122_PRESSURE_HOPPER_1_UNIT_02".OUTPUT.VALUE, PRESSURE_SETPOINT_AUTO :=, DB_PID := "DB22524_PID_U02_HPPR_1_STRR", PRESSURE_CONTROL_VALUE => "U02_HPPR_1_PRESSURE_CONTROL_Q", SIMULTANEITY_ALARM => "DB426_ALARMS_WARNINGS".CLADDING_HOPPERS."717296", TIME_EXCEEDED_ALARM => "DB426_ALARMS_WARNINGS".CLADDING_HOPPERS."717297", SWITCH_ON_ALARM => "DB426_ALARMS_WARNINGS".CLADDING_HOPPERS."717298", SWITCH_OFF_ALARM => "DB426_ALARMS_WARNINGS".CLADDING_HOPPERS."717299")
   END_RUNG
   // the same network as SCL:
   "DB22523_PRESSURE_CONTROL_HOPPER_1_UNIT_02"(CONTROL_ON_DELAYED := "DB2140_HOPPERS_MPP".MACHINE_ON_DELAYED,   // "FB22500_PRESSURE_CONTROL_REGTONIC"
                           PNEUMATIC_CONDITIONS := "DB7300_INTERLOCK".GENERAL.PNEUMATIC_SYSTEM_ON,
                           START_MANUAL_REQUEST := "DB7800_HMI_HOPPER_ACTIONS".ARRAY_HOPPER_COVER_MANUAL_START[2],
                           STOP_MANUAL_REQUEST := "DB7800_HMI_HOPPER_ACTIONS".ARRAY_HOPPER_COVER_MANUAL_STOP[2],
                           ACTUAL_PRESSURE := "DB22122_PRESSURE_HOPPER_1_UNIT_02".OUTPUT.VALUE,
                           DB_PID := "DB22524_PID_U02_HPPR_1_STRR",
                           PRESSURE_CONTROL_VALUE => "U02_HPPR_1_PRESSURE_CONTROL_Q",
                           SIMULTANEITY_ALARM => "DB426_ALARMS_WARNINGS".CLADDING_HOPPERS."717296",
                           TIME_EXCEEDED_ALARM => "DB426_ALARMS_WARNINGS".CLADDING_HOPPERS."717297",
                           SWITCH_ON_ALARM => "DB426_ALARMS_WARNINGS".CLADDING_HOPPERS."717298",
                           SWITCH_OFF_ALARM => "DB426_ALARMS_WARNINGS".CLADDING_HOPPERS."717299");
END_REGION

REGION Network 15: CALL FB22501 TEMPERATURE JKT CONTROL UPPER HOPPER 2 UNIT 02
   RUNG wire#powerrail
      "DB22531_TEMPERATURE_JKT_UPPER_HOPPER_2_UNIT_02"(iFEEDBACK_TEMP := "DB22136_HOPPER_UPPER_PART_TEMP_HOPPER_2_UNIT_02".OUTPUT.VALUE, iCONTROL_ON_DELAYED := "DB2140_HOPPERS_MPP".MACHINE_ON_DELAYED, iBREAKER :=, iMANUAL_START_REQUEST := "DB7800_HMI_HOPPER_ACTIONS".ARRAY_UPPER_JACKET_MANUAL_START[3], iMANUAL_STOP_REQUEST := "DB7800_HMI_HOPPER_ACTIONS".ARRAY_UPPER_JACKET_MANUAL_STOP[3], oANALOG_TEMP_VALUE => "U02_HOPPER_2_UPPER_JACKET_TEMP_CONTROL_Q", oSwitchoncondition_on =>)
   END_RUNG
   // the same network as SCL:
   "DB22531_TEMPERATURE_JKT_UPPER_HOPPER_2_UNIT_02"(iFEEDBACK_TEMP := "DB22136_HOPPER_UPPER_PART_TEMP_HOPPER_2_UNIT_02".OUTPUT.VALUE,   // "FB22501_TEMPERATURE_JKT_CONTROL"
                           iCONTROL_ON_DELAYED := "DB2140_HOPPERS_MPP".MACHINE_ON_DELAYED,
                           iMANUAL_START_REQUEST := "DB7800_HMI_HOPPER_ACTIONS".ARRAY_UPPER_JACKET_MANUAL_START[3],
                           iMANUAL_STOP_REQUEST := "DB7800_HMI_HOPPER_ACTIONS".ARRAY_UPPER_JACKET_MANUAL_STOP[3],
                           oANALOG_TEMP_VALUE => "U02_HOPPER_2_UPPER_JACKET_TEMP_CONTROL_Q");
END_REGION

REGION Network 16: CALL FB22501 TEMPERATURE JKT CONTROL LOWER HOPPER 2 UNIT 02
   RUNG wire#powerrail
      "DB22535_TEMPERATURE_JKT_LOWER_HOPPER_2_UNIT_02"(iFEEDBACK_TEMP := "DB22138_HOPPER_LOWER_PART_TEMP_HOPPER_2_UNIT_02".OUTPUT.VALUE, iCONTROL_ON_DELAYED := "DB2140_HOPPERS_MPP".MACHINE_ON_DELAYED, iBREAKER :=, iMANUAL_START_REQUEST := "DB7800_HMI_HOPPER_ACTIONS".ARRAY_LOWER_JACKET_MANUAL_START[3], iMANUAL_STOP_REQUEST := "DB7800_HMI_HOPPER_ACTIONS".ARRAY_LOWER_JACKET_MANUAL_STOP[3], oANALOG_TEMP_VALUE => "U02_HOPPER_2_LOWER_JACKET_TEMP_CONTROL_Q", oSwitchoncondition_on =>)
   END_RUNG
   // the same network as SCL:
   "DB22535_TEMPERATURE_JKT_LOWER_HOPPER_2_UNIT_02"(iFEEDBACK_TEMP := "DB22138_HOPPER_LOWER_PART_TEMP_HOPPER_2_UNIT_02".OUTPUT.VALUE,   // "FB22501_TEMPERATURE_JKT_CONTROL"
                           iCONTROL_ON_DELAYED := "DB2140_HOPPERS_MPP".MACHINE_ON_DELAYED,
                           iMANUAL_START_REQUEST := "DB7800_HMI_HOPPER_ACTIONS".ARRAY_LOWER_JACKET_MANUAL_START[3],
                           iMANUAL_STOP_REQUEST := "DB7800_HMI_HOPPER_ACTIONS".ARRAY_LOWER_JACKET_MANUAL_STOP[3],
                           oANALOG_TEMP_VALUE => "U02_HOPPER_2_LOWER_JACKET_TEMP_CONTROL_Q");
END_REGION

REGION Network 17: CALL FB22502 MOTOR STIRRER CONTROL HOPPER 2 UNIT 02
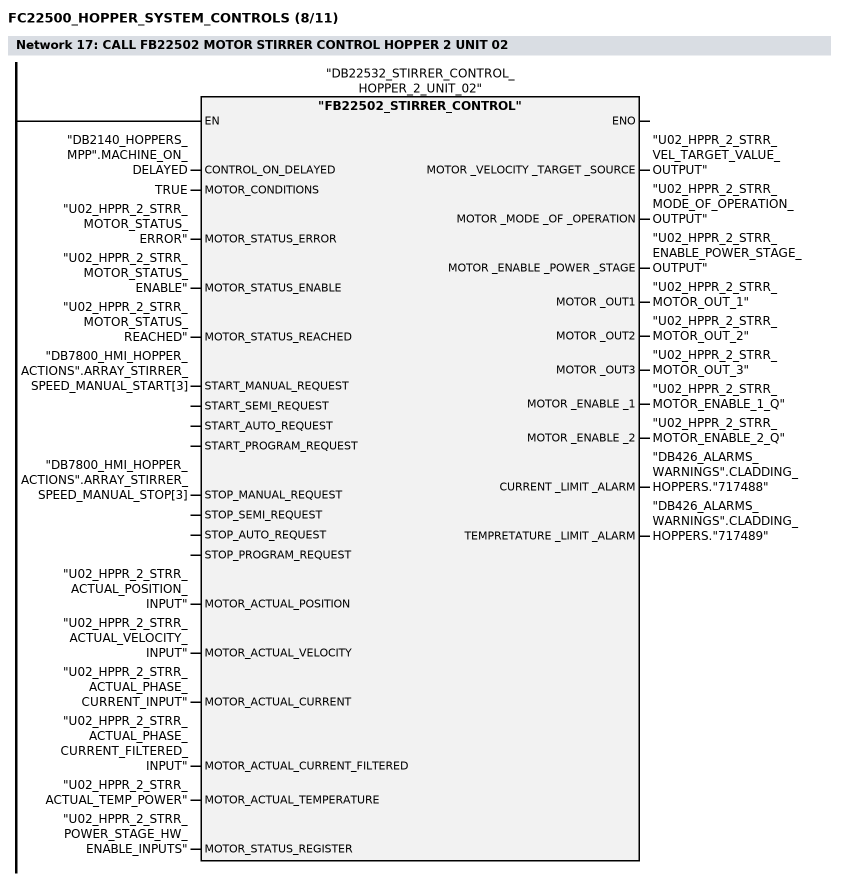
   RUNG wire#powerrail
      "DB22532_STIRRER_CONTROL_HOPPER_2_UNIT_02"(CONTROL_ON_DELAYED := "DB2140_HOPPERS_MPP".MACHINE_ON_DELAYED, MOTOR_CONDITIONS := TRUE, MOTOR_STATUS_ERROR := "U02_HPPR_2_STRR_MOTOR_STATUS_ERROR", MOTOR_STATUS_ENABLE := "U02_HPPR_2_STRR_MOTOR_STATUS_ENABLE", MOTOR_STATUS_REACHED := "U02_HPPR_2_STRR_MOTOR_STATUS_REACHED", START_MANUAL_REQUEST := "DB7800_HMI_HOPPER_ACTIONS".ARRAY_STIRRER_SPEED_MANUAL_START[3], START_SEMI_REQUEST :=, START_AUTO_REQUEST :=, START_PROGRAM_REQUEST :=, STOP_MANUAL_REQUEST := "DB7800_HMI_HOPPER_ACTIONS".ARRAY_STIRRER_SPEED_MANUAL_STOP[3], STOP_SEMI_REQUEST :=, STOP_AUTO_REQUEST :=, STOP_PROGRAM_REQUEST :=, MOTOR_ACTUAL_POSITION := "U02_HPPR_2_STRR_ACTUAL_POSITION_INPUT", MOTOR_ACTUAL_VELOCITY := "U02_HPPR_2_STRR_ACTUAL_VELOCITY_INPUT", MOTOR_ACTUAL_CURRENT := "U02_HPPR_2_STRR_ACTUAL_PHASE_CURRENT_INPUT", MOTOR_ACTUAL_CURRENT_FILTERED := "U02_HPPR_2_STRR_ACTUAL_PHASE_CURRENT_FILTERED_INPUT", MOTOR_ACTUAL_TEMPERATURE := "U02_HPPR_2_STRR_ACTUAL_TEMP_POWER", MOTOR_STATUS_REGISTER := "U02_HPPR_2_STRR_POWER_STAGE_HW_ENABLE_INPUTS", "MOTOR _VELOCITY _TARGET _SOURCE" => "U02_HPPR_2_STRR_VEL_TARGET_VALUE_OUTPUT", "MOTOR _MODE _OF _OPERATION" => "U02_HPPR_2_STRR_MODE_OF_OPERATION_OUTPUT", "MOTOR _ENABLE _POWER _STAGE" => "U02_HPPR_2_STRR_ENABLE_POWER_STAGE_OUTPUT", "MOTOR _OUT1" => "U02_HPPR_2_STRR_MOTOR_OUT_1", "MOTOR _OUT2" => "U02_HPPR_2_STRR_MOTOR_OUT_2", "MOTOR _OUT3" => "U02_HPPR_2_STRR_MOTOR_OUT_3", "MOTOR _ENABLE _1" => "U02_HPPR_2_STRR_MOTOR_ENABLE_1_Q", "MOTOR _ENABLE _2" => "U02_HPPR_2_STRR_MOTOR_ENABLE_2_Q", "CURRENT _LIMIT _ALARM" => "DB426_ALARMS_WARNINGS".CLADDING_HOPPERS."717488", "TEMPRETATURE _LIMIT _ALARM" => "DB426_ALARMS_WARNINGS".CLADDING_HOPPERS."717489")
   END_RUNG
   // the same network as SCL:
   "DB22532_STIRRER_CONTROL_HOPPER_2_UNIT_02"(CONTROL_ON_DELAYED := "DB2140_HOPPERS_MPP".MACHINE_ON_DELAYED,   // "FB22502_STIRRER_CONTROL"
                           MOTOR_CONDITIONS := TRUE,
                           MOTOR_STATUS_ERROR := "U02_HPPR_2_STRR_MOTOR_STATUS_ERROR",
                           MOTOR_STATUS_ENABLE := "U02_HPPR_2_STRR_MOTOR_STATUS_ENABLE",
                           MOTOR_STATUS_REACHED := "U02_HPPR_2_STRR_MOTOR_STATUS_REACHED",
                           START_MANUAL_REQUEST := "DB7800_HMI_HOPPER_ACTIONS".ARRAY_STIRRER_SPEED_MANUAL_START[3],
                           STOP_MANUAL_REQUEST := "DB7800_HMI_HOPPER_ACTIONS".ARRAY_STIRRER_SPEED_MANUAL_STOP[3],
                           MOTOR_ACTUAL_POSITION := "U02_HPPR_2_STRR_ACTUAL_POSITION_INPUT",
                           MOTOR_ACTUAL_VELOCITY := "U02_HPPR_2_STRR_ACTUAL_VELOCITY_INPUT",
                           MOTOR_ACTUAL_CURRENT := "U02_HPPR_2_STRR_ACTUAL_PHASE_CURRENT_INPUT",
                           MOTOR_ACTUAL_CURRENT_FILTERED := "U02_HPPR_2_STRR_ACTUAL_PHASE_CURRENT_FILTERED_INPUT",
                           MOTOR_ACTUAL_TEMPERATURE := "U02_HPPR_2_STRR_ACTUAL_TEMP_POWER",
                           MOTOR_STATUS_REGISTER := "U02_HPPR_2_STRR_POWER_STAGE_HW_ENABLE_INPUTS",
                           "MOTOR _VELOCITY _TARGET _SOURCE" => "U02_HPPR_2_STRR_VEL_TARGET_VALUE_OUTPUT",
                           "MOTOR _MODE _OF _OPERATION" => "U02_HPPR_2_STRR_MODE_OF_OPERATION_OUTPUT",
                           "MOTOR _ENABLE _POWER _STAGE" => "U02_HPPR_2_STRR_ENABLE_POWER_STAGE_OUTPUT",
                           "MOTOR _OUT1" => "U02_HPPR_2_STRR_MOTOR_OUT_1",
                           "MOTOR _OUT2" => "U02_HPPR_2_STRR_MOTOR_OUT_2",
                           "MOTOR _OUT3" => "U02_HPPR_2_STRR_MOTOR_OUT_3",
                           "MOTOR _ENABLE _1" => "U02_HPPR_2_STRR_MOTOR_ENABLE_1_Q",
                           "MOTOR _ENABLE _2" => "U02_HPPR_2_STRR_MOTOR_ENABLE_2_Q",
                           "CURRENT _LIMIT _ALARM" => "DB426_ALARMS_WARNINGS".CLADDING_HOPPERS."717488",
                           "TEMPRETATURE _LIMIT _ALARM" => "DB426_ALARMS_WARNINGS".CLADDING_HOPPERS."717489");
END_REGION

REGION Network 18: CALL FB22503 HOPPER PRESSURE CONTROL HOPPER 2 UNIT 02
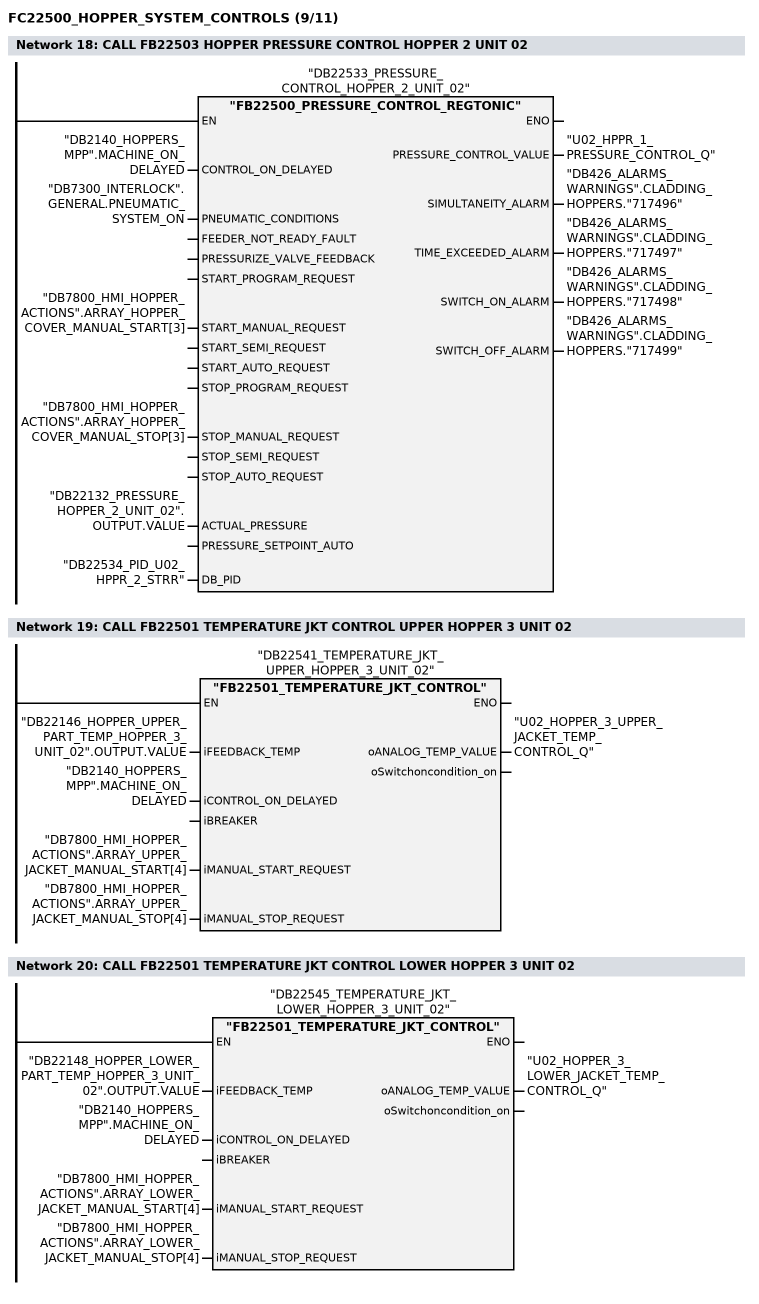
   RUNG wire#powerrail
      "DB22533_PRESSURE_CONTROL_HOPPER_2_UNIT_02"(CONTROL_ON_DELAYED := "DB2140_HOPPERS_MPP".MACHINE_ON_DELAYED, PNEUMATIC_CONDITIONS := "DB7300_INTERLOCK".GENERAL.PNEUMATIC_SYSTEM_ON, FEEDER_NOT_READY_FAULT :=, PRESSURIZE_VALVE_FEEDBACK :=, START_PROGRAM_REQUEST :=, START_MANUAL_REQUEST := "DB7800_HMI_HOPPER_ACTIONS".ARRAY_HOPPER_COVER_MANUAL_START[3], START_SEMI_REQUEST :=, START_AUTO_REQUEST :=, STOP_PROGRAM_REQUEST :=, STOP_MANUAL_REQUEST := "DB7800_HMI_HOPPER_ACTIONS".ARRAY_HOPPER_COVER_MANUAL_STOP[3], STOP_SEMI_REQUEST :=, STOP_AUTO_REQUEST :=, ACTUAL_PRESSURE := "DB22132_PRESSURE_HOPPER_2_UNIT_02".OUTPUT.VALUE, PRESSURE_SETPOINT_AUTO :=, DB_PID := "DB22534_PID_U02_HPPR_2_STRR", PRESSURE_CONTROL_VALUE => "U02_HPPR_1_PRESSURE_CONTROL_Q", SIMULTANEITY_ALARM => "DB426_ALARMS_WARNINGS".CLADDING_HOPPERS."717496", TIME_EXCEEDED_ALARM => "DB426_ALARMS_WARNINGS".CLADDING_HOPPERS."717497", SWITCH_ON_ALARM => "DB426_ALARMS_WARNINGS".CLADDING_HOPPERS."717498", SWITCH_OFF_ALARM => "DB426_ALARMS_WARNINGS".CLADDING_HOPPERS."717499")
   END_RUNG
   // the same network as SCL:
   "DB22533_PRESSURE_CONTROL_HOPPER_2_UNIT_02"(CONTROL_ON_DELAYED := "DB2140_HOPPERS_MPP".MACHINE_ON_DELAYED,   // "FB22500_PRESSURE_CONTROL_REGTONIC"
                           PNEUMATIC_CONDITIONS := "DB7300_INTERLOCK".GENERAL.PNEUMATIC_SYSTEM_ON,
                           START_MANUAL_REQUEST := "DB7800_HMI_HOPPER_ACTIONS".ARRAY_HOPPER_COVER_MANUAL_START[3],
                           STOP_MANUAL_REQUEST := "DB7800_HMI_HOPPER_ACTIONS".ARRAY_HOPPER_COVER_MANUAL_STOP[3],
                           ACTUAL_PRESSURE := "DB22132_PRESSURE_HOPPER_2_UNIT_02".OUTPUT.VALUE,
                           DB_PID := "DB22534_PID_U02_HPPR_2_STRR",
                           PRESSURE_CONTROL_VALUE => "U02_HPPR_1_PRESSURE_CONTROL_Q",
                           SIMULTANEITY_ALARM => "DB426_ALARMS_WARNINGS".CLADDING_HOPPERS."717496",
                           TIME_EXCEEDED_ALARM => "DB426_ALARMS_WARNINGS".CLADDING_HOPPERS."717497",
                           SWITCH_ON_ALARM => "DB426_ALARMS_WARNINGS".CLADDING_HOPPERS."717498",
                           SWITCH_OFF_ALARM => "DB426_ALARMS_WARNINGS".CLADDING_HOPPERS."717499");
END_REGION

REGION Network 19: CALL FB22501 TEMPERATURE JKT CONTROL UPPER HOPPER 3 UNIT 02
   RUNG wire#powerrail
      "DB22541_TEMPERATURE_JKT_UPPER_HOPPER_3_UNIT_02"(iFEEDBACK_TEMP := "DB22146_HOPPER_UPPER_PART_TEMP_HOPPER_3_UNIT_02".OUTPUT.VALUE, iCONTROL_ON_DELAYED := "DB2140_HOPPERS_MPP".MACHINE_ON_DELAYED, iBREAKER :=, iMANUAL_START_REQUEST := "DB7800_HMI_HOPPER_ACTIONS".ARRAY_UPPER_JACKET_MANUAL_START[4], iMANUAL_STOP_REQUEST := "DB7800_HMI_HOPPER_ACTIONS".ARRAY_UPPER_JACKET_MANUAL_STOP[4], oANALOG_TEMP_VALUE => "U02_HOPPER_3_UPPER_JACKET_TEMP_CONTROL_Q", oSwitchoncondition_on =>)
   END_RUNG
   // the same network as SCL:
   "DB22541_TEMPERATURE_JKT_UPPER_HOPPER_3_UNIT_02"(iFEEDBACK_TEMP := "DB22146_HOPPER_UPPER_PART_TEMP_HOPPER_3_UNIT_02".OUTPUT.VALUE,   // "FB22501_TEMPERATURE_JKT_CONTROL"
                           iCONTROL_ON_DELAYED := "DB2140_HOPPERS_MPP".MACHINE_ON_DELAYED,
                           iMANUAL_START_REQUEST := "DB7800_HMI_HOPPER_ACTIONS".ARRAY_UPPER_JACKET_MANUAL_START[4],
                           iMANUAL_STOP_REQUEST := "DB7800_HMI_HOPPER_ACTIONS".ARRAY_UPPER_JACKET_MANUAL_STOP[4],
                           oANALOG_TEMP_VALUE => "U02_HOPPER_3_UPPER_JACKET_TEMP_CONTROL_Q");
END_REGION

REGION Network 20: CALL FB22501 TEMPERATURE JKT CONTROL LOWER HOPPER 3 UNIT 02
   RUNG wire#powerrail
      "DB22545_TEMPERATURE_JKT_LOWER_HOPPER_3_UNIT_02"(iFEEDBACK_TEMP := "DB22148_HOPPER_LOWER_PART_TEMP_HOPPER_3_UNIT_02".OUTPUT.VALUE, iCONTROL_ON_DELAYED := "DB2140_HOPPERS_MPP".MACHINE_ON_DELAYED, iBREAKER :=, iMANUAL_START_REQUEST := "DB7800_HMI_HOPPER_ACTIONS".ARRAY_LOWER_JACKET_MANUAL_START[4], iMANUAL_STOP_REQUEST := "DB7800_HMI_HOPPER_ACTIONS".ARRAY_LOWER_JACKET_MANUAL_STOP[4], oANALOG_TEMP_VALUE => "U02_HOPPER_3_LOWER_JACKET_TEMP_CONTROL_Q", oSwitchoncondition_on =>)
   END_RUNG
   // the same network as SCL:
   "DB22545_TEMPERATURE_JKT_LOWER_HOPPER_3_UNIT_02"(iFEEDBACK_TEMP := "DB22148_HOPPER_LOWER_PART_TEMP_HOPPER_3_UNIT_02".OUTPUT.VALUE,   // "FB22501_TEMPERATURE_JKT_CONTROL"
                           iCONTROL_ON_DELAYED := "DB2140_HOPPERS_MPP".MACHINE_ON_DELAYED,
                           iMANUAL_START_REQUEST := "DB7800_HMI_HOPPER_ACTIONS".ARRAY_LOWER_JACKET_MANUAL_START[4],
                           iMANUAL_STOP_REQUEST := "DB7800_HMI_HOPPER_ACTIONS".ARRAY_LOWER_JACKET_MANUAL_STOP[4],
                           oANALOG_TEMP_VALUE => "U02_HOPPER_3_LOWER_JACKET_TEMP_CONTROL_Q");
END_REGION

REGION Network 21: CALL FB22502 MOTOR STIRRER CONTROL HOPPER 3 UNIT 02
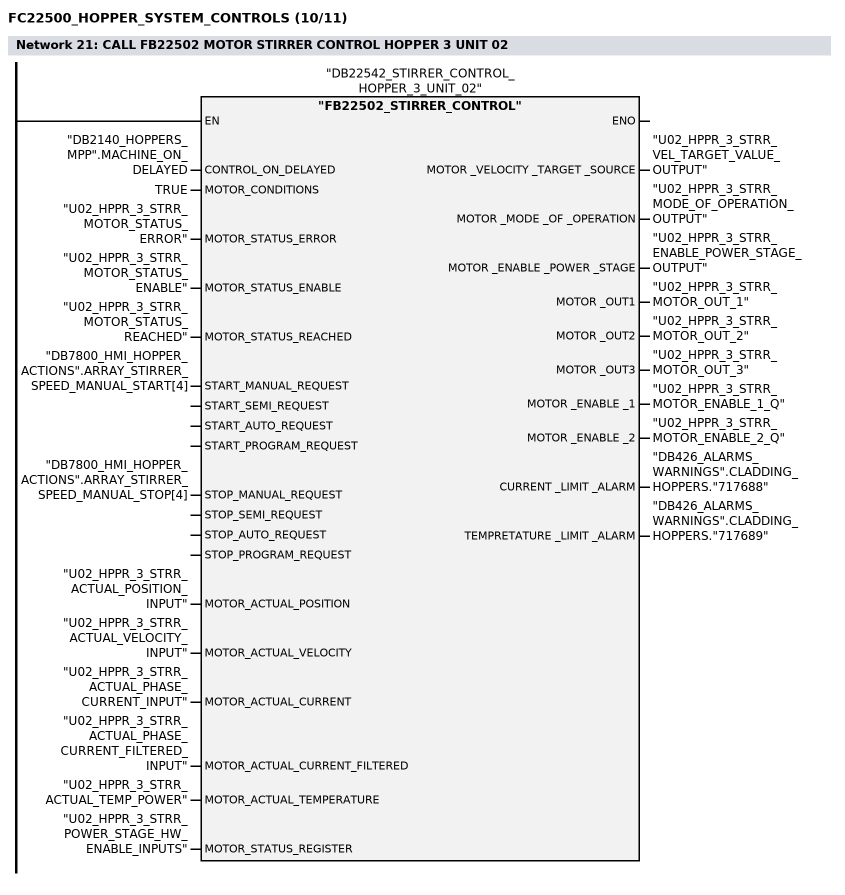
   RUNG wire#powerrail
      "DB22542_STIRRER_CONTROL_HOPPER_3_UNIT_02"(CONTROL_ON_DELAYED := "DB2140_HOPPERS_MPP".MACHINE_ON_DELAYED, MOTOR_CONDITIONS := TRUE, MOTOR_STATUS_ERROR := "U02_HPPR_3_STRR_MOTOR_STATUS_ERROR", MOTOR_STATUS_ENABLE := "U02_HPPR_3_STRR_MOTOR_STATUS_ENABLE", MOTOR_STATUS_REACHED := "U02_HPPR_3_STRR_MOTOR_STATUS_REACHED", START_MANUAL_REQUEST := "DB7800_HMI_HOPPER_ACTIONS".ARRAY_STIRRER_SPEED_MANUAL_START[4], START_SEMI_REQUEST :=, START_AUTO_REQUEST :=, START_PROGRAM_REQUEST :=, STOP_MANUAL_REQUEST := "DB7800_HMI_HOPPER_ACTIONS".ARRAY_STIRRER_SPEED_MANUAL_STOP[4], STOP_SEMI_REQUEST :=, STOP_AUTO_REQUEST :=, STOP_PROGRAM_REQUEST :=, MOTOR_ACTUAL_POSITION := "U02_HPPR_3_STRR_ACTUAL_POSITION_INPUT", MOTOR_ACTUAL_VELOCITY := "U02_HPPR_3_STRR_ACTUAL_VELOCITY_INPUT", MOTOR_ACTUAL_CURRENT := "U02_HPPR_3_STRR_ACTUAL_PHASE_CURRENT_INPUT", MOTOR_ACTUAL_CURRENT_FILTERED := "U02_HPPR_3_STRR_ACTUAL_PHASE_CURRENT_FILTERED_INPUT", MOTOR_ACTUAL_TEMPERATURE := "U02_HPPR_3_STRR_ACTUAL_TEMP_POWER", MOTOR_STATUS_REGISTER := "U02_HPPR_3_STRR_POWER_STAGE_HW_ENABLE_INPUTS", "MOTOR _VELOCITY _TARGET _SOURCE" => "U02_HPPR_3_STRR_VEL_TARGET_VALUE_OUTPUT", "MOTOR _MODE _OF _OPERATION" => "U02_HPPR_3_STRR_MODE_OF_OPERATION_OUTPUT", "MOTOR _ENABLE _POWER _STAGE" => "U02_HPPR_3_STRR_ENABLE_POWER_STAGE_OUTPUT", "MOTOR _OUT1" => "U02_HPPR_3_STRR_MOTOR_OUT_1", "MOTOR _OUT2" => "U02_HPPR_3_STRR_MOTOR_OUT_2", "MOTOR _OUT3" => "U02_HPPR_3_STRR_MOTOR_OUT_3", "MOTOR _ENABLE _1" => "U02_HPPR_3_STRR_MOTOR_ENABLE_1_Q", "MOTOR _ENABLE _2" => "U02_HPPR_3_STRR_MOTOR_ENABLE_2_Q", "CURRENT _LIMIT _ALARM" => "DB426_ALARMS_WARNINGS".CLADDING_HOPPERS."717688", "TEMPRETATURE _LIMIT _ALARM" => "DB426_ALARMS_WARNINGS".CLADDING_HOPPERS."717689")
   END_RUNG
   // the same network as SCL:
   "DB22542_STIRRER_CONTROL_HOPPER_3_UNIT_02"(CONTROL_ON_DELAYED := "DB2140_HOPPERS_MPP".MACHINE_ON_DELAYED,   // "FB22502_STIRRER_CONTROL"
                           MOTOR_CONDITIONS := TRUE,
                           MOTOR_STATUS_ERROR := "U02_HPPR_3_STRR_MOTOR_STATUS_ERROR",
                           MOTOR_STATUS_ENABLE := "U02_HPPR_3_STRR_MOTOR_STATUS_ENABLE",
                           MOTOR_STATUS_REACHED := "U02_HPPR_3_STRR_MOTOR_STATUS_REACHED",
                           START_MANUAL_REQUEST := "DB7800_HMI_HOPPER_ACTIONS".ARRAY_STIRRER_SPEED_MANUAL_START[4],
                           STOP_MANUAL_REQUEST := "DB7800_HMI_HOPPER_ACTIONS".ARRAY_STIRRER_SPEED_MANUAL_STOP[4],
                           MOTOR_ACTUAL_POSITION := "U02_HPPR_3_STRR_ACTUAL_POSITION_INPUT",
                           MOTOR_ACTUAL_VELOCITY := "U02_HPPR_3_STRR_ACTUAL_VELOCITY_INPUT",
                           MOTOR_ACTUAL_CURRENT := "U02_HPPR_3_STRR_ACTUAL_PHASE_CURRENT_INPUT",
                           MOTOR_ACTUAL_CURRENT_FILTERED := "U02_HPPR_3_STRR_ACTUAL_PHASE_CURRENT_FILTERED_INPUT",
                           MOTOR_ACTUAL_TEMPERATURE := "U02_HPPR_3_STRR_ACTUAL_TEMP_POWER",
                           MOTOR_STATUS_REGISTER := "U02_HPPR_3_STRR_POWER_STAGE_HW_ENABLE_INPUTS",
                           "MOTOR _VELOCITY _TARGET _SOURCE" => "U02_HPPR_3_STRR_VEL_TARGET_VALUE_OUTPUT",
                           "MOTOR _MODE _OF _OPERATION" => "U02_HPPR_3_STRR_MODE_OF_OPERATION_OUTPUT",
                           "MOTOR _ENABLE _POWER _STAGE" => "U02_HPPR_3_STRR_ENABLE_POWER_STAGE_OUTPUT",
                           "MOTOR _OUT1" => "U02_HPPR_3_STRR_MOTOR_OUT_1",
                           "MOTOR _OUT2" => "U02_HPPR_3_STRR_MOTOR_OUT_2",
                           "MOTOR _OUT3" => "U02_HPPR_3_STRR_MOTOR_OUT_3",
                           "MOTOR _ENABLE _1" => "U02_HPPR_3_STRR_MOTOR_ENABLE_1_Q",
                           "MOTOR _ENABLE _2" => "U02_HPPR_3_STRR_MOTOR_ENABLE_2_Q",
                           "CURRENT _LIMIT _ALARM" => "DB426_ALARMS_WARNINGS".CLADDING_HOPPERS."717688",
                           "TEMPRETATURE _LIMIT _ALARM" => "DB426_ALARMS_WARNINGS".CLADDING_HOPPERS."717689");
END_REGION

REGION Network 22: CALL FB22503 HOPPER PRESSURE CONTROL HOPPER 3 UNIT 02
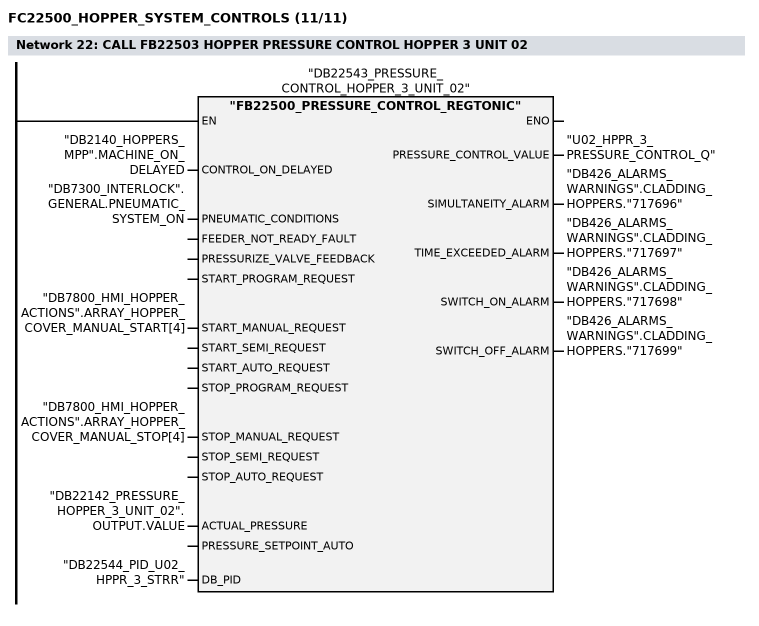
   RUNG wire#powerrail
      "DB22543_PRESSURE_CONTROL_HOPPER_3_UNIT_02"(CONTROL_ON_DELAYED := "DB2140_HOPPERS_MPP".MACHINE_ON_DELAYED, PNEUMATIC_CONDITIONS := "DB7300_INTERLOCK".GENERAL.PNEUMATIC_SYSTEM_ON, FEEDER_NOT_READY_FAULT :=, PRESSURIZE_VALVE_FEEDBACK :=, START_PROGRAM_REQUEST :=, START_MANUAL_REQUEST := "DB7800_HMI_HOPPER_ACTIONS".ARRAY_HOPPER_COVER_MANUAL_START[4], START_SEMI_REQUEST :=, START_AUTO_REQUEST :=, STOP_PROGRAM_REQUEST :=, STOP_MANUAL_REQUEST := "DB7800_HMI_HOPPER_ACTIONS".ARRAY_HOPPER_COVER_MANUAL_STOP[4], STOP_SEMI_REQUEST :=, STOP_AUTO_REQUEST :=, ACTUAL_PRESSURE := "DB22142_PRESSURE_HOPPER_3_UNIT_02".OUTPUT.VALUE, PRESSURE_SETPOINT_AUTO :=, DB_PID := "DB22544_PID_U02_HPPR_3_STRR", PRESSURE_CONTROL_VALUE => "U02_HPPR_3_PRESSURE_CONTROL_Q", SIMULTANEITY_ALARM => "DB426_ALARMS_WARNINGS".CLADDING_HOPPERS."717696", TIME_EXCEEDED_ALARM => "DB426_ALARMS_WARNINGS".CLADDING_HOPPERS."717697", SWITCH_ON_ALARM => "DB426_ALARMS_WARNINGS".CLADDING_HOPPERS."717698", SWITCH_OFF_ALARM => "DB426_ALARMS_WARNINGS".CLADDING_HOPPERS."717699")
   END_RUNG
   // the same network as SCL:
   "DB22543_PRESSURE_CONTROL_HOPPER_3_UNIT_02"(CONTROL_ON_DELAYED := "DB2140_HOPPERS_MPP".MACHINE_ON_DELAYED,   // "FB22500_PRESSURE_CONTROL_REGTONIC"
                           PNEUMATIC_CONDITIONS := "DB7300_INTERLOCK".GENERAL.PNEUMATIC_SYSTEM_ON,
                           START_MANUAL_REQUEST := "DB7800_HMI_HOPPER_ACTIONS".ARRAY_HOPPER_COVER_MANUAL_START[4],
                           STOP_MANUAL_REQUEST := "DB7800_HMI_HOPPER_ACTIONS".ARRAY_HOPPER_COVER_MANUAL_STOP[4],
                           ACTUAL_PRESSURE := "DB22142_PRESSURE_HOPPER_3_UNIT_02".OUTPUT.VALUE,
                           DB_PID := "DB22544_PID_U02_HPPR_3_STRR",
                           PRESSURE_CONTROL_VALUE => "U02_HPPR_3_PRESSURE_CONTROL_Q",
                           SIMULTANEITY_ALARM => "DB426_ALARMS_WARNINGS".CLADDING_HOPPERS."717696",
                           TIME_EXCEEDED_ALARM => "DB426_ALARMS_WARNINGS".CLADDING_HOPPERS."717697",
                           SWITCH_ON_ALARM => "DB426_ALARMS_WARNINGS".CLADDING_HOPPERS."717698",
                           SWITCH_OFF_ALARM => "DB426_ALARMS_WARNINGS".CLADDING_HOPPERS."717699");
END_REGION
END_FUNCTION

FUNCTION "FC22700_HOPPER_SEQUENCE_COORDINATOR" : Void   // FC22700, LAD
TITLE = FC22700 HOPPER SEQUENCE COORDINATOR
{ S7_Optimized_Access := 'TRUE' }
VERSION : 0.1
// stored: AutoNumber false, IsIECCheckEnabled false, SetENOAutomatically false, UDAEnableTagReadback false
BEGIN

REGION Network 1: CALL FC22701 LOAD FEEDER SEQUENCES
